REGION Network 51: 设备上砖流程 取砖X轴提前下降判断
   RUNG wire#powerrail
      { S7_Templates := "SrcType := DInt" } GE_Contact(in1 := #Z轴高速转低速编码值, in2 := #取砖X轴提前下降设定值)
      Coil( #上砖提前下降判断标志位 )
   END_RUNG
   // the same network as SCL:
   #上砖提前下降判断标志位 := #Z轴高速转低速编码值 >= #取砖X轴提前下降设定值;
END_REGION

REGION Network 52: 设备上砖流程 Z轴提前下降
   RUNG wire#powerrail
      Contact( #"上砖x轴正转转低速-待命位到2库" )
      wire#w1
      { S7_Templates := "SrcType := Byte" } EQ_Contact(in1 := #机械手取放砖选择, in2 := 2)
      wire#w2
      Contact( #上砖提前下降判断标志位 )
      Contact( #上砖z轴提前下降中间变量 )
      wire#w3
      I_Contact( #设备报警标志位 )
      Contact( #设备启动标志位 )
      S_Coil( #上砖z轴AB库位下降 )
   END_RUNG
   RUNG wire#powerrail
      Contact( #"上砖x轴反转转低速-待命位到1库" )
   END_RUNG wire#w1
   RUNG wire#w2
      I_Contact( #上砖提前下降判断标志位 )
      Contact( #上砖x轴到达A库下方中间变量 )
   END_RUNG wire#w3
   // the same network as SCL:
   IF (#"上砖x轴正转转低速-待命位到2库" OR #"上砖x轴反转转低速-待命位到1库") AND (#机械手取放砖选择 = 2) AND ((#上砖提前下降判断标志位 AND #上砖z轴提前下降中间变量) OR (NOT #上砖提前下降判断标志位 AND #上砖x轴到达A库下方中间变量)) AND NOT #设备报警标志位 AND #设备启动标志位 THEN
       #上砖z轴AB库位下降 := TRUE;
   END_IF;
END_REGION

REGION Network 53: 设备上砖流程 z轴下降取砖
   RUNG wire#powerrail
      Contact( #"上砖x轴正转转低速-待命位到2库" )
      wire#w1
      { S7_Templates := "SrcType := Byte" } EQ_Contact(in1 := #机械手取放砖选择, in2 := 2)
      Contact( #上砖x轴到达A库下方中间变量 )
      I_Contact( #设备报警标志位 )
      wire#w2
      R_Coil( #上砖X轴快速移动2库 )
   END_RUNG
   RUNG wire#powerrail
      Contact( #"上砖x轴反转转低速-待命位到1库" )
   END_RUNG wire#w1
   RUNG wire#w2
      R_Coil( #上砖X轴快速移动1库 )
   END_RUNG
   RUNG wire#w2
      R_Coil( #"上砖x轴正转转低速-待命位到2库" )
   END_RUNG
   RUNG wire#w2
      R_Coil( #"上砖x轴反转转低速-待命位到1库" )
   END_RUNG
   RUNG wire#w2
      Move(in := 0, out1 => #X轴减速光电通断次数, out2 => #减速光电计数传送)
   END_RUNG
   // the same network as SCL:
   IF (#"上砖x轴正转转低速-待命位到2库" OR #"上砖x轴反转转低速-待命位到1库") AND (#机械手取放砖选择 = 2) AND #上砖x轴到达A库下方中间变量 AND NOT #设备报警标志位 THEN
       #上砖X轴快速移动2库 := FALSE;
       #上砖X轴快速移动1库 := FALSE;
   END_IF;
   #_w1 := (#"上砖x轴正转转低速-待命位到2库" OR #"上砖x轴反转转低速-待命位到1库") AND (#机械手取放砖选择 = 2) AND #上砖x轴到达A库下方中间变量 AND NOT #设备报警标志位;
   IF #_w1 THEN
       #"上砖x轴正转转低速-待命位到2库" := FALSE;
       #"上砖x轴反转转低速-待命位到1库" := FALSE;
       #X轴减速光电通断次数 := 0;
       #减速光电计数传送 := 0;
   END_IF;
END_REGION

REGION Network 54: 设备上砖流程 到达检测，Z轴停止
   #上砖z轴AB库置取砖到位中间变量 := #上砖z轴AB库位下降 AND (#W轴吸取接近开关 OR #W轴吸取极限接近开关) AND (((#Z轴编码器实时值 >= #Z轴停止编码值下限) AND (#Z轴编码器实时值 <= #Z轴停止编码值上限)) OR #上砖吸取接近稳定时间定时器.Q);
   IF #上砖z轴AB库位下降 AND (#Z轴编码器实时值 > #Z轴高速转低速编码值) THEN #上砖真空电磁阀打开 := TRUE; END_IF;
   #上砖吸取接近稳定时间定时器.TON(IN := #上砖z轴AB库位下降 AND #W轴吸取接近开关, PT := #吸取到位稳定时间);   // TON coil
END_REGION

REGION Network 55: 设备上砖流程 压力开关检测标志位
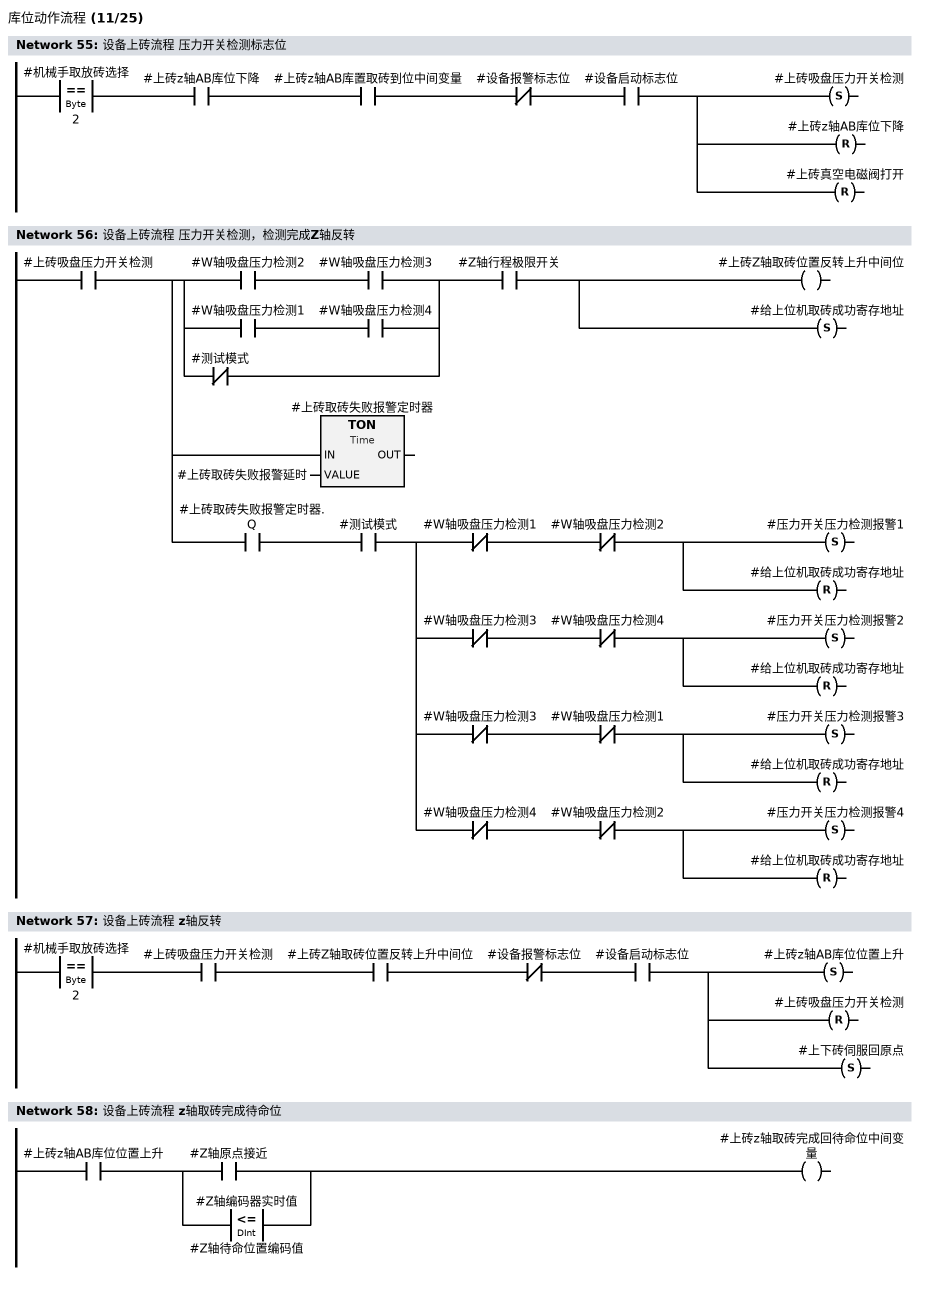
   RUNG wire#powerrail
      { S7_Templates := "SrcType := Byte" } EQ_Contact(in1 := #机械手取放砖选择, in2 := 2)
      Contact( #上砖z轴AB库位下降 )
      Contact( #上砖z轴AB库置取砖到位中间变量 )
      I_Contact( #设备报警标志位 )
      Contact( #设备启动标志位 )
      wire#w1
      S_Coil( #上砖吸盘压力开关检测 )
   END_RUNG
   RUNG wire#w1
      R_Coil( #上砖z轴AB库位下降 )
   END_RUNG
   RUNG wire#w1
      R_Coil( #上砖真空电磁阀打开 )
   END_RUNG
   // the same network as SCL:
   IF (#机械手取放砖选择 = 2) AND #上砖z轴AB库位下降 AND #上砖z轴AB库置取砖到位中间变量 AND NOT #设备报警标志位 AND #设备启动标志位 THEN
       #上砖吸盘压力开关检测 := TRUE;
   END_IF;
   #_w1 := (#机械手取放砖选择 = 2) AND #上砖z轴AB库位下降 AND #上砖z轴AB库置取砖到位中间变量 AND NOT #设备报警标志位 AND #设备启动标志位;
   IF #_w1 THEN
       #上砖z轴AB库位下降 := FALSE;
       #上砖真空电磁阀打开 := FALSE;
   END_IF;
END_REGION

REGION Network 56: 设备上砖流程 压力开关检测，检测完成Z轴反转
   #上砖Z轴取砖位置反转上升中间位 := #上砖吸盘压力开关检测 AND ((#W轴吸盘压力检测2 AND #W轴吸盘压力检测3) OR (#W轴吸盘压力检测1 AND #W轴吸盘压力检测4) OR NOT #测试模式) AND #Z轴行程极限开关;
   IF #上砖Z轴取砖位置反转上升中间位 THEN #给上位机取砖成功寄存地址 := TRUE; END_IF;
   #上砖取砖失败报警定时器.TON(IN := #上砖吸盘压力开关检测, PT := #上砖取砖失败报警延时);   // TON coil
   #_w1 := #上砖吸盘压力开关检测 AND #上砖取砖失败报警定时器.Q AND #测试模式;
   IF #_w1 AND NOT #W轴吸盘压力检测1 AND NOT #W轴吸盘压力检测2 THEN
       #压力开关压力检测报警1 := TRUE;
       #给上位机取砖成功寄存地址 := FALSE;
   END_IF;
   IF #_w1 AND NOT #W轴吸盘压力检测3 AND NOT #W轴吸盘压力检测4 THEN
       #压力开关压力检测报警2 := TRUE;
       #给上位机取砖成功寄存地址 := FALSE;
   END_IF;
   IF #_w1 AND NOT #W轴吸盘压力检测3 AND NOT #W轴吸盘压力检测1 THEN
       #压力开关压力检测报警3 := TRUE;
       #给上位机取砖成功寄存地址 := FALSE;
   END_IF;
   IF #_w1 AND NOT #W轴吸盘压力检测4 AND NOT #W轴吸盘压力检测2 THEN
       #压力开关压力检测报警4 := TRUE;
       #给上位机取砖成功寄存地址 := FALSE;
   END_IF;
END_REGION

REGION Network 57: 设备上砖流程 z轴反转
   RUNG wire#powerrail
      { S7_Templates := "SrcType := Byte" } EQ_Contact(in1 := #机械手取放砖选择, in2 := 2)
      Contact( #上砖吸盘压力开关检测 )
      Contact( #上砖Z轴取砖位置反转上升中间位 )
      I_Contact( #设备报警标志位 )
      Contact( #设备启动标志位 )
      wire#w1
      S_Coil( #上砖z轴AB库位位置上升 )
   END_RUNG
   RUNG wire#w1
      R_Coil( #上砖吸盘压力开关检测 )
   END_RUNG
   RUNG wire#w1
      S_Coil( #上下砖伺服回原点 )
   END_RUNG
   // the same network as SCL:
   IF (#机械手取放砖选择 = 2) AND #上砖吸盘压力开关检测 AND #上砖Z轴取砖位置反转上升中间位 AND NOT #设备报警标志位 AND #设备启动标志位 THEN
       #上砖z轴AB库位位置上升 := TRUE;
   END_IF;
   #_w1 := (#机械手取放砖选择 = 2) AND #上砖吸盘压力开关检测 AND #上砖Z轴取砖位置反转上升中间位 AND NOT #设备报警标志位 AND #设备启动标志位;
   IF #_w1 THEN
       #上砖吸盘压力开关检测 := FALSE;
       #上下砖伺服回原点 := TRUE;
   END_IF;
END_REGION

REGION Network 58: 设备上砖流程 z轴取砖完成待命位
   RUNG wire#powerrail
      Contact( #上砖z轴AB库位位置上升 )
      wire#w1
      Contact( #Z轴原点接近 )
      wire#w2
      Coil( #上砖z轴取砖完成回待命位中间变量 )
   END_RUNG
   RUNG wire#w1
      { S7_Templates := "SrcType := DInt" } LE_Contact(in1 := #Z轴编码器实时值, in2 := #Z轴待命位置编码值)
   END_RUNG wire#w2
   // the same network as SCL:
   #上砖z轴取砖完成回待命位中间变量 := #上砖z轴AB库位位置上升 AND (#Z轴原点接近 OR (#Z轴编码器实时值 <= #Z轴待命位置编码值));
END_REGION

REGION Network 59: 设备上砖流程 X轴正转高速A库--待命位 X轴反转高速B库---待命位
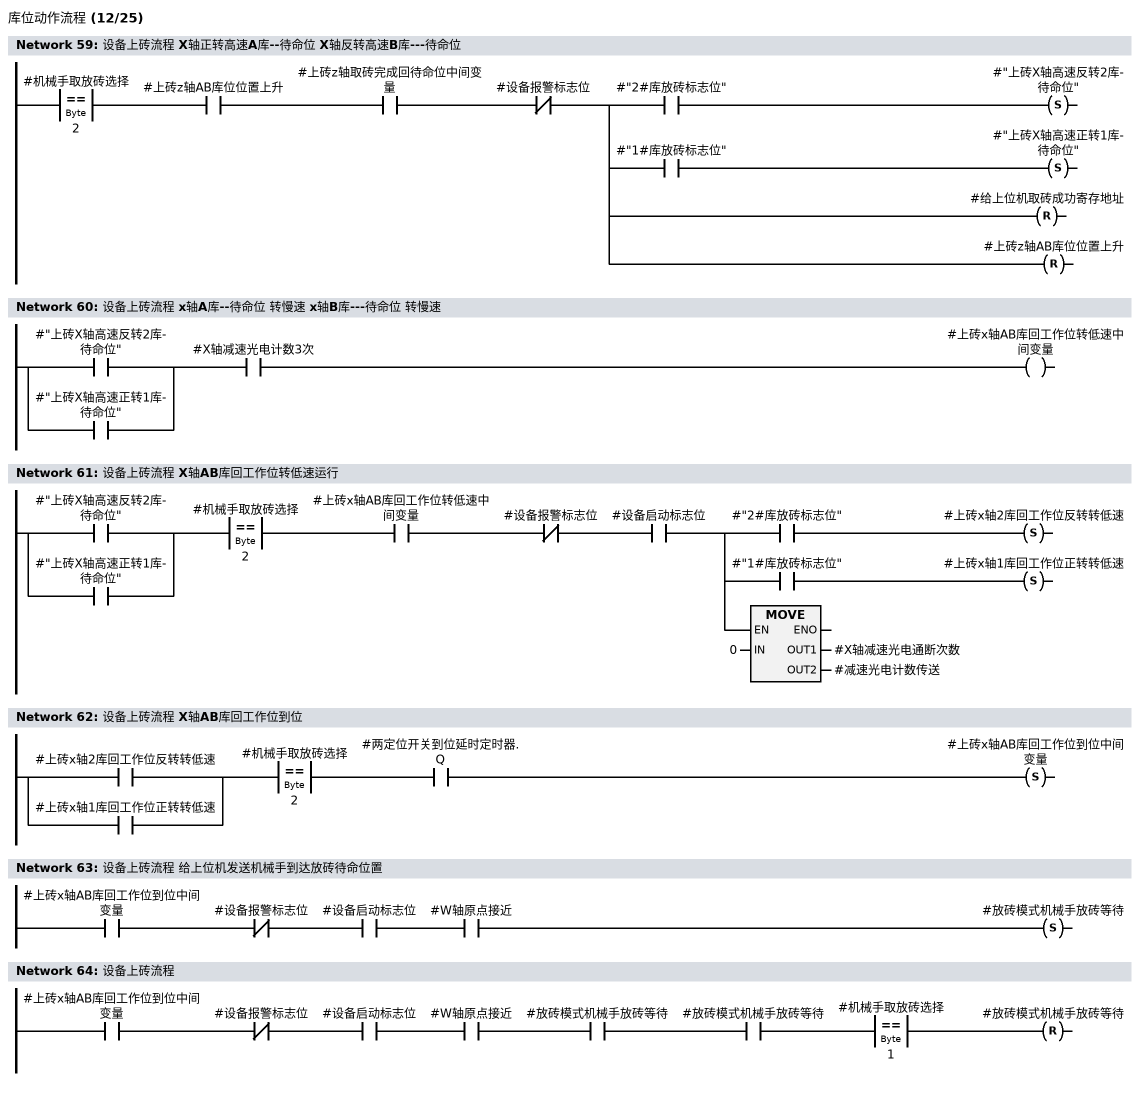
   RUNG wire#powerrail
      { S7_Templates := "SrcType := Byte" } EQ_Contact(in1 := #机械手取放砖选择, in2 := 2)
      Contact( #上砖z轴AB库位位置上升 )
      Contact( #上砖z轴取砖完成回待命位中间变量 )
      I_Contact( #设备报警标志位 )
      wire#w1
      Contact( #"2#库放砖标志位" )
      S_Coil( #"上砖X轴高速反转2库-待命位" )
   END_RUNG
   RUNG wire#w1
      Contact( #"1#库放砖标志位" )
      S_Coil( #"上砖X轴高速正转1库-待命位" )
   END_RUNG
   RUNG wire#w1
      R_Coil( #给上位机取砖成功寄存地址 )
   END_RUNG
   RUNG wire#w1
      R_Coil( #上砖z轴AB库位位置上升 )
   END_RUNG
   // the same network as SCL:
   #_w1 := (#机械手取放砖选择 = 2) AND #上砖z轴AB库位位置上升 AND #上砖z轴取砖完成回待命位中间变量 AND NOT #设备报警标志位;
   IF #_w1 AND #"2#库放砖标志位" THEN #"上砖X轴高速反转2库-待命位" := TRUE; END_IF;
   IF #_w1 AND #"1#库放砖标志位" THEN #"上砖X轴高速正转1库-待命位" := TRUE; END_IF;
   IF #_w1 THEN
       #给上位机取砖成功寄存地址 := FALSE;
       #上砖z轴AB库位位置上升 := FALSE;
   END_IF;
END_REGION

REGION Network 60: 设备上砖流程 x轴A库--待命位 转慢速 x轴B库---待命位 转慢速
   RUNG wire#powerrail
      Contact( #"上砖X轴高速反转2库-待命位" )
      wire#w1
      Contact( #X轴减速光电计数3次 )
      Coil( #上砖x轴AB库回工作位转低速中间变量 )
   END_RUNG
   RUNG wire#powerrail
      Contact( #"上砖X轴高速正转1库-待命位" )
   END_RUNG wire#w1
   // the same network as SCL:
   #上砖x轴AB库回工作位转低速中间变量 := (#"上砖X轴高速反转2库-待命位" OR #"上砖X轴高速正转1库-待命位") AND #X轴减速光电计数3次;
END_REGION

REGION Network 61: 设备上砖流程 X轴AB库回工作位转低速运行
   RUNG wire#powerrail
      Contact( #"上砖X轴高速反转2库-待命位" )
      wire#w1
      { S7_Templates := "SrcType := Byte" } EQ_Contact(in1 := #机械手取放砖选择, in2 := 2)
      Contact( #上砖x轴AB库回工作位转低速中间变量 )
      I_Contact( #设备报警标志位 )
      Contact( #设备启动标志位 )
      wire#w2
      Contact( #"2#库放砖标志位" )
      S_Coil( #上砖x轴2库回工作位反转转低速 )
   END_RUNG
   RUNG wire#powerrail
      Contact( #"上砖X轴高速正转1库-待命位" )
   END_RUNG wire#w1
   RUNG wire#w2
      Contact( #"1#库放砖标志位" )
      S_Coil( #上砖x轴1库回工作位正转转低速 )
   END_RUNG
   RUNG wire#w2
      Move(in := 0, out1 => #X轴减速光电通断次数, out2 => #减速光电计数传送)
   END_RUNG
   // the same network as SCL:
   #_w1 := (#"上砖X轴高速反转2库-待命位" OR #"上砖X轴高速正转1库-待命位") AND (#机械手取放砖选择 = 2) AND #上砖x轴AB库回工作位转低速中间变量 AND NOT #设备报警标志位 AND #设备启动标志位;
   IF #_w1 AND #"2#库放砖标志位" THEN #上砖x轴2库回工作位反转转低速 := TRUE; END_IF;
   IF #_w1 AND #"1#库放砖标志位" THEN #上砖x轴1库回工作位正转转低速 := TRUE; END_IF;
   IF #_w1 THEN
       #X轴减速光电通断次数 := 0;
       #减速光电计数传送 := 0;
   END_IF;
END_REGION

REGION Network 62: 设备上砖流程 X轴AB库回工作位到位
   RUNG wire#powerrail
      Contact( #上砖x轴2库回工作位反转转低速 )
      wire#w1
      { S7_Templates := "SrcType := Byte" } EQ_Contact(in1 := #机械手取放砖选择, in2 := 2)
      Contact( #两定位开关到位延时定时器.Q )
      S_Coil( #上砖x轴AB库回工作位到位中间变量 )
   END_RUNG
   RUNG wire#powerrail
      Contact( #上砖x轴1库回工作位正转转低速 )
   END_RUNG wire#w1
   // the same network as SCL:
   IF (#上砖x轴2库回工作位反转转低速 OR #上砖x轴1库回工作位正转转低速) AND (#机械手取放砖选择 = 2) AND #两定位开关到位延时定时器.Q THEN
       #上砖x轴AB库回工作位到位中间变量 := TRUE;
   END_IF;
END_REGION

REGION Network 63: 设备上砖流程 给上位机发送机械手到达放砖待命位置
   RUNG wire#powerrail
      Contact( #上砖x轴AB库回工作位到位中间变量 )
      I_Contact( #设备报警标志位 )
      Contact( #设备启动标志位 )
      Contact( #W轴原点接近 )
      S_Coil( #放砖模式机械手放砖等待 )
   END_RUNG
   // the same network as SCL:
   IF #上砖x轴AB库回工作位到位中间变量 AND NOT #设备报警标志位 AND #设备启动标志位 AND #W轴原点接近 THEN #放砖模式机械手放砖等待 := TRUE; END_IF;
END_REGION

REGION Network 64: 设备上砖流程
   RUNG wire#powerrail
      Contact( #上砖x轴AB库回工作位到位中间变量 )
      I_Contact( #设备报警标志位 )
      Contact( #设备启动标志位 )
      Contact( #W轴原点接近 )
      Contact( #放砖模式机械手放砖等待 )
      Contact( #放砖模式机械手放砖等待 )
      { S7_Templates := "SrcType := Byte" } EQ_Contact(in1 := #机械手取放砖选择, in2 := 1)
      R_Coil( #放砖模式机械手放砖等待 )
   END_RUNG
   // the same network as SCL:
   IF #上砖x轴AB库回工作位到位中间变量 AND NOT #设备报警标志位 AND #设备启动标志位 AND #W轴原点接近 AND #放砖模式机械手放砖等待 AND #放砖模式机械手放砖等待 AND (#机械手取放砖选择 = 1) THEN
       #放砖模式机械手放砖等待 := FALSE;
   END_IF;
END_REGION

REGION Network 65: 设备上砖流程 z轴下降放砖
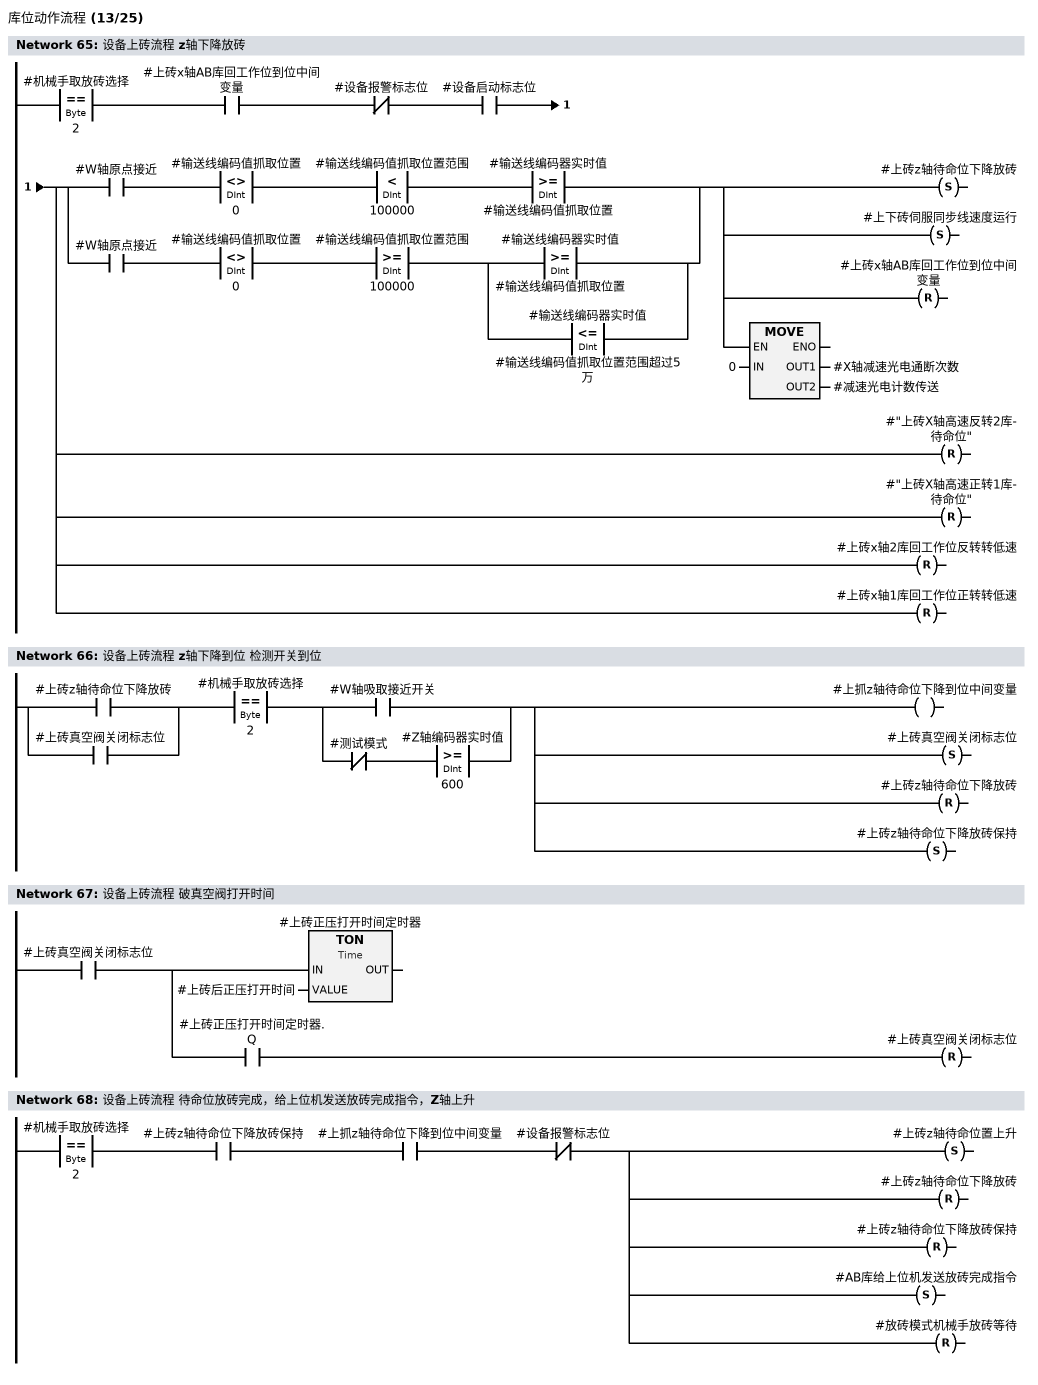
   RUNG wire#powerrail
      { S7_Templates := "SrcType := Byte" } EQ_Contact(in1 := #机械手取放砖选择, in2 := 2)
      Contact( #上砖x轴AB库回工作位到位中间变量 )
      I_Contact( #设备报警标志位 )
      Contact( #设备启动标志位 )
      wire#w1
      Contact( #W轴原点接近 )
      { S7_Templates := "SrcType := DInt" } NE_Contact(in1 := #输送线编码值抓取位置, in2 := 0)
      { S7_Templates := "SrcType := DInt" } LT_Contact(in1 := #输送线编码值抓取位置范围, in2 := 100000)
      { S7_Templates := "SrcType := DInt" } GE_Contact(in1 := #输送线编码器实时值, in2 := #输送线编码值抓取位置)
      wire#w2
      S_Coil( #上砖z轴待命位下降放砖 )
   END_RUNG
   RUNG wire#w1
      Contact( #W轴原点接近 )
      { S7_Templates := "SrcType := DInt" } NE_Contact(in1 := #输送线编码值抓取位置, in2 := 0)
      { S7_Templates := "SrcType := DInt" } GE_Contact(in1 := #输送线编码值抓取位置范围, in2 := 100000)
      wire#w3
      { S7_Templates := "SrcType := DInt" } GE_Contact(in1 := #输送线编码器实时值, in2 := #输送线编码值抓取位置)
   END_RUNG wire#w2
   RUNG wire#w3
      { S7_Templates := "SrcType := DInt" } LE_Contact(in1 := #输送线编码器实时值, in2 := #输送线编码值抓取位置范围超过5万)
   END_RUNG wire#w2
   RUNG wire#w2
      S_Coil( #上下砖伺服同步线速度运行 )
   END_RUNG
   RUNG wire#w2
      R_Coil( #上砖x轴AB库回工作位到位中间变量 )
   END_RUNG
   RUNG wire#w2
      Move(in := 0, out1 => #X轴减速光电通断次数, out2 => #减速光电计数传送)
   END_RUNG
   RUNG wire#w1
      R_Coil( #"上砖X轴高速反转2库-待命位" )
   END_RUNG
   RUNG wire#w1
      R_Coil( #"上砖X轴高速正转1库-待命位" )
   END_RUNG
   RUNG wire#w1
      R_Coil( #上砖x轴2库回工作位反转转低速 )
   END_RUNG
   RUNG wire#w1
      R_Coil( #上砖x轴1库回工作位正转转低速 )
   END_RUNG
   // the same network as SCL:
   #_w1 := (#机械手取放砖选择 = 2) AND #上砖x轴AB库回工作位到位中间变量 AND NOT #设备报警标志位 AND #设备启动标志位;
   IF #_w1 AND ((#W轴原点接近 AND (#输送线编码值抓取位置 <> 0) AND (#输送线编码值抓取位置范围 < 100000) AND (#输送线编码器实时值 >= #输送线编码值抓取位置)) OR (#W轴原点接近 AND (#输送线编码值抓取位置 <> 0) AND (#输送线编码值抓取位置范围 >= 100000) AND ((#输送线编码器实时值 >= #输送线编码值抓取位置) OR (#输送线编码器实时值 <= #输送线编码值抓取位置范围超过5万)))) THEN
       #上砖z轴待命位下降放砖 := TRUE;
       #上下砖伺服同步线速度运行 := TRUE;
       #上砖x轴AB库回工作位到位中间变量 := FALSE;
       #X轴减速光电通断次数 := 0;
       #减速光电计数传送 := 0;
   END_IF;
   IF #_w1 THEN
       #"上砖X轴高速反转2库-待命位" := FALSE;
       #"上砖X轴高速正转1库-待命位" := FALSE;
       #上砖x轴2库回工作位反转转低速 := FALSE;
       #上砖x轴1库回工作位正转转低速 := FALSE;
   END_IF;
END_REGION

REGION Network 66: 设备上砖流程 z轴下降到位 检测开关到位
   RUNG wire#powerrail
      Contact( #上砖z轴待命位下降放砖 )
      wire#w1
      { S7_Templates := "SrcType := Byte" } EQ_Contact(in1 := #机械手取放砖选择, in2 := 2)
      wire#w2
      Contact( #W轴吸取接近开关 )
      wire#w3
      Coil( #上抓z轴待命位下降到位中间变量 )
   END_RUNG
   RUNG wire#powerrail
      Contact( #上砖真空阀关闭标志位 )
   END_RUNG wire#w1
   RUNG wire#w2
      I_Contact( #测试模式 )
      { S7_Templates := "SrcType := DInt" } GE_Contact(in1 := #Z轴编码器实时值, in2 := 600)
   END_RUNG wire#w3
   RUNG wire#w3
      S_Coil( #上砖真空阀关闭标志位 )
   END_RUNG
   RUNG wire#w3
      R_Coil( #上砖z轴待命位下降放砖 )
   END_RUNG
   RUNG wire#w3
      S_Coil( #上砖z轴待命位下降放砖保持 )
   END_RUNG
   // the same network as SCL:
   #上抓z轴待命位下降到位中间变量 := (#上砖z轴待命位下降放砖 OR #上砖真空阀关闭标志位) AND (#机械手取放砖选择 = 2) AND (#W轴吸取接近开关 OR (NOT #测试模式 AND (#Z轴编码器实时值 >= 600)));
   IF #上抓z轴待命位下降到位中间变量 THEN
       #上砖真空阀关闭标志位 := TRUE;
       #上砖z轴待命位下降放砖 := FALSE;
       #上砖z轴待命位下降放砖保持 := TRUE;
   END_IF;
END_REGION

REGION Network 67: 设备上砖流程 破真空阀打开时间
   #上砖正压打开时间定时器.TON(IN := #上砖真空阀关闭标志位, PT := #上砖后正压打开时间);   // TON coil
   IF #上砖真空阀关闭标志位 AND #上砖正压打开时间定时器.Q THEN #上砖真空阀关闭标志位 := FALSE; END_IF;
END_REGION

REGION Network 68: 设备上砖流程 待命位放砖完成，给上位机发送放砖完成指令，Z轴上升
   RUNG wire#powerrail
      { S7_Templates := "SrcType := Byte" } EQ_Contact(in1 := #机械手取放砖选择, in2 := 2)
      Contact( #上砖z轴待命位下降放砖保持 )
      Contact( #上抓z轴待命位下降到位中间变量 )
      I_Contact( #设备报警标志位 )
      wire#w1
      S_Coil( #上砖z轴待命位置上升 )
   END_RUNG
   RUNG wire#w1
      R_Coil( #上砖z轴待命位下降放砖 )
   END_RUNG
   RUNG wire#w1
      R_Coil( #上砖z轴待命位下降放砖保持 )
   END_RUNG
   RUNG wire#w1
      S_Coil( #AB库给上位机发送放砖完成指令 )
   END_RUNG
   RUNG wire#w1
      R_Coil( #放砖模式机械手放砖等待 )
   END_RUNG
   // the same network as SCL:
   IF (#机械手取放砖选择 = 2) AND #上砖z轴待命位下降放砖保持 AND #上抓z轴待命位下降到位中间变量 AND NOT #设备报警标志位 THEN
       #上砖z轴待命位置上升 := TRUE;
       #上砖z轴待命位下降放砖 := FALSE;
   END_IF;
   #_w1 := (#机械手取放砖选择 = 2) AND #上砖z轴待命位下降放砖保持 AND #上抓z轴待命位下降到位中间变量 AND NOT #设备报警标志位;
   IF #_w1 THEN
       #上砖z轴待命位下降放砖保持 := FALSE;
       #AB库给上位机发送放砖完成指令 := TRUE;
       #放砖模式机械手放砖等待 := FALSE;
   END_IF;
END_REGION

REGION Network 69: 设备上砖流程 Z轴待命位上升到目标位
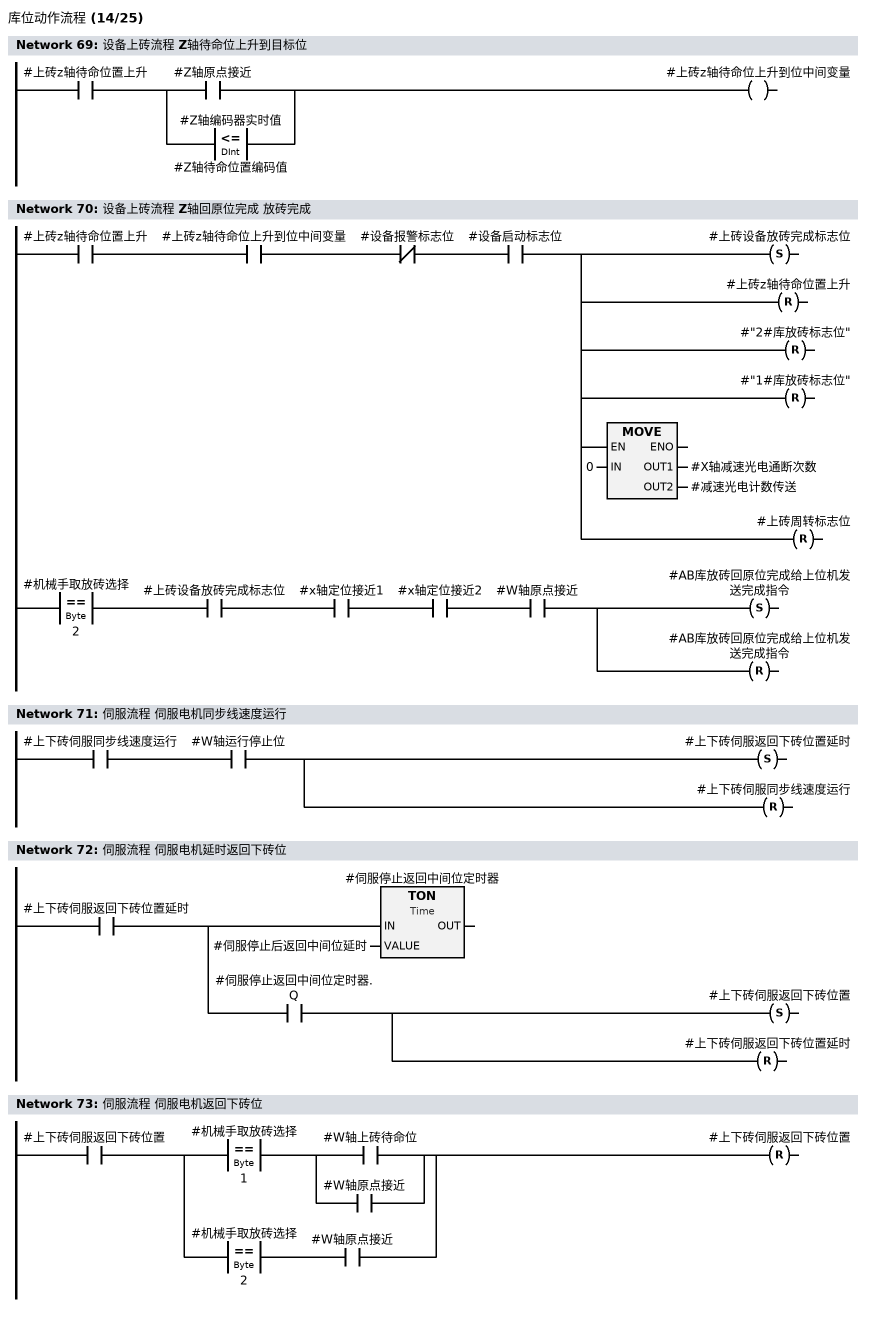
   RUNG wire#powerrail
      Contact( #上砖z轴待命位置上升 )
      wire#w1
      Contact( #Z轴原点接近 )
      wire#w2
      Coil( #上砖z轴待命位上升到位中间变量 )
   END_RUNG
   RUNG wire#w1
      { S7_Templates := "SrcType := DInt" } LE_Contact(in1 := #Z轴编码器实时值, in2 := #Z轴待命位置编码值)
   END_RUNG wire#w2
   // the same network as SCL:
   #上砖z轴待命位上升到位中间变量 := #上砖z轴待命位置上升 AND (#Z轴原点接近 OR (#Z轴编码器实时值 <= #Z轴待命位置编码值));
END_REGION

REGION Network 70: 设备上砖流程 Z轴回原位完成 放砖完成
   RUNG wire#powerrail
      Contact( #上砖z轴待命位置上升 )
      Contact( #上砖z轴待命位上升到位中间变量 )
      I_Contact( #设备报警标志位 )
      Contact( #设备启动标志位 )
      wire#w1
      S_Coil( #上砖设备放砖完成标志位 )
   END_RUNG
   RUNG wire#w1
      R_Coil( #上砖z轴待命位置上升 )
   END_RUNG
   RUNG wire#w1
      R_Coil( #"2#库放砖标志位" )
   END_RUNG
   RUNG wire#w1
      R_Coil( #"1#库放砖标志位" )
   END_RUNG
   RUNG wire#w1
      Move(in := 0, out1 => #X轴减速光电通断次数, out2 => #减速光电计数传送)
   END_RUNG
   RUNG wire#w1
      R_Coil( #上砖周转标志位 )
   END_RUNG
   RUNG wire#powerrail
      { S7_Templates := "SrcType := Byte" } EQ_Contact(in1 := #机械手取放砖选择, in2 := 2)
      Contact( #上砖设备放砖完成标志位 )
      Contact( #x轴定位接近1 )
      Contact( #x轴定位接近2 )
      Contact( #W轴原点接近 )
      wire#w2
      S_Coil( #AB库放砖回原位完成给上位机发送完成指令 )
   END_RUNG
   RUNG wire#w2
      R_Coil( #AB库放砖回原位完成给上位机发送完成指令 )
   END_RUNG
   // the same network as SCL:
   IF #上砖z轴待命位置上升 AND #上砖z轴待命位上升到位中间变量 AND NOT #设备报警标志位 AND #设备启动标志位 THEN #上砖设备放砖完成标志位 := TRUE; END_IF;
   #_w1 := #上砖z轴待命位置上升 AND #上砖z轴待命位上升到位中间变量 AND NOT #设备报警标志位 AND #设备启动标志位;
   IF #_w1 THEN
       #上砖z轴待命位置上升 := FALSE;
       #"2#库放砖标志位" := FALSE;
       #"1#库放砖标志位" := FALSE;
       #X轴减速光电通断次数 := 0;
       #减速光电计数传送 := 0;
       #上砖周转标志位 := FALSE;
   END_IF;
   IF (#机械手取放砖选择 = 2) AND #上砖设备放砖完成标志位 AND #x轴定位接近1 AND #x轴定位接近2 AND #W轴原点接近 THEN
       #AB库放砖回原位完成给上位机发送完成指令 := TRUE;
       #AB库放砖回原位完成给上位机发送完成指令 := FALSE;
   END_IF;
END_REGION

REGION Network 71: 伺服流程 伺服电机同步线速度运行
   RUNG wire#powerrail
      Contact( #上下砖伺服同步线速度运行 )
      Contact( #W轴运行停止位 )
      wire#w1
      S_Coil( #上下砖伺服返回下砖位置延时 )
   END_RUNG
   RUNG wire#w1
      R_Coil( #上下砖伺服同步线速度运行 )
   END_RUNG
   // the same network as SCL:
   IF #上下砖伺服同步线速度运行 AND #W轴运行停止位 THEN
       #上下砖伺服返回下砖位置延时 := TRUE;
       #上下砖伺服同步线速度运行 := FALSE;
   END_IF;
END_REGION

REGION Network 72: 伺服流程 伺服电机延时返回下砖位
   #伺服停止返回中间位定时器.TON(IN := #上下砖伺服返回下砖位置延时, PT := #伺服停止后返回中间位延时);   // TON coil
   IF #上下砖伺服返回下砖位置延时 AND #伺服停止返回中间位定时器.Q THEN
       #上下砖伺服返回下砖位置 := TRUE;
       #上下砖伺服返回下砖位置延时 := FALSE;
   END_IF;
END_REGION

REGION Network 73: 伺服流程 伺服电机返回下砖位
   RUNG wire#powerrail
      Contact( #上下砖伺服返回下砖位置 )
      wire#w1
      { S7_Templates := "SrcType := Byte" } EQ_Contact(in1 := #机械手取放砖选择, in2 := 1)
      wire#w2
      Contact( #W轴上砖待命位 )
      wire#w3
      R_Coil( #上下砖伺服返回下砖位置 )
   END_RUNG
   RUNG wire#w2
      Contact( #W轴原点接近 )
   END_RUNG wire#w3
   RUNG wire#w1
      { S7_Templates := "SrcType := Byte" } EQ_Contact(in1 := #机械手取放砖选择, in2 := 2)
      Contact( #W轴原点接近 )
   END_RUNG wire#w3
   // the same network as SCL:
   IF #上下砖伺服返回下砖位置 AND (((#机械手取放砖选择 = 1) AND (#W轴上砖待命位 OR #W轴原点接近)) OR ((#机械手取放砖选择 = 2) AND #W轴原点接近)) THEN
       #上下砖伺服返回下砖位置 := FALSE;
   END_IF;
END_REGION

REGION Network 74: 伺服流程 伺服回原点
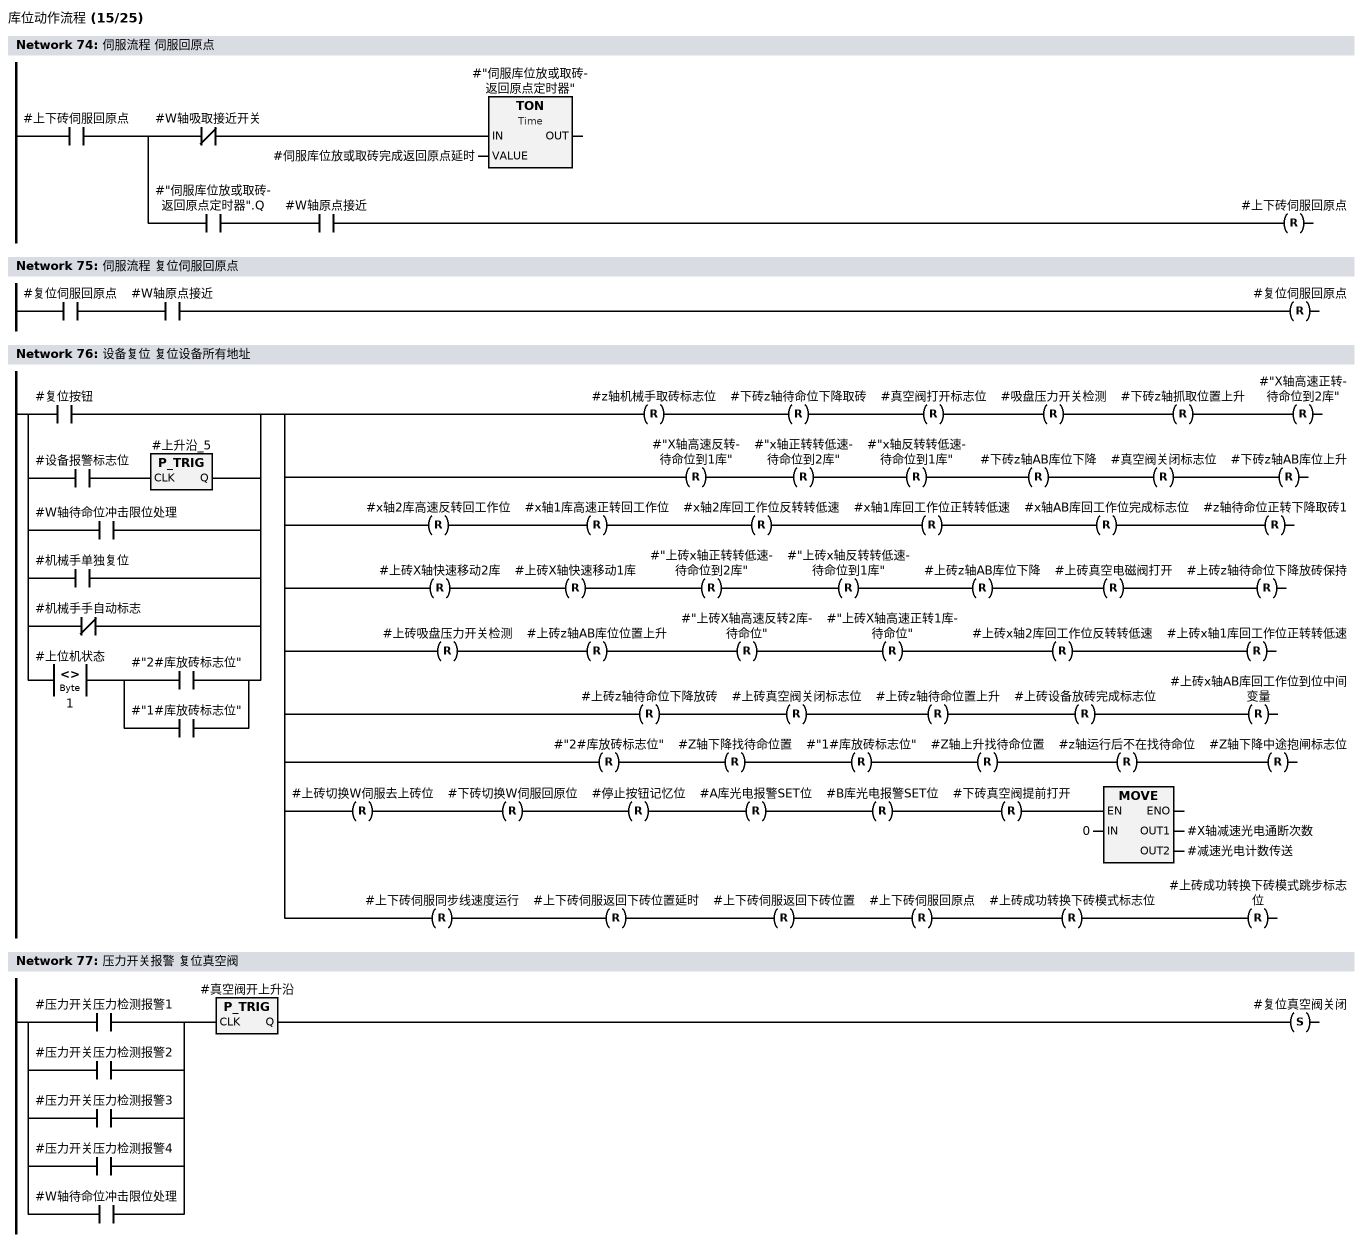
   #"伺服库位放或取砖-返回原点定时器".TON(IN := #上下砖伺服回原点 AND NOT #W轴吸取接近开关, PT := #伺服库位放或取砖完成返回原点延时);   // TON coil
   IF #上下砖伺服回原点 AND #"伺服库位放或取砖-返回原点定时器".Q AND #W轴原点接近 THEN #上下砖伺服回原点 := FALSE; END_IF;
END_REGION

REGION Network 75: 伺服流程 复位伺服回原点
   RUNG wire#powerrail
      Contact( #复位伺服回原点 )
      Contact( #W轴原点接近 )
      R_Coil( #复位伺服回原点 )
   END_RUNG
   // the same network as SCL:
   IF #复位伺服回原点 AND #W轴原点接近 THEN #复位伺服回原点 := FALSE; END_IF;
END_REGION

REGION Network 76: 设备复位 复位设备所有地址
   RUNG wire#powerrail
      Contact( #复位按钮 )
      wire#w1
      R_Coil( #z轴机械手取砖标志位 )
      R_Coil( #下砖z轴待命位下降取砖 )
      R_Coil( #真空阀打开标志位 )
      R_Coil( #吸盘压力开关检测 )
      R_Coil( #下砖z轴抓取位置上升 )
      R_Coil( #"X轴高速正转-待命位到2库" )
   END_RUNG
   RUNG wire#powerrail
      Contact( #设备报警标志位 )
      P_Trig( #上升沿_5 )
   END_RUNG wire#w1
   RUNG wire#powerrail
      Contact( #W轴待命位冲击限位处理 )
   END_RUNG wire#w1
   RUNG wire#powerrail
      Contact( #机械手单独复位 )
   END_RUNG wire#w1
   RUNG wire#powerrail
      I_Contact( #机械手手自动标志 )
   END_RUNG wire#w1
   RUNG wire#powerrail
      { S7_Templates := "SrcType := Byte" } NE_Contact(in1 := #上位机状态, in2 := 1)
      wire#w2
      Contact( #"2#库放砖标志位" )
   END_RUNG wire#w1
   RUNG wire#w2
      Contact( #"1#库放砖标志位" )
   END_RUNG wire#w1
   RUNG wire#w1
      R_Coil( #"X轴高速反转-待命位到1库" )
      R_Coil( #"x轴正转转低速-待命位到2库" )
      R_Coil( #"x轴反转转低速-待命位到1库" )
      R_Coil( #下砖z轴AB库位下降 )
      R_Coil( #真空阀关闭标志位 )
      R_Coil( #下砖z轴AB库位上升 )
   END_RUNG
   RUNG wire#w1
      R_Coil( #x轴2库高速反转回工作位 )
      R_Coil( #x轴1库高速正转回工作位 )
      R_Coil( #x轴2库回工作位反转转低速 )
      R_Coil( #x轴1库回工作位正转转低速 )
      R_Coil( #x轴AB库回工作位完成标志位 )
      R_Coil( #z轴待命位正转下降取砖1 )
   END_RUNG
   RUNG wire#w1
      R_Coil( #上砖X轴快速移动2库 )
      R_Coil( #上砖X轴快速移动1库 )
      R_Coil( #"上砖x轴正转转低速-待命位到2库" )
      R_Coil( #"上砖x轴反转转低速-待命位到1库" )
      R_Coil( #上砖z轴AB库位下降 )
      R_Coil( #上砖真空电磁阀打开 )
      R_Coil( #上砖z轴待命位下降放砖保持 )
   END_RUNG
   RUNG wire#w1
      R_Coil( #上砖吸盘压力开关检测 )
      R_Coil( #上砖z轴AB库位位置上升 )
      R_Coil( #"上砖X轴高速反转2库-待命位" )
      R_Coil( #"上砖X轴高速正转1库-待命位" )
      R_Coil( #上砖x轴2库回工作位反转转低速 )
      R_Coil( #上砖x轴1库回工作位正转转低速 )
   END_RUNG
   RUNG wire#w1
      R_Coil( #上砖z轴待命位下降放砖 )
      R_Coil( #上砖真空阀关闭标志位 )
      R_Coil( #上砖z轴待命位置上升 )
      R_Coil( #上砖设备放砖完成标志位 )
      R_Coil( #上砖x轴AB库回工作位到位中间变量 )
   END_RUNG
   RUNG wire#w1
      R_Coil( #"2#库放砖标志位" )
      R_Coil( #Z轴下降找待命位置 )
      R_Coil( #"1#库放砖标志位" )
      R_Coil( #Z轴上升找待命位置 )
      R_Coil( #z轴运行后不在找待命位 )
      R_Coil( #Z轴下降中途抱闸标志位 )
   END_RUNG
   RUNG wire#w1
      R_Coil( #上砖切换W伺服去上砖位 )
      R_Coil( #下砖切换W伺服回原位 )
      R_Coil( #停止按钮记忆位 )
      R_Coil( #A库光电报警SET位 )
      R_Coil( #B库光电报警SET位 )
      R_Coil( #下砖真空阀提前打开 )
      Move(in := 0, out1 => #X轴减速光电通断次数, out2 => #减速光电计数传送)
   END_RUNG
   RUNG wire#w1
      R_Coil( #上下砖伺服同步线速度运行 )
      R_Coil( #上下砖伺服返回下砖位置延时 )
      R_Coil( #上下砖伺服返回下砖位置 )
      R_Coil( #上下砖伺服回原点 )
      R_Coil( #上砖成功转换下砖模式标志位 )
      R_Coil( #上砖成功转换下砖模式跳步标志位 )
   END_RUNG
   // the same network as SCL:
   #_w1 := #设备报警标志位 AND NOT #上升沿_5;   // rising edge
   #上升沿_5 := #设备报警标志位;
   IF #复位按钮 OR #_w1 OR #W轴待命位冲击限位处理 OR #机械手单独复位 OR NOT #机械手手自动标志 OR ((#上位机状态 <> 1) AND (#"2#库放砖标志位" OR #"1#库放砖标志位")) THEN
       #z轴机械手取砖标志位 := FALSE;
       #下砖z轴待命位下降取砖 := FALSE;
       #真空阀打开标志位 := FALSE;
       #吸盘压力开关检测 := FALSE;
       #下砖z轴抓取位置上升 := FALSE;
       #"X轴高速正转-待命位到2库" := FALSE;
       #"X轴高速反转-待命位到1库" := FALSE;
       #"x轴正转转低速-待命位到2库" := FALSE;
       #"x轴反转转低速-待命位到1库" := FALSE;
       #下砖z轴AB库位下降 := FALSE;
       #真空阀关闭标志位 := FALSE;
       #下砖z轴AB库位上升 := FALSE;
       #x轴2库高速反转回工作位 := FALSE;
       #x轴1库高速正转回工作位 := FALSE;
       #x轴2库回工作位反转转低速 := FALSE;
       #x轴1库回工作位正转转低速 := FALSE;
       #x轴AB库回工作位完成标志位 := FALSE;
       #z轴待命位正转下降取砖1 := FALSE;
       #上砖X轴快速移动2库 := FALSE;
       #上砖X轴快速移动1库 := FALSE;
       #"上砖x轴正转转低速-待命位到2库" := FALSE;
       #"上砖x轴反转转低速-待命位到1库" := FALSE;
       #上砖z轴AB库位下降 := FALSE;
       #上砖真空电磁阀打开 := FALSE;
       #上砖z轴待命位下降放砖保持 := FALSE;
       #上砖吸盘压力开关检测 := FALSE;
       #上砖z轴AB库位位置上升 := FALSE;
       #"上砖X轴高速反转2库-待命位" := FALSE;
       #"上砖X轴高速正转1库-待命位" := FALSE;
       #上砖x轴2库回工作位反转转低速 := FALSE;
       #上砖x轴1库回工作位正转转低速 := FALSE;
       #上砖z轴待命位下降放砖 := FALSE;
       #上砖真空阀关闭标志位 := FALSE;
       #上砖z轴待命位置上升 := FALSE;
       #上砖设备放砖完成标志位 := FALSE;
       #上砖x轴AB库回工作位到位中间变量 := FALSE;
   END_IF;
   #_w2 := #复位按钮 OR #_w1 OR #W轴待命位冲击限位处理 OR #机械手单独复位 OR NOT #机械手手自动标志 OR ((#上位机状态 <> 1) AND (#"2#库放砖标志位" OR #"1#库放砖标志位"));
   IF #_w2 THEN
       #"2#库放砖标志位" := FALSE;
       #Z轴下降找待命位置 := FALSE;
       #"1#库放砖标志位" := FALSE;
       #Z轴上升找待命位置 := FALSE;
       #z轴运行后不在找待命位 := FALSE;
       #Z轴下降中途抱闸标志位 := FALSE;
       #上砖切换W伺服去上砖位 := FALSE;
       #下砖切换W伺服回原位 := FALSE;
       #停止按钮记忆位 := FALSE;
       #A库光电报警SET位 := FALSE;
       #B库光电报警SET位 := FALSE;
       #下砖真空阀提前打开 := FALSE;
       #X轴减速光电通断次数 := 0;
       #减速光电计数传送 := 0;
       #上下砖伺服同步线速度运行 := FALSE;
       #上下砖伺服返回下砖位置延时 := FALSE;
       #上下砖伺服返回下砖位置 := FALSE;
       #上下砖伺服回原点 := FALSE;
       #上砖成功转换下砖模式标志位 := FALSE;
       #上砖成功转换下砖模式跳步标志位 := FALSE;
   END_IF;
END_REGION

REGION Network 77: 压力开关报警 复位真空阀
   RUNG wire#powerrail
      Contact( #压力开关压力检测报警1 )
      wire#w1
      P_Trig( #真空阀开上升沿 )
      S_Coil( #复位真空阀关闭 )
   END_RUNG
   RUNG wire#powerrail
      Contact( #压力开关压力检测报警2 )
   END_RUNG wire#w1
   RUNG wire#powerrail
      Contact( #压力开关压力检测报警3 )
   END_RUNG wire#w1
   RUNG wire#powerrail
      Contact( #压力开关压力检测报警4 )
   END_RUNG wire#w1
   RUNG wire#powerrail
      Contact( #W轴待命位冲击限位处理 )
   END_RUNG wire#w1
   // the same network as SCL:
   #_w1 := #压力开关压力检测报警1 OR #压力开关压力检测报警2 OR #压力开关压力检测报警3 OR #压力开关压力检测报警4 OR #W轴待命位冲击限位处理;
   #_w2 := #_w1 AND NOT #真空阀开上升沿;   // rising edge
   #真空阀开上升沿 := #_w1;
   IF #_w2 THEN #复位真空阀关闭 := TRUE; END_IF;
END_REGION

REGION Network 78: 设备复位开始
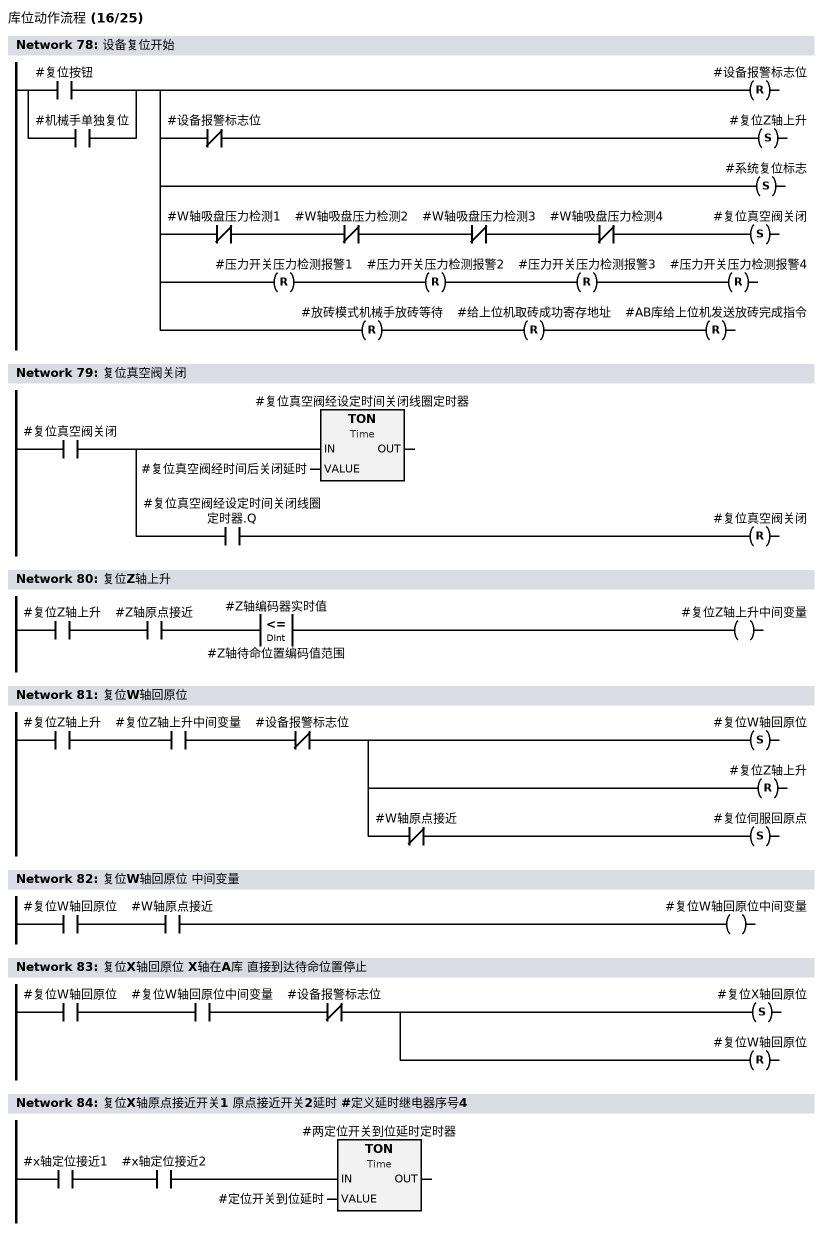
   RUNG wire#powerrail
      Contact( #复位按钮 )
      wire#w1
      R_Coil( #设备报警标志位 )
   END_RUNG
   RUNG wire#powerrail
      Contact( #机械手单独复位 )
   END_RUNG wire#w1
   RUNG wire#w1
      I_Contact( #设备报警标志位 )
      S_Coil( #复位Z轴上升 )
   END_RUNG
   RUNG wire#w1
      S_Coil( #系统复位标志 )
   END_RUNG
   RUNG wire#w1
      I_Contact( #W轴吸盘压力检测1 )
      I_Contact( #W轴吸盘压力检测2 )
      I_Contact( #W轴吸盘压力检测3 )
      I_Contact( #W轴吸盘压力检测4 )
      S_Coil( #复位真空阀关闭 )
   END_RUNG
   RUNG wire#w1
      R_Coil( #压力开关压力检测报警1 )
      R_Coil( #压力开关压力检测报警2 )
      R_Coil( #压力开关压力检测报警3 )
      R_Coil( #压力开关压力检测报警4 )
   END_RUNG
   RUNG wire#w1
      R_Coil( #放砖模式机械手放砖等待 )
      R_Coil( #给上位机取砖成功寄存地址 )
      R_Coil( #AB库给上位机发送放砖完成指令 )
   END_RUNG
   // the same network as SCL:
   #_w1 := #复位按钮 OR #机械手单独复位;
   IF #_w1 THEN #设备报警标志位 := FALSE; END_IF;
   IF #_w1 AND NOT #设备报警标志位 THEN #复位Z轴上升 := TRUE; END_IF;
   IF #_w1 THEN #系统复位标志 := TRUE; END_IF;
   IF #_w1 AND NOT #W轴吸盘压力检测1 AND NOT #W轴吸盘压力检测2 AND NOT #W轴吸盘压力检测3 AND NOT #W轴吸盘压力检测4 THEN
       #复位真空阀关闭 := TRUE;
   END_IF;
   IF #_w1 THEN
       #压力开关压力检测报警1 := FALSE;
       #压力开关压力检测报警2 := FALSE;
       #压力开关压力检测报警3 := FALSE;
       #压力开关压力检测报警4 := FALSE;
       #放砖模式机械手放砖等待 := FALSE;
       #给上位机取砖成功寄存地址 := FALSE;
       #AB库给上位机发送放砖完成指令 := FALSE;
   END_IF;
END_REGION

REGION Network 79: 复位真空阀关闭
   #复位真空阀经设定时间关闭线圈定时器.TON(IN := #复位真空阀关闭, PT := #复位真空阀经时间后关闭延时);   // TON coil
   IF #复位真空阀关闭 AND #复位真空阀经设定时间关闭线圈定时器.Q THEN #复位真空阀关闭 := FALSE; END_IF;
END_REGION

REGION Network 80: 复位Z轴上升
   RUNG wire#powerrail
      Contact( #复位Z轴上升 )
      Contact( #Z轴原点接近 )
      { S7_Templates := "SrcType := DInt" } LE_Contact(in1 := #Z轴编码器实时值, in2 := #Z轴待命位置编码值范围)
      Coil( #复位Z轴上升中间变量 )
   END_RUNG
   // the same network as SCL:
   #复位Z轴上升中间变量 := #复位Z轴上升 AND #Z轴原点接近 AND (#Z轴编码器实时值 <= #Z轴待命位置编码值范围);
END_REGION

REGION Network 81: 复位W轴回原位
   RUNG wire#powerrail
      Contact( #复位Z轴上升 )
      Contact( #复位Z轴上升中间变量 )
      I_Contact( #设备报警标志位 )
      wire#w1
      S_Coil( #复位W轴回原位 )
   END_RUNG
   RUNG wire#w1
      R_Coil( #复位Z轴上升 )
   END_RUNG
   RUNG wire#w1
      I_Contact( #W轴原点接近 )
      S_Coil( #复位伺服回原点 )
   END_RUNG
   // the same network as SCL:
   #_w1 := #复位Z轴上升 AND #复位Z轴上升中间变量 AND NOT #设备报警标志位;
   IF #_w1 THEN
       #复位W轴回原位 := TRUE;
       #复位Z轴上升 := FALSE;
   END_IF;
   IF #_w1 AND NOT #W轴原点接近 THEN #复位伺服回原点 := TRUE; END_IF;
END_REGION

REGION Network 82: 复位W轴回原位 中间变量
   RUNG wire#powerrail
      Contact( #复位W轴回原位 )
      Contact( #W轴原点接近 )
      Coil( #复位W轴回原位中间变量 )
   END_RUNG
   // the same network as SCL:
   #复位W轴回原位中间变量 := #复位W轴回原位 AND #W轴原点接近;
END_REGION

REGION Network 83: 复位X轴回原位 X轴在A库 直接到达待命位置停止
   RUNG wire#powerrail
      Contact( #复位W轴回原位 )
      Contact( #复位W轴回原位中间变量 )
      I_Contact( #设备报警标志位 )
      wire#w1
      S_Coil( #复位X轴回原位 )
   END_RUNG
   RUNG wire#w1
      R_Coil( #复位W轴回原位 )
   END_RUNG
   // the same network as SCL:
   IF #复位W轴回原位 AND #复位W轴回原位中间变量 AND NOT #设备报警标志位 THEN
       #复位X轴回原位 := TRUE;
       #复位W轴回原位 := FALSE;
   END_IF;
END_REGION

REGION Network 84: 复位X轴原点接近开关1 原点接近开关2延时 #定义延时继电器序号4
   #两定位开关到位延时定时器.TON(IN := #x轴定位接近1 AND #x轴定位接近2, PT := #定位开关到位延时);   // TON coil
END_REGION

REGION Network 85: 复位X轴回原位 X轴在A库 直接到达待命位置 经过设定延时停止 X轴在B库 经过定位接近2后反转
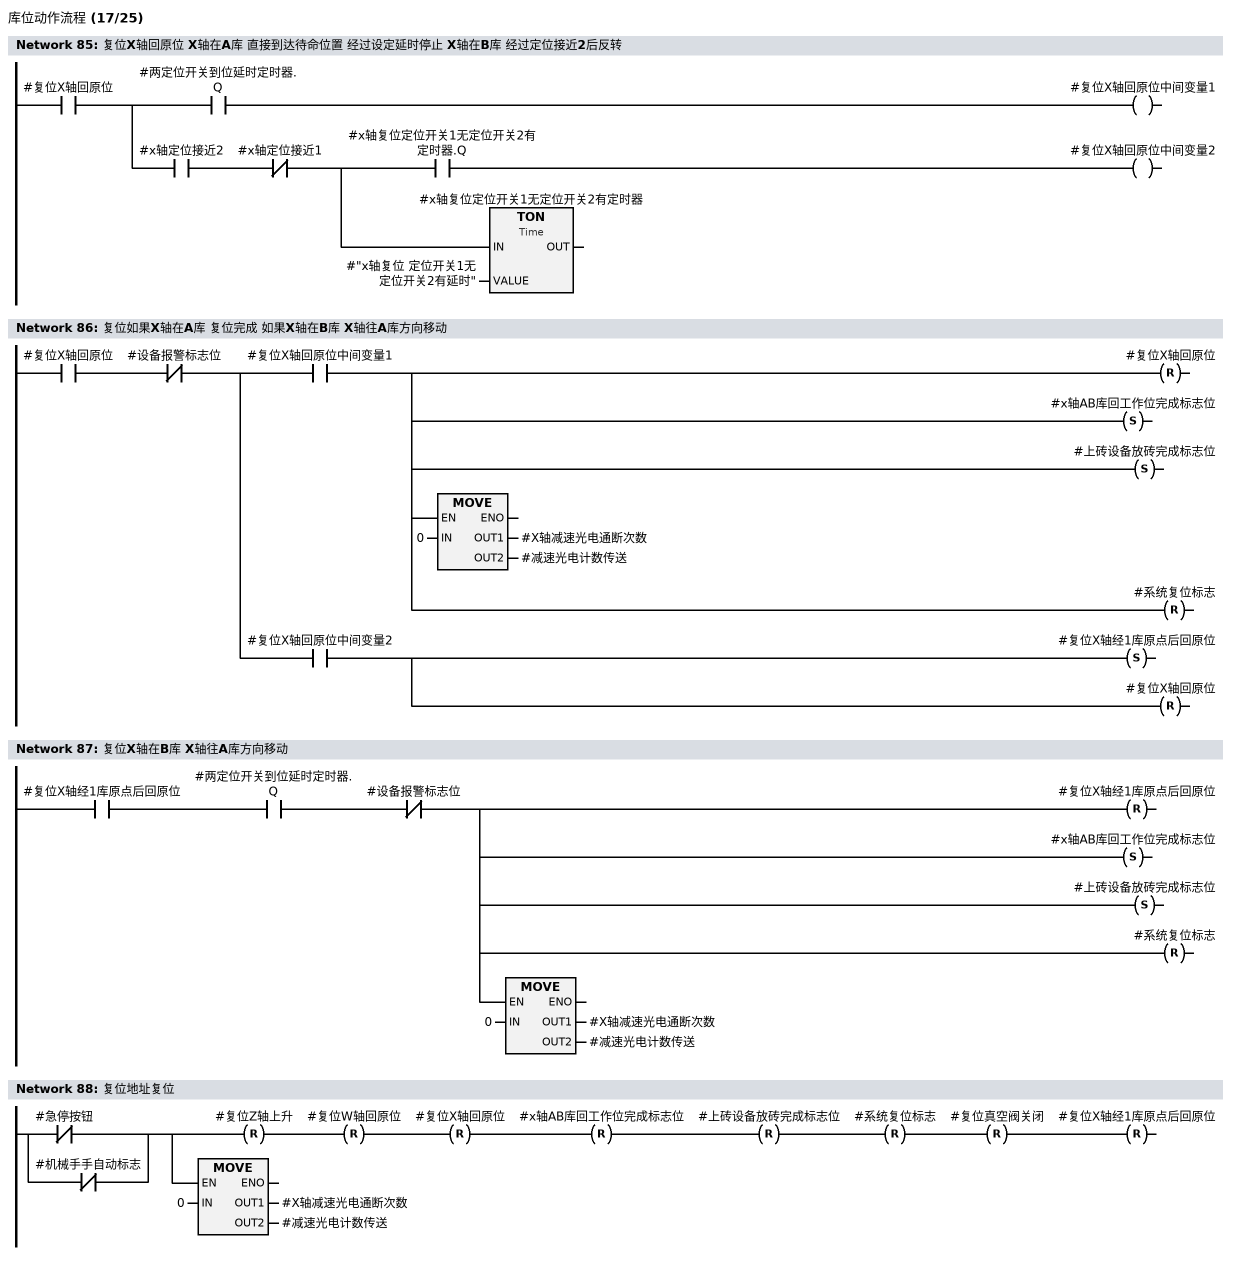
   #复位X轴回原位中间变量1 := #复位X轴回原位 AND #两定位开关到位延时定时器.Q;
   #_w1 := #复位X轴回原位 AND #x轴定位接近2 AND NOT #x轴定位接近1;
   #复位X轴回原位中间变量2 := #_w1 AND #x轴复位定位开关1无定位开关2有定时器.Q;
   #x轴复位定位开关1无定位开关2有定时器.TON(IN := #_w1, PT := #"x轴复位 定位开关1无 定位开关2有延时");   // TON coil
END_REGION

REGION Network 86: 复位如果X轴在A库 复位完成 如果X轴在B库 X轴往A库方向移动
   RUNG wire#powerrail
      Contact( #复位X轴回原位 )
      I_Contact( #设备报警标志位 )
      wire#w1
      Contact( #复位X轴回原位中间变量1 )
      wire#w2
      R_Coil( #复位X轴回原位 )
   END_RUNG
   RUNG wire#w2
      S_Coil( #x轴AB库回工作位完成标志位 )
   END_RUNG
   RUNG wire#w2
      S_Coil( #上砖设备放砖完成标志位 )
   END_RUNG
   RUNG wire#w2
      Move(in := 0, out1 => #X轴减速光电通断次数, out2 => #减速光电计数传送)
   END_RUNG
   RUNG wire#w2
      R_Coil( #系统复位标志 )
   END_RUNG
   RUNG wire#w1
      Contact( #复位X轴回原位中间变量2 )
      wire#w3
      S_Coil( #复位X轴经1库原点后回原位 )
   END_RUNG
   RUNG wire#w3
      R_Coil( #复位X轴回原位 )
   END_RUNG
   // the same network as SCL:
   #_w1 := #复位X轴回原位 AND NOT #设备报警标志位;
   IF #_w1 AND #复位X轴回原位中间变量1 THEN
       #复位X轴回原位 := FALSE;
       #x轴AB库回工作位完成标志位 := TRUE;
       #上砖设备放砖完成标志位 := TRUE;
       #X轴减速光电通断次数 := 0;
       #减速光电计数传送 := 0;
       #系统复位标志 := FALSE;
   END_IF;
   IF #_w1 AND #复位X轴回原位中间变量2 THEN
       #复位X轴经1库原点后回原位 := TRUE;
       #复位X轴回原位 := FALSE;
   END_IF;
END_REGION

REGION Network 87: 复位X轴在B库 X轴往A库方向移动
   RUNG wire#powerrail
      Contact( #复位X轴经1库原点后回原位 )
      Contact( #两定位开关到位延时定时器.Q )
      I_Contact( #设备报警标志位 )
      wire#w1
      R_Coil( #复位X轴经1库原点后回原位 )
   END_RUNG
   RUNG wire#w1
      S_Coil( #x轴AB库回工作位完成标志位 )
   END_RUNG
   RUNG wire#w1
      S_Coil( #上砖设备放砖完成标志位 )
   END_RUNG
   RUNG wire#w1
      R_Coil( #系统复位标志 )
   END_RUNG
   RUNG wire#w1
      Move(in := 0, out1 => #X轴减速光电通断次数, out2 => #减速光电计数传送)
   END_RUNG
   // the same network as SCL:
   #_w1 := #复位X轴经1库原点后回原位 AND #两定位开关到位延时定时器.Q AND NOT #设备报警标志位;
   IF #_w1 THEN
       #复位X轴经1库原点后回原位 := FALSE;
       #x轴AB库回工作位完成标志位 := TRUE;
       #上砖设备放砖完成标志位 := TRUE;
       #系统复位标志 := FALSE;
       #X轴减速光电通断次数 := 0;
       #减速光电计数传送 := 0;
   END_IF;
END_REGION

REGION Network 88: 复位地址复位
   RUNG wire#powerrail
      I_Contact( #急停按钮 )
      wire#w1
      R_Coil( #复位Z轴上升 )
      R_Coil( #复位W轴回原位 )
      R_Coil( #复位X轴回原位 )
      R_Coil( #x轴AB库回工作位完成标志位 )
      R_Coil( #上砖设备放砖完成标志位 )
      R_Coil( #系统复位标志 )
      R_Coil( #复位真空阀关闭 )
      R_Coil( #复位X轴经1库原点后回原位 )
   END_RUNG
   RUNG wire#powerrail
      I_Contact( #机械手手自动标志 )
   END_RUNG wire#w1
   RUNG wire#w1
      Move(in := 0, out1 => #X轴减速光电通断次数, out2 => #减速光电计数传送)
   END_RUNG
   // the same network as SCL:
   IF NOT #急停按钮 OR NOT #机械手手自动标志 THEN
       #复位Z轴上升 := FALSE;
       #复位W轴回原位 := FALSE;
       #复位X轴回原位 := FALSE;
       #x轴AB库回工作位完成标志位 := FALSE;
       #上砖设备放砖完成标志位 := FALSE;
       #系统复位标志 := FALSE;
       #复位真空阀关闭 := FALSE;
       #复位X轴经1库原点后回原位 := FALSE;
       #X轴减速光电通断次数 := 0;
       #减速光电计数传送 := 0;
   END_IF;
END_REGION

REGION Network 89: W轴在待命位置冲击限位处理
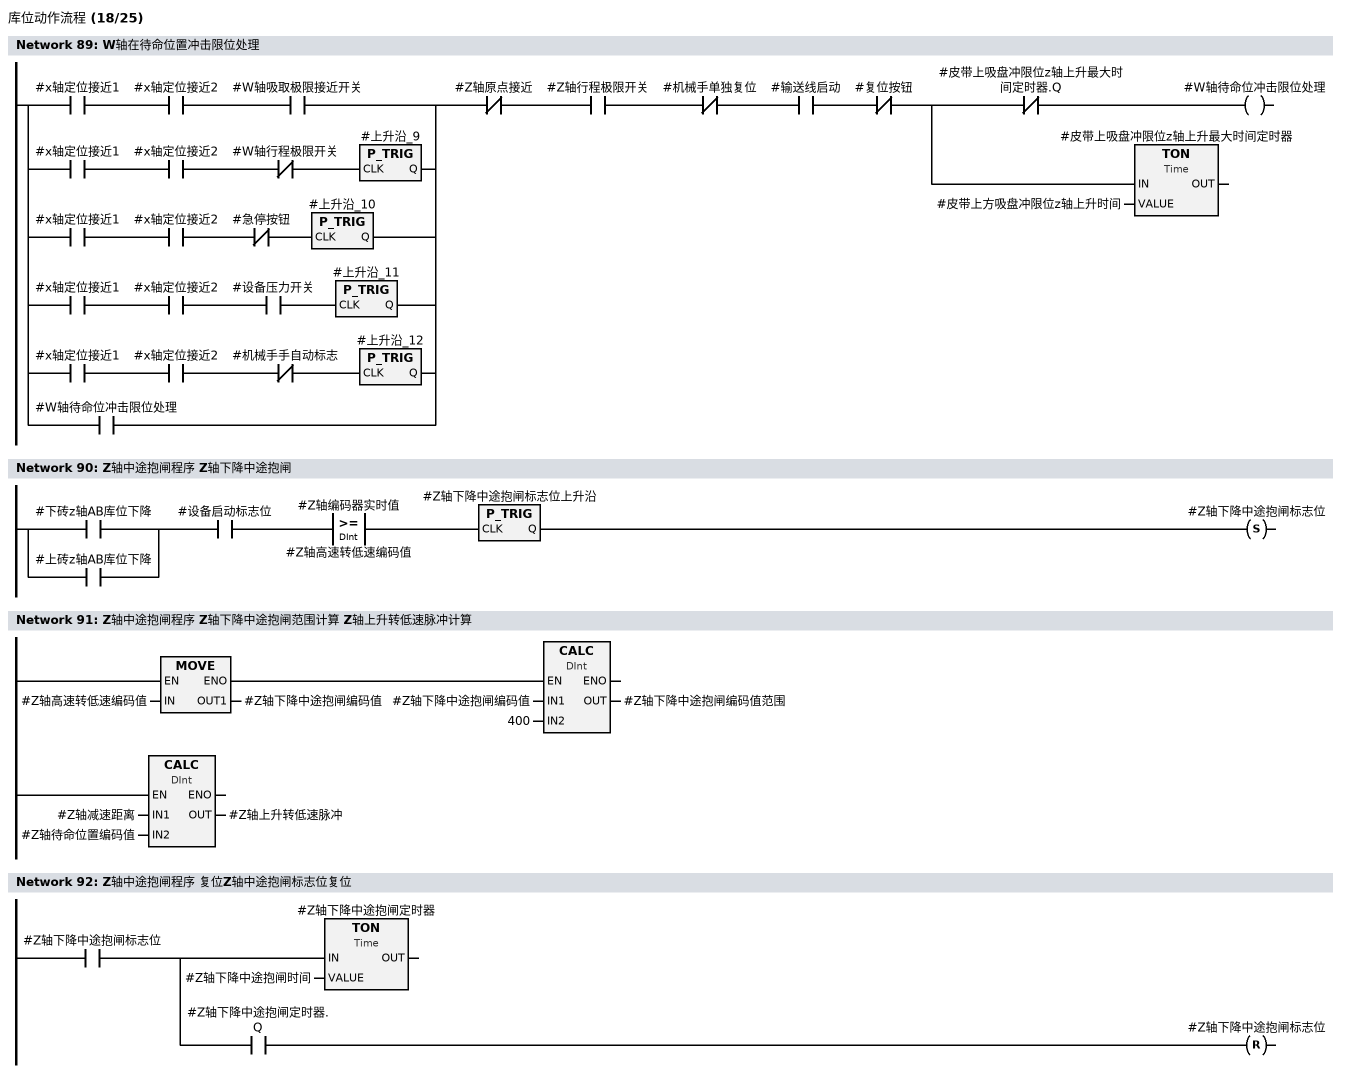
   #_w1 := #x轴定位接近1 AND #x轴定位接近2 AND NOT #W轴行程极限开关;
   #_w2 := #_w1 AND NOT #上升沿_9;   // rising edge
   #上升沿_9 := #_w1;
   #_w3 := #x轴定位接近1 AND #x轴定位接近2 AND NOT #急停按钮;
   #_w4 := #_w3 AND NOT #上升沿_10;   // rising edge
   #上升沿_10 := #_w3;
   #_w5 := #x轴定位接近1 AND #x轴定位接近2 AND #设备压力开关;
   #_w6 := #_w5 AND NOT #上升沿_11;   // rising edge
   #上升沿_11 := #_w5;
   #_w7 := #x轴定位接近1 AND #x轴定位接近2 AND NOT #机械手手自动标志;
   #_w8 := #_w7 AND NOT #上升沿_12;   // rising edge
   #上升沿_12 := #_w7;
   #_w9 := ((#x轴定位接近1 AND #x轴定位接近2 AND #W轴吸取极限接近开关) OR #_w2 OR #_w4 OR #_w6 OR #_w8 OR #W轴待命位冲击限位处理) AND NOT #Z轴原点接近 AND #Z轴行程极限开关 AND NOT #机械手单独复位 AND #输送线启动 AND NOT #复位按钮;
   #W轴待命位冲击限位处理 := #_w9 AND NOT #皮带上吸盘冲限位z轴上升最大时间定时器.Q;
   #皮带上吸盘冲限位z轴上升最大时间定时器.TON(IN := #_w9, PT := #皮带上方吸盘冲限位z轴上升时间);   // TON coil
END_REGION

REGION Network 90: Z轴中途抱闸程序 Z轴下降中途抱闸
   RUNG wire#powerrail
      Contact( #下砖z轴AB库位下降 )
      wire#w1
      Contact( #设备启动标志位 )
      { S7_Templates := "SrcType := DInt" } GE_Contact(in1 := #Z轴编码器实时值, in2 := #Z轴高速转低速编码值)
      P_Trig( #Z轴下降中途抱闸标志位上升沿 )
      S_Coil( #Z轴下降中途抱闸标志位 )
   END_RUNG
   RUNG wire#powerrail
      Contact( #上砖z轴AB库位下降 )
   END_RUNG wire#w1
   // the same network as SCL:
   #_w1 := (#下砖z轴AB库位下降 OR #上砖z轴AB库位下降) AND #设备启动标志位 AND (#Z轴编码器实时值 >= #Z轴高速转低速编码值);
   #_w2 := #_w1 AND NOT #Z轴下降中途抱闸标志位上升沿;   // rising edge
   #Z轴下降中途抱闸标志位上升沿 := #_w1;
   IF #_w2 THEN #Z轴下降中途抱闸标志位 := TRUE; END_IF;
END_REGION

REGION Network 91: Z轴中途抱闸程序 Z轴下降中途抱闸范围计算 Z轴上升转低速脉冲计算
   #Z轴下降中途抱闸编码值 := #Z轴高速转低速编码值;
   CALC(in1 := #Z轴下降中途抱闸编码值, in2 := 400, out => #Z轴下降中途抱闸编码值范围);
   CALC(in1 := #Z轴减速距离, in2 := #Z轴待命位置编码值, out => #Z轴上升转低速脉冲);
END_REGION

REGION Network 92: Z轴中途抱闸程序 复位Z轴中途抱闸标志位复位
   #Z轴下降中途抱闸定时器.TON(IN := #Z轴下降中途抱闸标志位, PT := #Z轴下降中途抱闸时间);   // TON coil
   IF #Z轴下降中途抱闸标志位 AND #Z轴下降中途抱闸定时器.Q THEN #Z轴下降中途抱闸标志位 := FALSE; END_IF;
END_REGION

REGION Network 93: 输出 Z轴下降输出
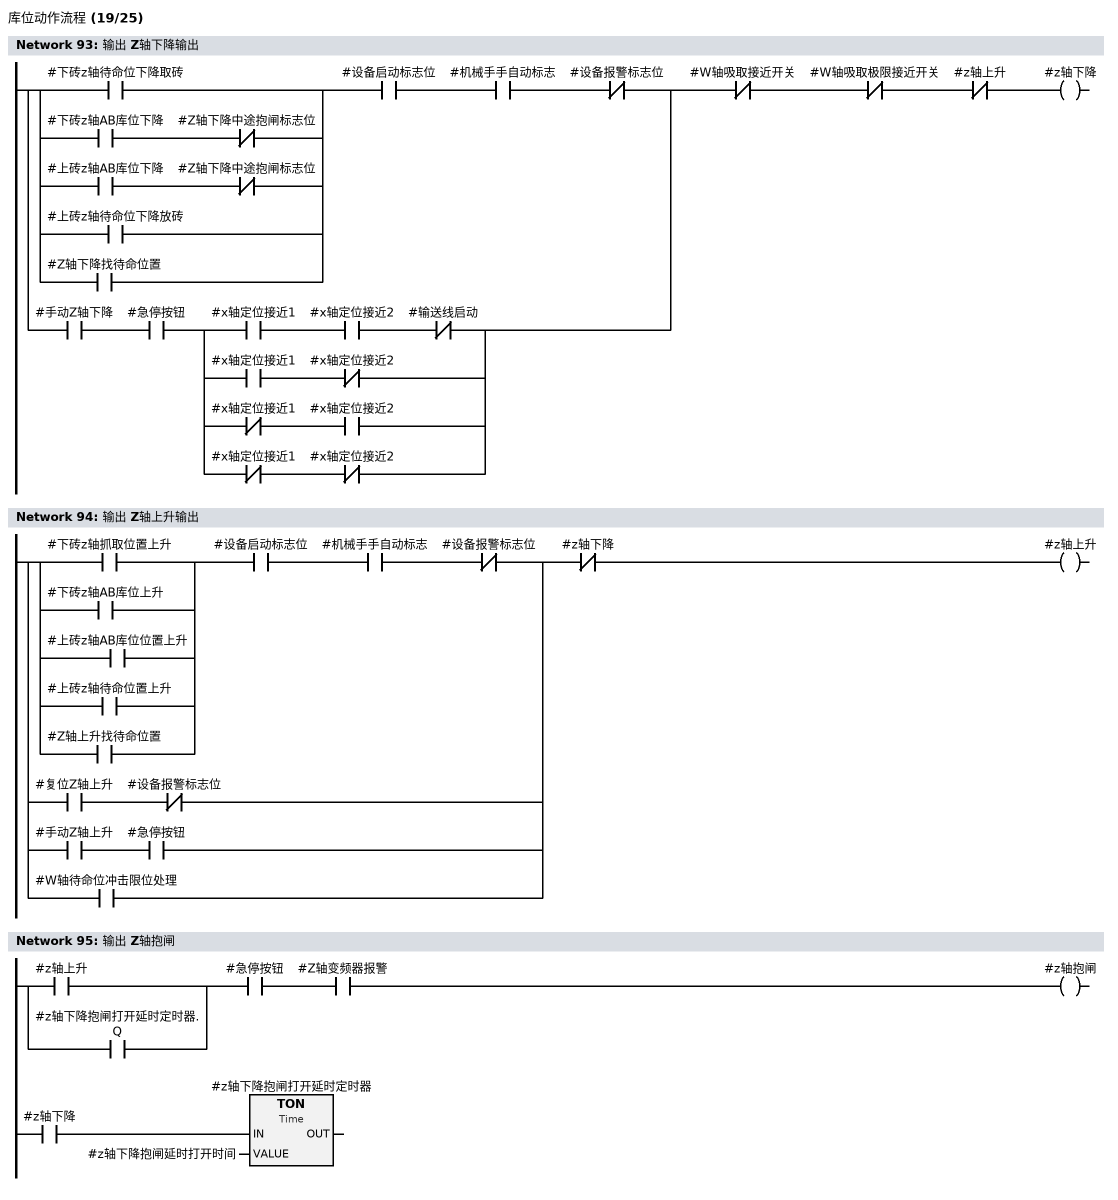
   RUNG wire#powerrail
      Contact( #下砖z轴待命位下降取砖 )
      wire#w1
      Contact( #设备启动标志位 )
      Contact( #机械手手自动标志 )
      I_Contact( #设备报警标志位 )
      wire#w2
      I_Contact( #W轴吸取接近开关 )
      I_Contact( #W轴吸取极限接近开关 )
      I_Contact( #z轴上升 )
      Coil( #z轴下降 )
   END_RUNG
   RUNG wire#powerrail
      Contact( #下砖z轴AB库位下降 )
      I_Contact( #Z轴下降中途抱闸标志位 )
   END_RUNG wire#w1
   RUNG wire#powerrail
      Contact( #上砖z轴AB库位下降 )
      I_Contact( #Z轴下降中途抱闸标志位 )
   END_RUNG wire#w1
   RUNG wire#powerrail
      Contact( #上砖z轴待命位下降放砖 )
   END_RUNG wire#w1
   RUNG wire#powerrail
      Contact( #Z轴下降找待命位置 )
   END_RUNG wire#w1
   RUNG wire#powerrail
      Contact( #手动Z轴下降 )
      Contact( #急停按钮 )
      wire#w3
      Contact( #x轴定位接近1 )
      Contact( #x轴定位接近2 )
      I_Contact( #输送线启动 )
   END_RUNG wire#w2
   RUNG wire#w3
      Contact( #x轴定位接近1 )
      I_Contact( #x轴定位接近2 )
   END_RUNG wire#w2
   RUNG wire#w3
      I_Contact( #x轴定位接近1 )
      Contact( #x轴定位接近2 )
   END_RUNG wire#w2
   RUNG wire#w3
      I_Contact( #x轴定位接近1 )
      I_Contact( #x轴定位接近2 )
   END_RUNG wire#w2
   // the same network as SCL:
   #z轴下降 := (((#下砖z轴待命位下降取砖 OR (#下砖z轴AB库位下降 AND NOT #Z轴下降中途抱闸标志位) OR (#上砖z轴AB库位下降 AND NOT #Z轴下降中途抱闸标志位) OR #上砖z轴待命位下降放砖 OR #Z轴下降找待命位置) AND #设备启动标志位 AND #机械手手自动标志 AND NOT #设备报警标志位) OR (#手动Z轴下降 AND #急停按钮 AND ((#x轴定位接近1 AND #x轴定位接近2 AND NOT #输送线启动) OR (#x轴定位接近1 AND NOT #x轴定位接近2) OR (NOT #x轴定位接近1 AND #x轴定位接近2) OR (NOT #x轴定位接近1 AND NOT #x轴定位接近2)))) AND NOT #W轴吸取接近开关 AND NOT #W轴吸取极限接近开关 AND NOT #z轴上升;
END_REGION

REGION Network 94: 输出 Z轴上升输出
   RUNG wire#powerrail
      Contact( #下砖z轴抓取位置上升 )
      wire#w1
      Contact( #设备启动标志位 )
      Contact( #机械手手自动标志 )
      I_Contact( #设备报警标志位 )
      wire#w2
      I_Contact( #z轴下降 )
      Coil( #z轴上升 )
   END_RUNG
   RUNG wire#powerrail
      Contact( #下砖z轴AB库位上升 )
   END_RUNG wire#w1
   RUNG wire#powerrail
      Contact( #上砖z轴AB库位位置上升 )
   END_RUNG wire#w1
   RUNG wire#powerrail
      Contact( #上砖z轴待命位置上升 )
   END_RUNG wire#w1
   RUNG wire#powerrail
      Contact( #Z轴上升找待命位置 )
   END_RUNG wire#w1
   RUNG wire#powerrail
      Contact( #复位Z轴上升 )
      I_Contact( #设备报警标志位 )
   END_RUNG wire#w2
   RUNG wire#powerrail
      Contact( #手动Z轴上升 )
      Contact( #急停按钮 )
   END_RUNG wire#w2
   RUNG wire#powerrail
      Contact( #W轴待命位冲击限位处理 )
   END_RUNG wire#w2
   // the same network as SCL:
   #z轴上升 := (((#下砖z轴抓取位置上升 OR #下砖z轴AB库位上升 OR #上砖z轴AB库位位置上升 OR #上砖z轴待命位置上升 OR #Z轴上升找待命位置) AND #设备启动标志位 AND #机械手手自动标志 AND NOT #设备报警标志位) OR (#复位Z轴上升 AND NOT #设备报警标志位) OR (#手动Z轴上升 AND #急停按钮) OR #W轴待命位冲击限位处理) AND NOT #z轴下降;
END_REGION

REGION Network 95: 输出 Z轴抱闸
   #z轴抱闸 := (#z轴上升 OR #z轴下降抱闸打开延时定时器.Q) AND #急停按钮 AND #Z轴变频器报警;
   #z轴下降抱闸打开延时定时器.TON(IN := #z轴下降, PT := #z轴下降抱闸延时打开时间);   // TON coil
END_REGION

REGION Network 96: 输出 Z轴端子1-速度
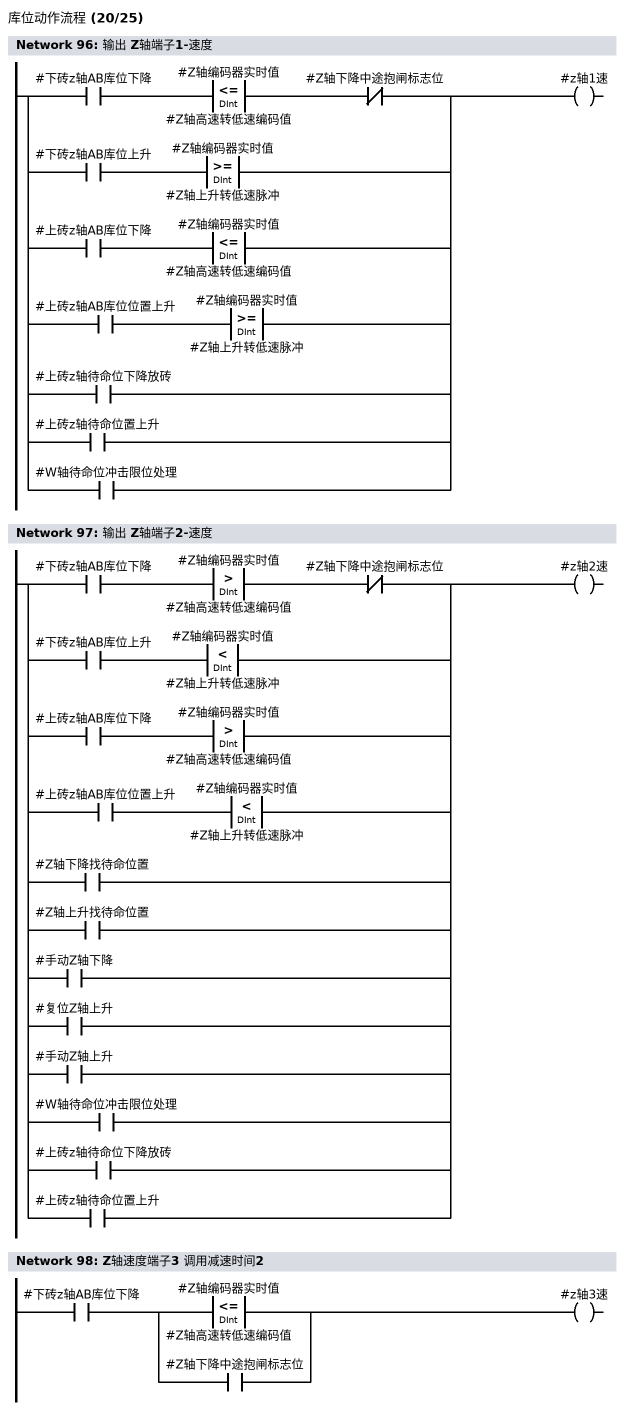
   RUNG wire#powerrail
      Contact( #下砖z轴AB库位下降 )
      { S7_Templates := "SrcType := DInt" } LE_Contact(in1 := #Z轴编码器实时值, in2 := #Z轴高速转低速编码值)
      I_Contact( #Z轴下降中途抱闸标志位 )
      wire#w1
      Coil( #z轴1速 )
   END_RUNG
   RUNG wire#powerrail
      Contact( #下砖z轴AB库位上升 )
      { S7_Templates := "SrcType := DInt" } GE_Contact(in1 := #Z轴编码器实时值, in2 := #Z轴上升转低速脉冲)
   END_RUNG wire#w1
   RUNG wire#powerrail
      Contact( #上砖z轴AB库位下降 )
      { S7_Templates := "SrcType := DInt" } LE_Contact(in1 := #Z轴编码器实时值, in2 := #Z轴高速转低速编码值)
   END_RUNG wire#w1
   RUNG wire#powerrail
      Contact( #上砖z轴AB库位位置上升 )
      { S7_Templates := "SrcType := DInt" } GE_Contact(in1 := #Z轴编码器实时值, in2 := #Z轴上升转低速脉冲)
   END_RUNG wire#w1
   RUNG wire#powerrail
      Contact( #上砖z轴待命位下降放砖 )
   END_RUNG wire#w1
   RUNG wire#powerrail
      Contact( #上砖z轴待命位置上升 )
   END_RUNG wire#w1
   RUNG wire#powerrail
      Contact( #W轴待命位冲击限位处理 )
   END_RUNG wire#w1
   // the same network as SCL:
   #z轴1速 := (#下砖z轴AB库位下降 AND (#Z轴编码器实时值 <= #Z轴高速转低速编码值) AND NOT #Z轴下降中途抱闸标志位) OR (#下砖z轴AB库位上升 AND (#Z轴编码器实时值 >= #Z轴上升转低速脉冲)) OR (#上砖z轴AB库位下降 AND (#Z轴编码器实时值 <= #Z轴高速转低速编码值)) OR (#上砖z轴AB库位位置上升 AND (#Z轴编码器实时值 >= #Z轴上升转低速脉冲)) OR #上砖z轴待命位下降放砖 OR #上砖z轴待命位置上升 OR #W轴待命位冲击限位处理;
END_REGION

REGION Network 97: 输出 Z轴端子2-速度
   RUNG wire#powerrail
      Contact( #下砖z轴AB库位下降 )
      { S7_Templates := "SrcType := DInt" } GT_Contact(in1 := #Z轴编码器实时值, in2 := #Z轴高速转低速编码值)
      I_Contact( #Z轴下降中途抱闸标志位 )
      wire#w1
      Coil( #z轴2速 )
   END_RUNG
   RUNG wire#powerrail
      Contact( #下砖z轴AB库位上升 )
      { S7_Templates := "SrcType := DInt" } LT_Contact(in1 := #Z轴编码器实时值, in2 := #Z轴上升转低速脉冲)
   END_RUNG wire#w1
   RUNG wire#powerrail
      Contact( #上砖z轴AB库位下降 )
      { S7_Templates := "SrcType := DInt" } GT_Contact(in1 := #Z轴编码器实时值, in2 := #Z轴高速转低速编码值)
   END_RUNG wire#w1
   RUNG wire#powerrail
      Contact( #上砖z轴AB库位位置上升 )
      { S7_Templates := "SrcType := DInt" } LT_Contact(in1 := #Z轴编码器实时值, in2 := #Z轴上升转低速脉冲)
   END_RUNG wire#w1
   RUNG wire#powerrail
      Contact( #Z轴下降找待命位置 )
   END_RUNG wire#w1
   RUNG wire#powerrail
      Contact( #Z轴上升找待命位置 )
   END_RUNG wire#w1
   RUNG wire#powerrail
      Contact( #手动Z轴下降 )
   END_RUNG wire#w1
   RUNG wire#powerrail
      Contact( #复位Z轴上升 )
   END_RUNG wire#w1
   RUNG wire#powerrail
      Contact( #手动Z轴上升 )
   END_RUNG wire#w1
   RUNG wire#powerrail
      Contact( #W轴待命位冲击限位处理 )
   END_RUNG wire#w1
   RUNG wire#powerrail
      Contact( #上砖z轴待命位下降放砖 )
   END_RUNG wire#w1
   RUNG wire#powerrail
      Contact( #上砖z轴待命位置上升 )
   END_RUNG wire#w1
   // the same network as SCL:
   #z轴2速 := (#下砖z轴AB库位下降 AND (#Z轴编码器实时值 > #Z轴高速转低速编码值) AND NOT #Z轴下降中途抱闸标志位) OR (#下砖z轴AB库位上升 AND (#Z轴编码器实时值 < #Z轴上升转低速脉冲)) OR (#上砖z轴AB库位下降 AND (#Z轴编码器实时值 > #Z轴高速转低速编码值)) OR (#上砖z轴AB库位位置上升 AND (#Z轴编码器实时值 < #Z轴上升转低速脉冲)) OR #Z轴下降找待命位置 OR #Z轴上升找待命位置 OR #手动Z轴下降 OR #复位Z轴上升 OR #手动Z轴上升 OR #W轴待命位冲击限位处理 OR #上砖z轴待命位下降放砖 OR #上砖z轴待命位置上升;
END_REGION

REGION Network 98: Z轴速度端子3 调用减速时间2
   RUNG wire#powerrail
      Contact( #下砖z轴AB库位下降 )
      wire#w1
      { S7_Templates := "SrcType := DInt" } LE_Contact(in1 := #Z轴编码器实时值, in2 := #Z轴高速转低速编码值)
      wire#w2
      Coil( #z轴3速 )
   END_RUNG
   RUNG wire#w1
      Contact( #Z轴下降中途抱闸标志位 )
   END_RUNG wire#w2
   // the same network as SCL:
   #z轴3速 := #下砖z轴AB库位下降 AND ((#Z轴编码器实时值 <= #Z轴高速转低速编码值) OR #Z轴下降中途抱闸标志位);
END_REGION

REGION Network 99: 输出 真空阀吸真空打开
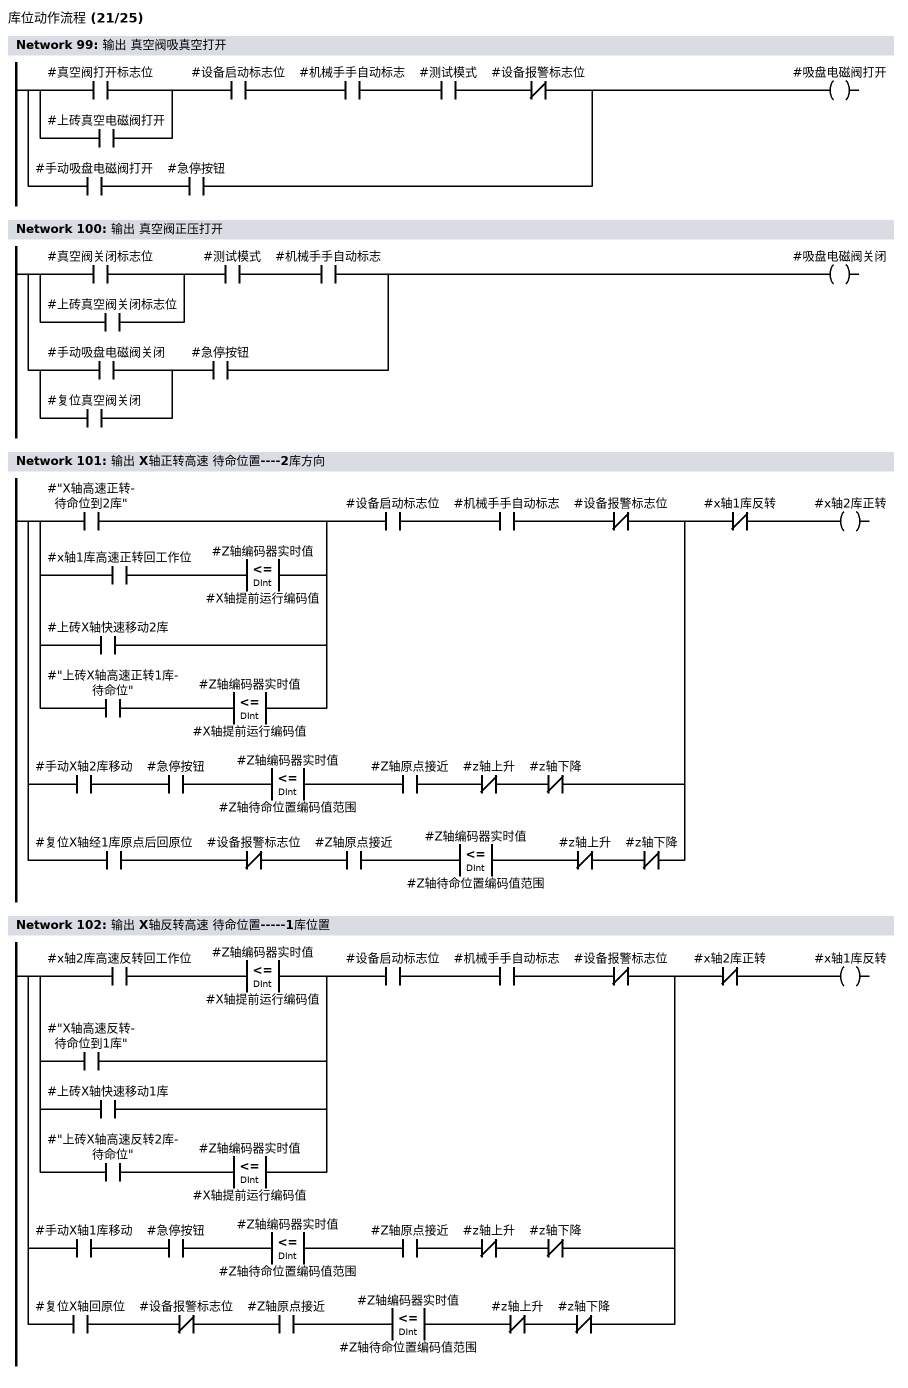
   RUNG wire#powerrail
      Contact( #真空阀打开标志位 )
      wire#w1
      Contact( #设备启动标志位 )
      Contact( #机械手手自动标志 )
      Contact( #测试模式 )
      I_Contact( #设备报警标志位 )
      wire#w2
      Coil( #吸盘电磁阀打开 )
   END_RUNG
   RUNG wire#powerrail
      Contact( #上砖真空电磁阀打开 )
   END_RUNG wire#w1
   RUNG wire#powerrail
      Contact( #手动吸盘电磁阀打开 )
      Contact( #急停按钮 )
   END_RUNG wire#w2
   // the same network as SCL:
   #吸盘电磁阀打开 := ((#真空阀打开标志位 OR #上砖真空电磁阀打开) AND #设备启动标志位 AND #机械手手自动标志 AND #测试模式 AND NOT #设备报警标志位) OR (#手动吸盘电磁阀打开 AND #急停按钮);
END_REGION

REGION Network 100: 输出 真空阀正压打开
   RUNG wire#powerrail
      Contact( #真空阀关闭标志位 )
      wire#w1
      Contact( #测试模式 )
      Contact( #机械手手自动标志 )
      wire#w2
      Coil( #吸盘电磁阀关闭 )
   END_RUNG
   RUNG wire#powerrail
      Contact( #上砖真空阀关闭标志位 )
   END_RUNG wire#w1
   RUNG wire#powerrail
      Contact( #手动吸盘电磁阀关闭 )
      wire#w3
      Contact( #急停按钮 )
   END_RUNG wire#w2
   RUNG wire#powerrail
      Contact( #复位真空阀关闭 )
   END_RUNG wire#w3
   // the same network as SCL:
   #吸盘电磁阀关闭 := ((#真空阀关闭标志位 OR #上砖真空阀关闭标志位) AND #测试模式 AND #机械手手自动标志) OR ((#手动吸盘电磁阀关闭 OR #复位真空阀关闭) AND #急停按钮);
END_REGION

REGION Network 101: 输出 X轴正转高速 待命位置----2库方向
   RUNG wire#powerrail
      Contact( #"X轴高速正转-待命位到2库" )
      wire#w1
      Contact( #设备启动标志位 )
      Contact( #机械手手自动标志 )
      I_Contact( #设备报警标志位 )
      wire#w2
      I_Contact( #x轴1库反转 )
      Coil( #x轴2库正转 )
   END_RUNG
   RUNG wire#powerrail
      Contact( #x轴1库高速正转回工作位 )
      { S7_Templates := "SrcType := DInt" } LE_Contact(in1 := #Z轴编码器实时值, in2 := #X轴提前运行编码值)
   END_RUNG wire#w1
   RUNG wire#powerrail
      Contact( #上砖X轴快速移动2库 )
   END_RUNG wire#w1
   RUNG wire#powerrail
      Contact( #"上砖X轴高速正转1库-待命位" )
      { S7_Templates := "SrcType := DInt" } LE_Contact(in1 := #Z轴编码器实时值, in2 := #X轴提前运行编码值)
   END_RUNG wire#w1
   RUNG wire#powerrail
      Contact( #手动X轴2库移动 )
      Contact( #急停按钮 )
      { S7_Templates := "SrcType := DInt" } LE_Contact(in1 := #Z轴编码器实时值, in2 := #Z轴待命位置编码值范围)
      Contact( #Z轴原点接近 )
      I_Contact( #z轴上升 )
      I_Contact( #z轴下降 )
   END_RUNG wire#w2
   RUNG wire#powerrail
      Contact( #复位X轴经1库原点后回原位 )
      I_Contact( #设备报警标志位 )
      Contact( #Z轴原点接近 )
      { S7_Templates := "SrcType := DInt" } LE_Contact(in1 := #Z轴编码器实时值, in2 := #Z轴待命位置编码值范围)
      I_Contact( #z轴上升 )
      I_Contact( #z轴下降 )
   END_RUNG wire#w2
   // the same network as SCL:
   #x轴2库正转 := (((#"X轴高速正转-待命位到2库" OR (#x轴1库高速正转回工作位 AND (#Z轴编码器实时值 <= #X轴提前运行编码值)) OR #上砖X轴快速移动2库 OR (#"上砖X轴高速正转1库-待命位" AND (#Z轴编码器实时值 <= #X轴提前运行编码值))) AND #设备启动标志位 AND #机械手手自动标志 AND NOT #设备报警标志位) OR (#手动X轴2库移动 AND #急停按钮 AND (#Z轴编码器实时值 <= #Z轴待命位置编码值范围) AND #Z轴原点接近 AND NOT #z轴上升 AND NOT #z轴下降) OR (#复位X轴经1库原点后回原位 AND NOT #设备报警标志位 AND #Z轴原点接近 AND (#Z轴编码器实时值 <= #Z轴待命位置编码值范围) AND NOT #z轴上升 AND NOT #z轴下降)) AND NOT #x轴1库反转;
END_REGION

REGION Network 102: 输出 X轴反转高速 待命位置-----1库位置
   RUNG wire#powerrail
      Contact( #x轴2库高速反转回工作位 )
      { S7_Templates := "SrcType := DInt" } LE_Contact(in1 := #Z轴编码器实时值, in2 := #X轴提前运行编码值)
      wire#w1
      Contact( #设备启动标志位 )
      Contact( #机械手手自动标志 )
      I_Contact( #设备报警标志位 )
      wire#w2
      I_Contact( #x轴2库正转 )
      Coil( #x轴1库反转 )
   END_RUNG
   RUNG wire#powerrail
      Contact( #"X轴高速反转-待命位到1库" )
   END_RUNG wire#w1
   RUNG wire#powerrail
      Contact( #上砖X轴快速移动1库 )
   END_RUNG wire#w1
   RUNG wire#powerrail
      Contact( #"上砖X轴高速反转2库-待命位" )
      { S7_Templates := "SrcType := DInt" } LE_Contact(in1 := #Z轴编码器实时值, in2 := #X轴提前运行编码值)
   END_RUNG wire#w1
   RUNG wire#powerrail
      Contact( #手动X轴1库移动 )
      Contact( #急停按钮 )
      { S7_Templates := "SrcType := DInt" } LE_Contact(in1 := #Z轴编码器实时值, in2 := #Z轴待命位置编码值范围)
      Contact( #Z轴原点接近 )
      I_Contact( #z轴上升 )
      I_Contact( #z轴下降 )
   END_RUNG wire#w2
   RUNG wire#powerrail
      Contact( #复位X轴回原位 )
      I_Contact( #设备报警标志位 )
      Contact( #Z轴原点接近 )
      { S7_Templates := "SrcType := DInt" } LE_Contact(in1 := #Z轴编码器实时值, in2 := #Z轴待命位置编码值范围)
      I_Contact( #z轴上升 )
      I_Contact( #z轴下降 )
   END_RUNG wire#w2
   // the same network as SCL:
   #x轴1库反转 := ((((#x轴2库高速反转回工作位 AND (#Z轴编码器实时值 <= #X轴提前运行编码值)) OR #"X轴高速反转-待命位到1库" OR #上砖X轴快速移动1库 OR (#"上砖X轴高速反转2库-待命位" AND (#Z轴编码器实时值 <= #X轴提前运行编码值))) AND #设备启动标志位 AND #机械手手自动标志 AND NOT #设备报警标志位) OR (#手动X轴1库移动 AND #急停按钮 AND (#Z轴编码器实时值 <= #Z轴待命位置编码值范围) AND #Z轴原点接近 AND NOT #z轴上升 AND NOT #z轴下降) OR (#复位X轴回原位 AND NOT #设备报警标志位 AND #Z轴原点接近 AND (#Z轴编码器实时值 <= #Z轴待命位置编码值范围) AND NOT #z轴上升 AND NOT #z轴下降)) AND NOT #x轴2库正转;
END_REGION

REGION Network 103: 输出 x轴低速输出
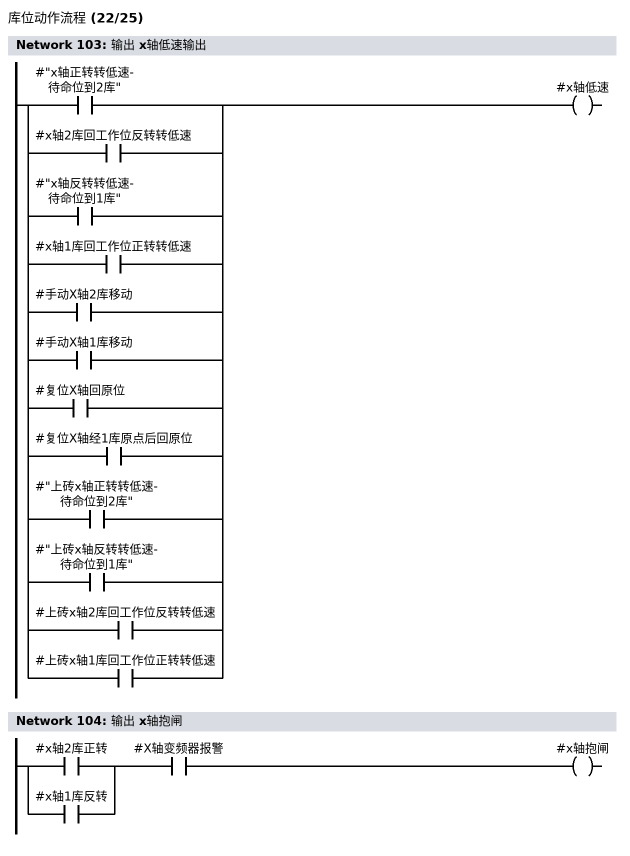
   RUNG wire#powerrail
      Contact( #"x轴正转转低速-待命位到2库" )
      wire#w1
      Coil( #x轴低速 )
   END_RUNG
   RUNG wire#powerrail
      Contact( #x轴2库回工作位反转转低速 )
   END_RUNG wire#w1
   RUNG wire#powerrail
      Contact( #"x轴反转转低速-待命位到1库" )
   END_RUNG wire#w1
   RUNG wire#powerrail
      Contact( #x轴1库回工作位正转转低速 )
   END_RUNG wire#w1
   RUNG wire#powerrail
      Contact( #手动X轴2库移动 )
   END_RUNG wire#w1
   RUNG wire#powerrail
      Contact( #手动X轴1库移动 )
   END_RUNG wire#w1
   RUNG wire#powerrail
      Contact( #复位X轴回原位 )
   END_RUNG wire#w1
   RUNG wire#powerrail
      Contact( #复位X轴经1库原点后回原位 )
   END_RUNG wire#w1
   RUNG wire#powerrail
      Contact( #"上砖x轴正转转低速-待命位到2库" )
   END_RUNG wire#w1
   RUNG wire#powerrail
      Contact( #"上砖x轴反转转低速-待命位到1库" )
   END_RUNG wire#w1
   RUNG wire#powerrail
      Contact( #上砖x轴2库回工作位反转转低速 )
   END_RUNG wire#w1
   RUNG wire#powerrail
      Contact( #上砖x轴1库回工作位正转转低速 )
   END_RUNG wire#w1
   // the same network as SCL:
   #x轴低速 := #"x轴正转转低速-待命位到2库" OR #x轴2库回工作位反转转低速 OR #"x轴反转转低速-待命位到1库" OR #x轴1库回工作位正转转低速 OR #手动X轴2库移动 OR #手动X轴1库移动 OR #复位X轴回原位 OR #复位X轴经1库原点后回原位 OR #"上砖x轴正转转低速-待命位到2库" OR #"上砖x轴反转转低速-待命位到1库" OR #上砖x轴2库回工作位反转转低速 OR #上砖x轴1库回工作位正转转低速;
END_REGION

REGION Network 104: 输出 x轴抱闸
   RUNG wire#powerrail
      Contact( #x轴2库正转 )
      wire#w1
      Contact( #X轴变频器报警 )
      Coil( #x轴抱闸 )
   END_RUNG
   RUNG wire#powerrail
      Contact( #x轴1库反转 )
   END_RUNG wire#w1
   // the same network as SCL:
   #x轴抱闸 := (#x轴2库正转 OR #x轴1库反转) AND #X轴变频器报警;
END_REGION

REGION Network 105: 输出 W伺服启动
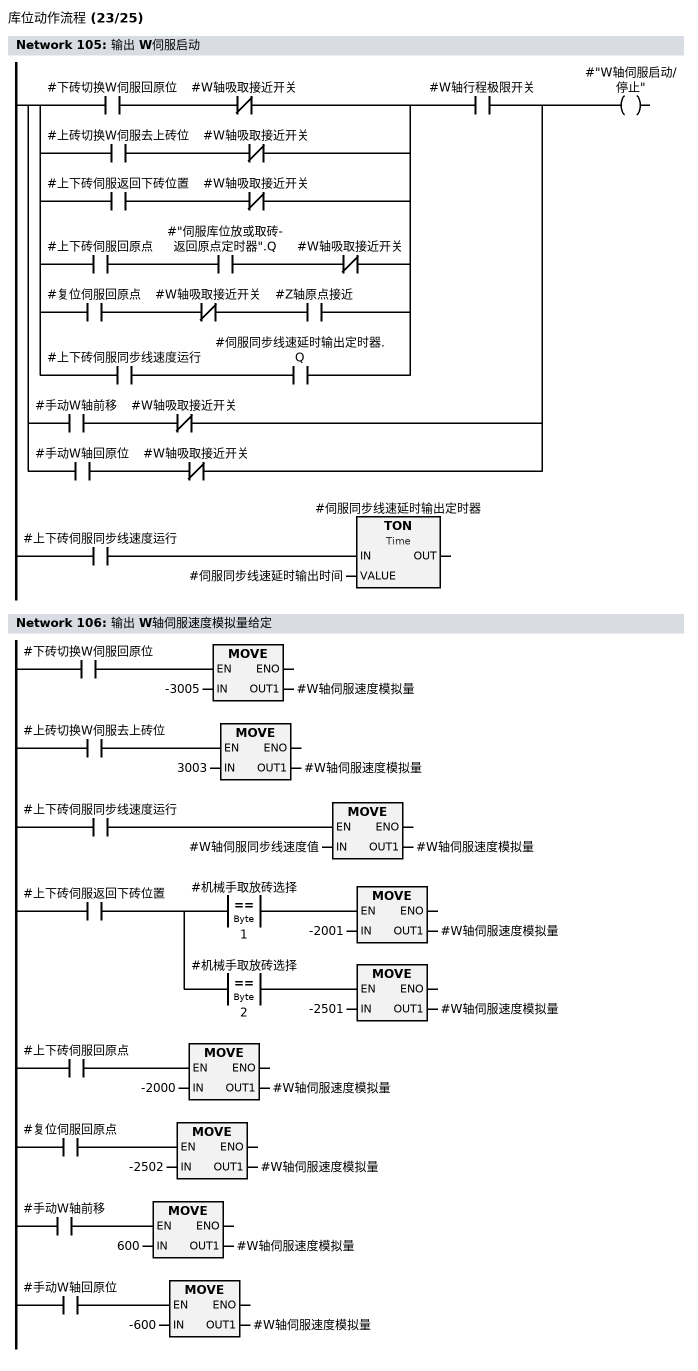
   #"W轴伺服启动/停止" := (((#下砖切换W伺服回原位 AND NOT #W轴吸取接近开关) OR (#上砖切换W伺服去上砖位 AND NOT #W轴吸取接近开关) OR (#上下砖伺服返回下砖位置 AND NOT #W轴吸取接近开关) OR (#上下砖伺服回原点 AND #"伺服库位放或取砖-返回原点定时器".Q AND NOT #W轴吸取接近开关) OR (#复位伺服回原点 AND NOT #W轴吸取接近开关 AND #Z轴原点接近) OR (#上下砖伺服同步线速度运行 AND #伺服同步线速延时输出定时器.Q)) AND #W轴行程极限开关) OR (#手动W轴前移 AND NOT #W轴吸取接近开关) OR (#手动W轴回原位 AND NOT #W轴吸取接近开关);
   #伺服同步线速延时输出定时器.TON(IN := #上下砖伺服同步线速度运行, PT := #伺服同步线速延时输出时间);   // TON coil
END_REGION

REGION Network 106: 输出 W轴伺服速度模拟量给定
   RUNG wire#powerrail
      Contact( #下砖切换W伺服回原位 )
      Move(in := -3005, out1 => #W轴伺服速度模拟量)
   END_RUNG
   RUNG wire#powerrail
      Contact( #上砖切换W伺服去上砖位 )
      Move(in := 3003, out1 => #W轴伺服速度模拟量)
   END_RUNG
   RUNG wire#powerrail
      Contact( #上下砖伺服同步线速度运行 )
      Move(in := #W轴伺服同步线速度值, out1 => #W轴伺服速度模拟量)
   END_RUNG
   RUNG wire#powerrail
      Contact( #上下砖伺服返回下砖位置 )
      wire#w1
      { S7_Templates := "SrcType := Byte" } EQ_Contact(in1 := #机械手取放砖选择, in2 := 1)
      Move(in := -2001, out1 => #W轴伺服速度模拟量)
   END_RUNG
   RUNG wire#w1
      { S7_Templates := "SrcType := Byte" } EQ_Contact(in1 := #机械手取放砖选择, in2 := 2)
      Move(in := -2501, out1 => #W轴伺服速度模拟量)
   END_RUNG
   RUNG wire#powerrail
      Contact( #上下砖伺服回原点 )
      Move(in := -2000, out1 => #W轴伺服速度模拟量)
   END_RUNG
   RUNG wire#powerrail
      Contact( #复位伺服回原点 )
      Move(in := -2502, out1 => #W轴伺服速度模拟量)
   END_RUNG
   RUNG wire#powerrail
      Contact( #手动W轴前移 )
      Move(in := 600, out1 => #W轴伺服速度模拟量)
   END_RUNG
   RUNG wire#powerrail
      Contact( #手动W轴回原位 )
      Move(in := -600, out1 => #W轴伺服速度模拟量)
   END_RUNG
   // the same network as SCL:
   IF #下砖切换W伺服回原位 THEN #W轴伺服速度模拟量 := -3005; END_IF;
   IF #上砖切换W伺服去上砖位 THEN #W轴伺服速度模拟量 := 3003; END_IF;
   IF #上下砖伺服同步线速度运行 THEN #W轴伺服速度模拟量 := #W轴伺服同步线速度值; END_IF;
   IF #上下砖伺服返回下砖位置 AND (#机械手取放砖选择 = 1) THEN #W轴伺服速度模拟量 := -2001; END_IF;
   IF #上下砖伺服返回下砖位置 AND (#机械手取放砖选择 = 2) THEN #W轴伺服速度模拟量 := -2501; END_IF;
   IF #上下砖伺服回原点 THEN #W轴伺服速度模拟量 := -2000; END_IF;
   IF #复位伺服回原点 THEN #W轴伺服速度模拟量 := -2502; END_IF;
   IF #手动W轴前移 THEN #W轴伺服速度模拟量 := 600; END_IF;
   IF #手动W轴回原位 THEN #W轴伺服速度模拟量 := -600; END_IF;
END_REGION

REGION Network 107: 输出 库位按钮指示灯
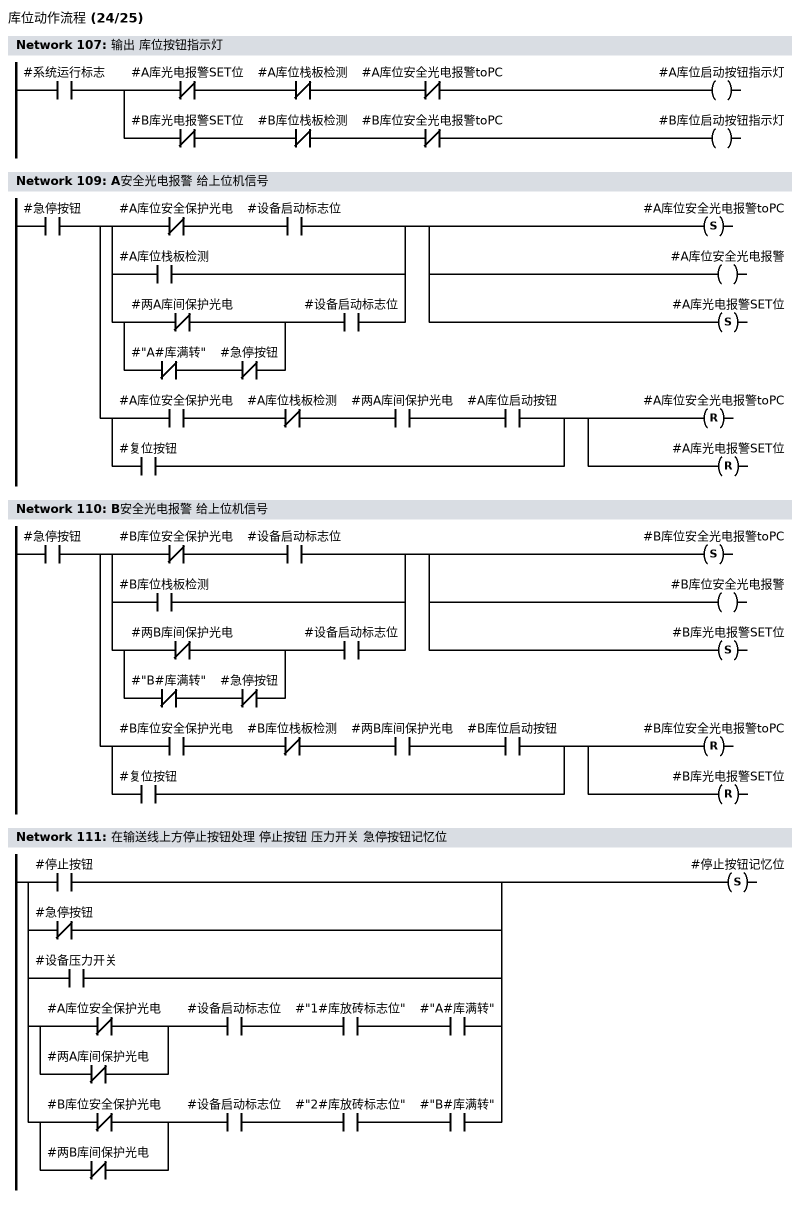
   RUNG wire#powerrail
      Contact( #系统运行标志 )
      wire#w1
      I_Contact( #A库光电报警SET位 )
      I_Contact( #A库位栈板检测 )
      I_Contact( #A库位安全光电报警toPC )
      Coil( #A库位启动按钮指示灯 )
   END_RUNG
   RUNG wire#w1
      I_Contact( #B库光电报警SET位 )
      I_Contact( #B库位栈板检测 )
      I_Contact( #B库位安全光电报警toPC )
      Coil( #B库位启动按钮指示灯 )
   END_RUNG
   // the same network as SCL:
   #A库位启动按钮指示灯 := #系统运行标志 AND NOT #A库光电报警SET位 AND NOT #A库位栈板检测 AND NOT #A库位安全光电报警toPC;
   #B库位启动按钮指示灯 := #系统运行标志 AND NOT #B库光电报警SET位 AND NOT #B库位栈板检测 AND NOT #B库位安全光电报警toPC;
END_REGION

REGION Network 108: 特殊故障处理
END_REGION

REGION Network 109: A安全光电报警 给上位机信号
   RUNG wire#powerrail
      Contact( #急停按钮 )
      wire#w1
      I_Contact( #A库位安全保护光电 )
      Contact( #设备启动标志位 )
      wire#w2
      S_Coil( #A库位安全光电报警toPC )
   END_RUNG
   RUNG wire#w1
      Contact( #A库位栈板检测 )
   END_RUNG wire#w2
   RUNG wire#w1
      I_Contact( #两A库间保护光电 )
      wire#w3
      Contact( #设备启动标志位 )
   END_RUNG wire#w2
   RUNG wire#w1
      I_Contact( #"A#库满转" )
      I_Contact( #急停按钮 )
   END_RUNG wire#w3
   RUNG wire#w2
      Coil( #A库位安全光电报警 )
   END_RUNG
   RUNG wire#w2
      S_Coil( #A库光电报警SET位 )
   END_RUNG
   RUNG wire#w1
      Contact( #A库位安全保护光电 )
      I_Contact( #A库位栈板检测 )
      Contact( #两A库间保护光电 )
      Contact( #A库位启动按钮 )
      wire#w4
      R_Coil( #A库位安全光电报警toPC )
   END_RUNG
   RUNG wire#w1
      Contact( #复位按钮 )
   END_RUNG wire#w4
   RUNG wire#w4
      R_Coil( #A库光电报警SET位 )
   END_RUNG
   // the same network as SCL:
   #_w1 := #急停按钮 AND ((NOT #A库位安全保护光电 AND #设备启动标志位) OR #A库位栈板检测 OR ((NOT #两A库间保护光电 OR (NOT #"A#库满转" AND NOT #急停按钮)) AND #设备启动标志位));
   IF #_w1 THEN #A库位安全光电报警toPC := TRUE; END_IF;
   #A库位安全光电报警 := #_w1;
   IF #_w1 THEN #A库光电报警SET位 := TRUE; END_IF;
   IF #急停按钮 AND ((#A库位安全保护光电 AND NOT #A库位栈板检测 AND #两A库间保护光电 AND #A库位启动按钮) OR #复位按钮) THEN
       #A库位安全光电报警toPC := FALSE;
       #A库光电报警SET位 := FALSE;
   END_IF;
END_REGION

REGION Network 110: B安全光电报警 给上位机信号
   RUNG wire#powerrail
      Contact( #急停按钮 )
      wire#w1
      I_Contact( #B库位安全保护光电 )
      Contact( #设备启动标志位 )
      wire#w2
      S_Coil( #B库位安全光电报警toPC )
   END_RUNG
   RUNG wire#w1
      Contact( #B库位栈板检测 )
   END_RUNG wire#w2
   RUNG wire#w1
      I_Contact( #两B库间保护光电 )
      wire#w3
      Contact( #设备启动标志位 )
   END_RUNG wire#w2
   RUNG wire#w1
      I_Contact( #"B#库满转" )
      I_Contact( #急停按钮 )
   END_RUNG wire#w3
   RUNG wire#w2
      Coil( #B库位安全光电报警 )
   END_RUNG
   RUNG wire#w2
      S_Coil( #B库光电报警SET位 )
   END_RUNG
   RUNG wire#w1
      Contact( #B库位安全保护光电 )
      I_Contact( #B库位栈板检测 )
      Contact( #两B库间保护光电 )
      Contact( #B库位启动按钮 )
      wire#w4
      R_Coil( #B库位安全光电报警toPC )
   END_RUNG
   RUNG wire#w1
      Contact( #复位按钮 )
   END_RUNG wire#w4
   RUNG wire#w4
      R_Coil( #B库光电报警SET位 )
   END_RUNG
   // the same network as SCL:
   #_w1 := #急停按钮 AND ((NOT #B库位安全保护光电 AND #设备启动标志位) OR #B库位栈板检测 OR ((NOT #两B库间保护光电 OR (NOT #"B#库满转" AND NOT #急停按钮)) AND #设备启动标志位));
   IF #_w1 THEN #B库位安全光电报警toPC := TRUE; END_IF;
   #B库位安全光电报警 := #_w1;
   IF #_w1 THEN #B库光电报警SET位 := TRUE; END_IF;
   IF #急停按钮 AND ((#B库位安全保护光电 AND NOT #B库位栈板检测 AND #两B库间保护光电 AND #B库位启动按钮) OR #复位按钮) THEN
       #B库位安全光电报警toPC := FALSE;
       #B库光电报警SET位 := FALSE;
   END_IF;
END_REGION

REGION Network 111: 在输送线上方停止按钮处理 停止按钮 压力开关 急停按钮记忆位
   RUNG wire#powerrail
      Contact( #停止按钮 )
      wire#w1
      S_Coil( #停止按钮记忆位 )
   END_RUNG
   RUNG wire#powerrail
      I_Contact( #急停按钮 )
   END_RUNG wire#w1
   RUNG wire#powerrail
      Contact( #设备压力开关 )
   END_RUNG wire#w1
   RUNG wire#powerrail
      I_Contact( #A库位安全保护光电 )
      wire#w2
      Contact( #设备启动标志位 )
      Contact( #"1#库放砖标志位" )
      Contact( #"A#库满转" )
   END_RUNG wire#w1
   RUNG wire#powerrail
      I_Contact( #两A库间保护光电 )
   END_RUNG wire#w2
   RUNG wire#powerrail
      I_Contact( #B库位安全保护光电 )
      wire#w3
      Contact( #设备启动标志位 )
      Contact( #"2#库放砖标志位" )
      Contact( #"B#库满转" )
   END_RUNG wire#w1
   RUNG wire#powerrail
      I_Contact( #两B库间保护光电 )
   END_RUNG wire#w3
   // the same network as SCL:
   IF #停止按钮 OR NOT #急停按钮 OR #设备压力开关 OR ((NOT #A库位安全保护光电 OR NOT #两A库间保护光电) AND #设备启动标志位 AND #"1#库放砖标志位" AND #"A#库满转") OR ((NOT #B库位安全保护光电 OR NOT #两B库间保护光电) AND #设备启动标志位 AND #"2#库放砖标志位" AND #"B#库满转") THEN
       #停止按钮记忆位 := TRUE;
   END_IF;
END_REGION

REGION Network 112: 在输送线上方停止按钮处理 停止按钮标志位
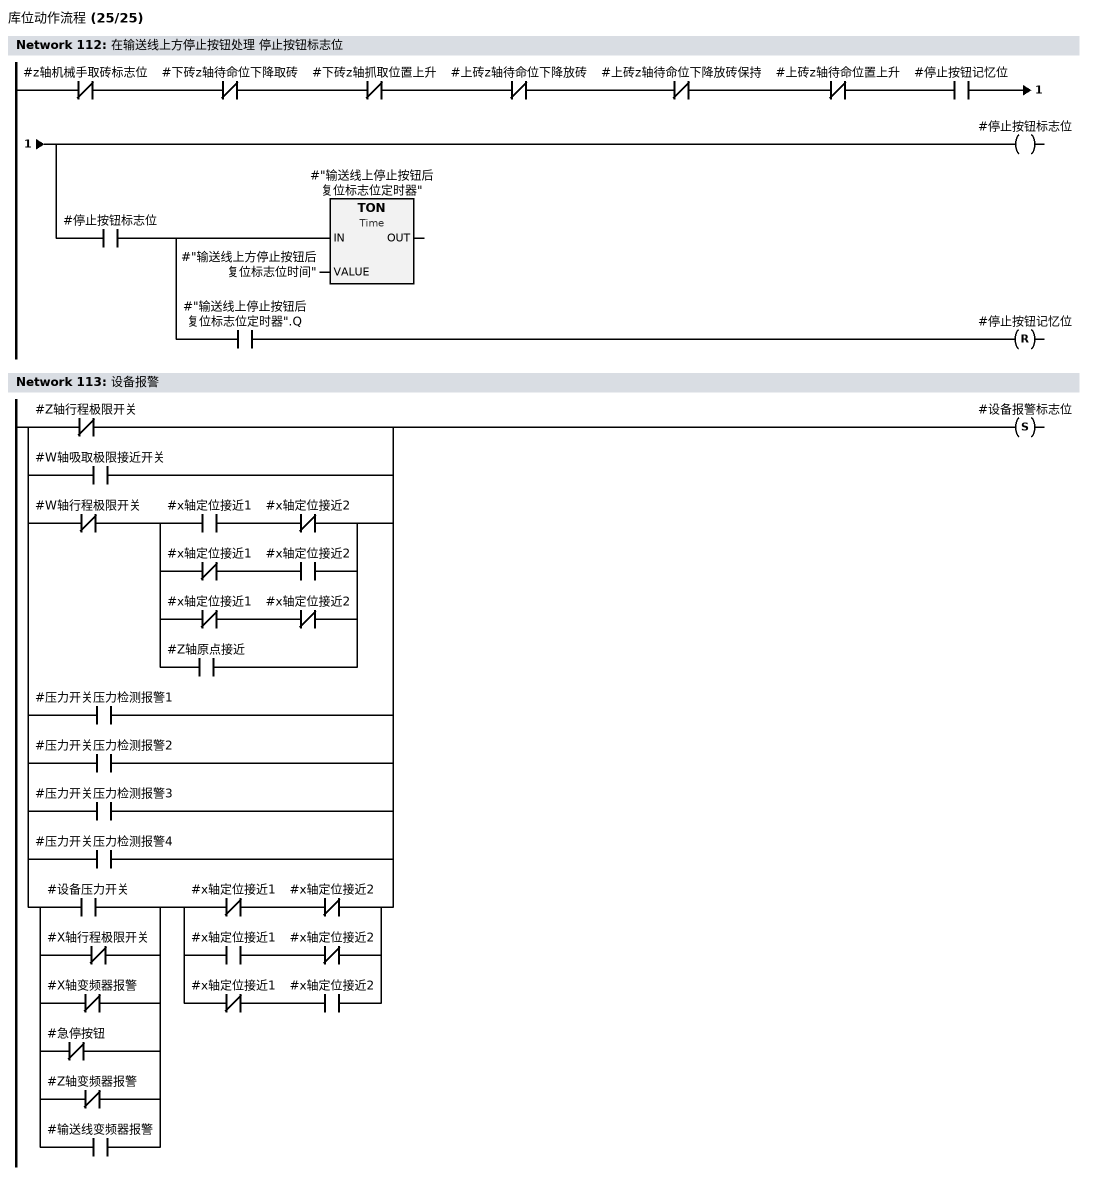
   #停止按钮标志位 := NOT #z轴机械手取砖标志位 AND NOT #下砖z轴待命位下降取砖 AND NOT #下砖z轴抓取位置上升 AND NOT #上砖z轴待命位下降放砖 AND NOT #上砖z轴待命位下降放砖保持 AND NOT #上砖z轴待命位置上升 AND #停止按钮记忆位;
   #_w1 := #停止按钮标志位 AND #停止按钮标志位;
   #"输送线上停止按钮后 复位标志位定时器".TON(IN := #_w1, PT := #"输送线上方停止按钮后 复位标志位时间");   // TON coil
   IF #_w1 AND #"输送线上停止按钮后 复位标志位定时器".Q THEN #停止按钮记忆位 := FALSE; END_IF;
END_REGION

REGION Network 113: 设备报警
   RUNG wire#powerrail
      I_Contact( #Z轴行程极限开关 )
      wire#w1
      S_Coil( #设备报警标志位 )
   END_RUNG
   RUNG wire#powerrail
      Contact( #W轴吸取极限接近开关 )
   END_RUNG wire#w1
   RUNG wire#powerrail
      I_Contact( #W轴行程极限开关 )
      wire#w2
      Contact( #x轴定位接近1 )
      I_Contact( #x轴定位接近2 )
   END_RUNG wire#w1
   RUNG wire#w2
      I_Contact( #x轴定位接近1 )
      Contact( #x轴定位接近2 )
   END_RUNG wire#w1
   RUNG wire#w2
      I_Contact( #x轴定位接近1 )
      I_Contact( #x轴定位接近2 )
   END_RUNG wire#w1
   RUNG wire#w2
      Contact( #Z轴原点接近 )
   END_RUNG wire#w1
   RUNG wire#powerrail
      Contact( #压力开关压力检测报警1 )
   END_RUNG wire#w1
   RUNG wire#powerrail
      Contact( #压力开关压力检测报警2 )
   END_RUNG wire#w1
   RUNG wire#powerrail
      Contact( #压力开关压力检测报警3 )
   END_RUNG wire#w1
   RUNG wire#powerrail
      Contact( #压力开关压力检测报警4 )
   END_RUNG wire#w1
   RUNG wire#powerrail
      Contact( #设备压力开关 )
      wire#w3
      I_Contact( #x轴定位接近1 )
      I_Contact( #x轴定位接近2 )
   END_RUNG wire#w1
   RUNG wire#powerrail
      I_Contact( #X轴行程极限开关 )
   END_RUNG wire#w3
   RUNG wire#powerrail
      I_Contact( #X轴变频器报警 )
   END_RUNG wire#w3
   RUNG wire#powerrail
      I_Contact( #急停按钮 )
   END_RUNG wire#w3
   RUNG wire#powerrail
      I_Contact( #Z轴变频器报警 )
   END_RUNG wire#w3
   RUNG wire#powerrail
      Contact( #输送线变频器报警 )
   END_RUNG wire#w3
   RUNG wire#w3
      Contact( #x轴定位接近1 )
      I_Contact( #x轴定位接近2 )
   END_RUNG wire#w1
   RUNG wire#w3
      I_Contact( #x轴定位接近1 )
      Contact( #x轴定位接近2 )
   END_RUNG wire#w1
   // the same network as SCL:
   IF NOT #Z轴行程极限开关 OR #W轴吸取极限接近开关 OR (NOT #W轴行程极限开关 AND ((#x轴定位接近1 AND NOT #x轴定位接近2) OR (NOT #x轴定位接近1 AND #x轴定位接近2) OR (NOT #x轴定位接近1 AND NOT #x轴定位接近2) OR #Z轴原点接近)) OR #压力开关压力检测报警1 OR #压力开关压力检测报警2 OR #压力开关压力检测报警3 OR #压力开关压力检测报警4 OR ((#设备压力开关 OR NOT #X轴行程极限开关 OR NOT #X轴变频器报警 OR NOT #急停按钮 OR NOT #Z轴变频器报警 OR #输送线变频器报警) AND ((NOT #x轴定位接近1 AND NOT #x轴定位接近2) OR (#x轴定位接近1 AND NOT #x轴定位接近2) OR (NOT #x轴定位接近1 AND #x轴定位接近2))) THEN
       #设备报警标志位 := TRUE;
   END_IF;
END_REGION
END_FUNCTION_BLOCK

FUNCTION_BLOCK "手动"   // FB2, LAD
{ S7_Optimized_Access := 'TRUE' }
VERSION : 0.1
   VAR_INPUT
      机械手手自动状态 : Bool;   // （1手动2自动）
      手动Z轴上下 : Byte;   // （1上2下）
      消音按钮 : Bool;
      限位开关Z轴 : Bool;
      Z轴正转下降 : Bool;
      Z轴原点光电 : Bool;
      Z轴反转上升 : Bool;
      急停按钮 : Bool;
      手动X轴左右 : Byte;
      限位开关X轴 : Bool;
      X轴2库正转 : Bool;
      X轴1库反转 : Bool;
      手动W轴前后 : Byte;
      限位开关W轴 : Bool;
      W轴速度写入值 : Int;
      W轴原位光电 : Bool;
      W轴停止光电 : Bool;
      手动吸盘打开关闭 : Bool;
      X轴定位开关1 : Bool;
      X轴定位开关2 : Bool;
   END_VAR
   VAR_OUTPUT
      手动Z轴下降 : Bool;
      手动Z轴上升 : Bool;
      手动X轴2库移动 : Bool;
      手动X轴1库移动 : Bool;
      手动W轴前移 : Bool;
      手动W轴后退 : Bool;
      手动真空阀打开 : Bool;
      手动真空阀关闭 : Bool;
   END_VAR
   VAR
      手动Z撞击限位下 : Bool;
      手动Z撞击限位上 : Bool;
      手动X撞击限位2库 : Bool;
      手动X撞击限位1库 : Bool;
      手动W撞击限位前 : Bool;
      手动W撞击限位后 : Bool;
   END_VAR
BEGIN

REGION Network 1: 机械手 Z轴下降
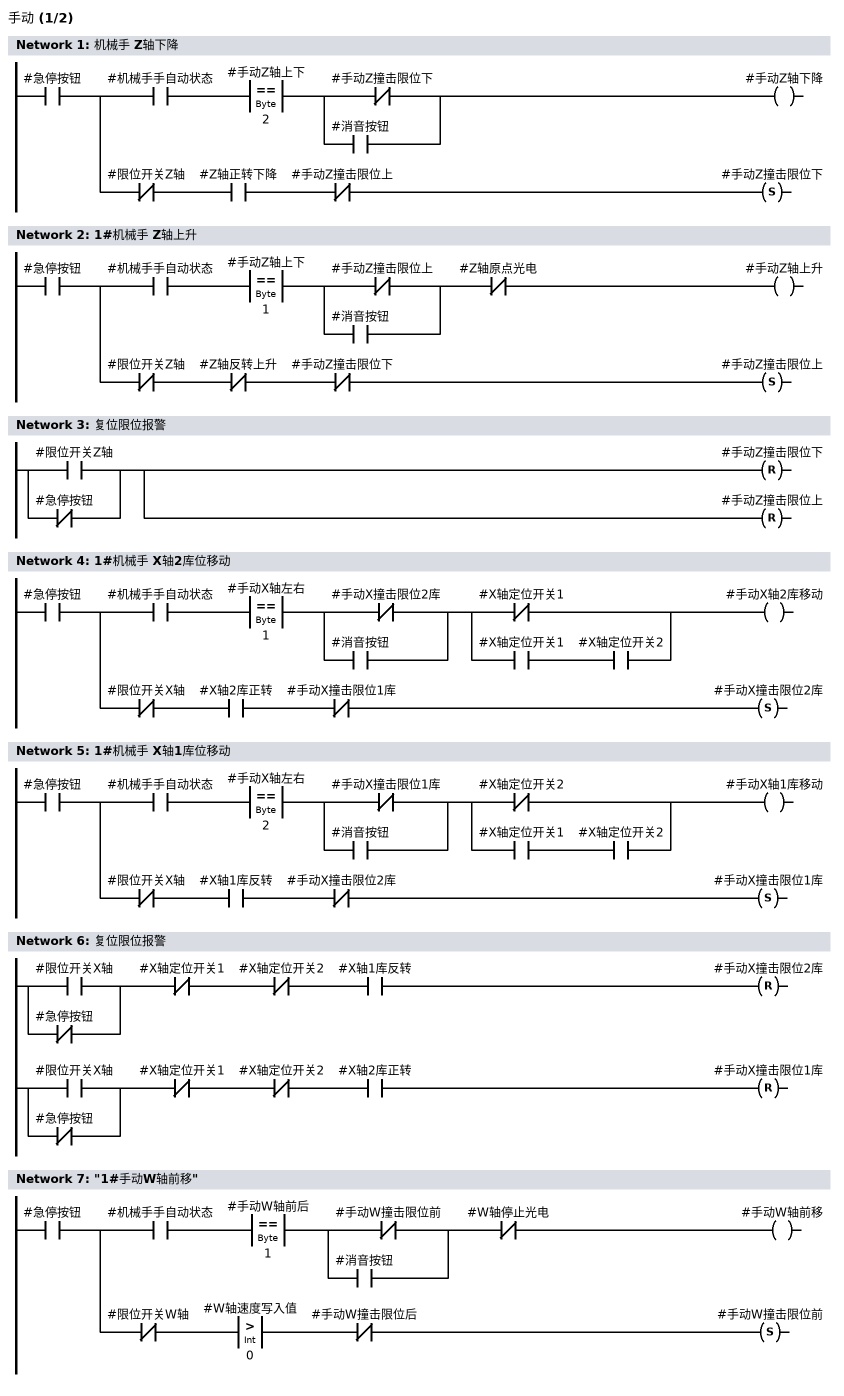
   RUNG wire#powerrail
      Contact( #急停按钮 )
      wire#w1
      Contact( #机械手手自动状态 )
      { S7_Templates := "SrcType := Byte" } EQ_Contact(in1 := #手动Z轴上下, in2 := 2)
      wire#w2
      I_Contact( #手动Z撞击限位下 )
      wire#w3
      Coil( #手动Z轴下降 )
   END_RUNG
   RUNG wire#w2
      Contact( #消音按钮 )
   END_RUNG wire#w3
   RUNG wire#w1
      I_Contact( #限位开关Z轴 )
      Contact( #Z轴正转下降 )
      I_Contact( #手动Z撞击限位上 )
      S_Coil( #手动Z撞击限位下 )
   END_RUNG
   // the same network as SCL:
   #手动Z轴下降 := #急停按钮 AND #机械手手自动状态 AND (#手动Z轴上下 = 2) AND (NOT #手动Z撞击限位下 OR #消音按钮);
   IF #急停按钮 AND NOT #限位开关Z轴 AND #Z轴正转下降 AND NOT #手动Z撞击限位上 THEN #手动Z撞击限位下 := TRUE; END_IF;
END_REGION

REGION Network 2: 1#机械手 Z轴上升
   RUNG wire#powerrail
      Contact( #急停按钮 )
      wire#w1
      Contact( #机械手手自动状态 )
      { S7_Templates := "SrcType := Byte" } EQ_Contact(in1 := #手动Z轴上下, in2 := 1)
      wire#w2
      I_Contact( #手动Z撞击限位上 )
      wire#w3
      I_Contact( #Z轴原点光电 )
      Coil( #手动Z轴上升 )
   END_RUNG
   RUNG wire#w2
      Contact( #消音按钮 )
   END_RUNG wire#w3
   RUNG wire#w1
      I_Contact( #限位开关Z轴 )
      I_Contact( #Z轴反转上升 )
      I_Contact( #手动Z撞击限位下 )
      S_Coil( #手动Z撞击限位上 )
   END_RUNG
   // the same network as SCL:
   #手动Z轴上升 := #急停按钮 AND #机械手手自动状态 AND (#手动Z轴上下 = 1) AND (NOT #手动Z撞击限位上 OR #消音按钮) AND NOT #Z轴原点光电;
   IF #急停按钮 AND NOT #限位开关Z轴 AND NOT #Z轴反转上升 AND NOT #手动Z撞击限位下 THEN #手动Z撞击限位上 := TRUE; END_IF;
END_REGION

REGION Network 3: 复位限位报警
   RUNG wire#powerrail
      Contact( #限位开关Z轴 )
      wire#w1
      R_Coil( #手动Z撞击限位下 )
   END_RUNG
   RUNG wire#powerrail
      I_Contact( #急停按钮 )
   END_RUNG wire#w1
   RUNG wire#w1
      R_Coil( #手动Z撞击限位上 )
   END_RUNG
   // the same network as SCL:
   IF #限位开关Z轴 OR NOT #急停按钮 THEN
       #手动Z撞击限位下 := FALSE;
       #手动Z撞击限位上 := FALSE;
   END_IF;
END_REGION

REGION Network 4: 1#机械手 X轴2库位移动
   RUNG wire#powerrail
      Contact( #急停按钮 )
      wire#w1
      Contact( #机械手手自动状态 )
      { S7_Templates := "SrcType := Byte" } EQ_Contact(in1 := #手动X轴左右, in2 := 1)
      wire#w2
      I_Contact( #手动X撞击限位2库 )
      wire#w3
      I_Contact( #X轴定位开关1 )
      wire#w4
      Coil( #手动X轴2库移动 )
   END_RUNG
   RUNG wire#w2
      Contact( #消音按钮 )
   END_RUNG wire#w3
   RUNG wire#w3
      Contact( #X轴定位开关1 )
      Contact( #X轴定位开关2 )
   END_RUNG wire#w4
   RUNG wire#w1
      I_Contact( #限位开关X轴 )
      Contact( #X轴2库正转 )
      I_Contact( #手动X撞击限位1库 )
      S_Coil( #手动X撞击限位2库 )
   END_RUNG
   // the same network as SCL:
   #手动X轴2库移动 := #急停按钮 AND #机械手手自动状态 AND (#手动X轴左右 = 1) AND (NOT #手动X撞击限位2库 OR #消音按钮) AND (NOT #X轴定位开关1 OR (#X轴定位开关1 AND #X轴定位开关2));
   IF #急停按钮 AND NOT #限位开关X轴 AND #X轴2库正转 AND NOT #手动X撞击限位1库 THEN #手动X撞击限位2库 := TRUE; END_IF;
END_REGION

REGION Network 5: 1#机械手 X轴1库位移动
   RUNG wire#powerrail
      Contact( #急停按钮 )
      wire#w1
      Contact( #机械手手自动状态 )
      { S7_Templates := "SrcType := Byte" } EQ_Contact(in1 := #手动X轴左右, in2 := 2)
      wire#w2
      I_Contact( #手动X撞击限位1库 )
      wire#w3
      I_Contact( #X轴定位开关2 )
      wire#w4
      Coil( #手动X轴1库移动 )
   END_RUNG
   RUNG wire#w2
      Contact( #消音按钮 )
   END_RUNG wire#w3
   RUNG wire#w3
      Contact( #X轴定位开关1 )
      Contact( #X轴定位开关2 )
   END_RUNG wire#w4
   RUNG wire#w1
      I_Contact( #限位开关X轴 )
      Contact( #X轴1库反转 )
      I_Contact( #手动X撞击限位2库 )
      S_Coil( #手动X撞击限位1库 )
   END_RUNG
   // the same network as SCL:
   #手动X轴1库移动 := #急停按钮 AND #机械手手自动状态 AND (#手动X轴左右 = 2) AND (NOT #手动X撞击限位1库 OR #消音按钮) AND (NOT #X轴定位开关2 OR (#X轴定位开关1 AND #X轴定位开关2));
   IF #急停按钮 AND NOT #限位开关X轴 AND #X轴1库反转 AND NOT #手动X撞击限位2库 THEN #手动X撞击限位1库 := TRUE; END_IF;
END_REGION

REGION Network 6: 复位限位报警
   RUNG wire#powerrail
      Contact( #限位开关X轴 )
      wire#w1
      I_Contact( #X轴定位开关1 )
      I_Contact( #X轴定位开关2 )
      Contact( #X轴1库反转 )
      R_Coil( #手动X撞击限位2库 )
   END_RUNG
   RUNG wire#powerrail
      I_Contact( #急停按钮 )
   END_RUNG wire#w1
   RUNG wire#powerrail
      Contact( #限位开关X轴 )
      wire#w2
      I_Contact( #X轴定位开关1 )
      I_Contact( #X轴定位开关2 )
      Contact( #X轴2库正转 )
      R_Coil( #手动X撞击限位1库 )
   END_RUNG
   RUNG wire#powerrail
      I_Contact( #急停按钮 )
   END_RUNG wire#w2
   // the same network as SCL:
   IF (#限位开关X轴 OR NOT #急停按钮) AND NOT #X轴定位开关1 AND NOT #X轴定位开关2 AND #X轴1库反转 THEN #手动X撞击限位2库 := FALSE; END_IF;
   IF (#限位开关X轴 OR NOT #急停按钮) AND NOT #X轴定位开关1 AND NOT #X轴定位开关2 AND #X轴2库正转 THEN #手动X撞击限位1库 := FALSE; END_IF;
END_REGION

REGION Network 7: "1#手动W轴前移"
   RUNG wire#powerrail
      Contact( #急停按钮 )
      wire#w1
      Contact( #机械手手自动状态 )
      { S7_Templates := "SrcType := Byte" } EQ_Contact(in1 := #手动W轴前后, in2 := 1)
      wire#w2
      I_Contact( #手动W撞击限位前 )
      wire#w3
      I_Contact( #W轴停止光电 )
      Coil( #手动W轴前移 )
   END_RUNG
   RUNG wire#w2
      Contact( #消音按钮 )
   END_RUNG wire#w3
   RUNG wire#w1
      I_Contact( #限位开关W轴 )
      { S7_Templates := "SrcType := Int" } GT_Contact(in1 := #W轴速度写入值, in2 := 0)
      I_Contact( #手动W撞击限位后 )
      S_Coil( #手动W撞击限位前 )
   END_RUNG
   // the same network as SCL:
   #手动W轴前移 := #急停按钮 AND #机械手手自动状态 AND (#手动W轴前后 = 1) AND (NOT #手动W撞击限位前 OR #消音按钮) AND NOT #W轴停止光电;
   IF #急停按钮 AND NOT #限位开关W轴 AND (#W轴速度写入值 > 0) AND NOT #手动W撞击限位后 THEN #手动W撞击限位前 := TRUE; END_IF;
END_REGION

REGION Network 8: "1#手动W轴回原位"
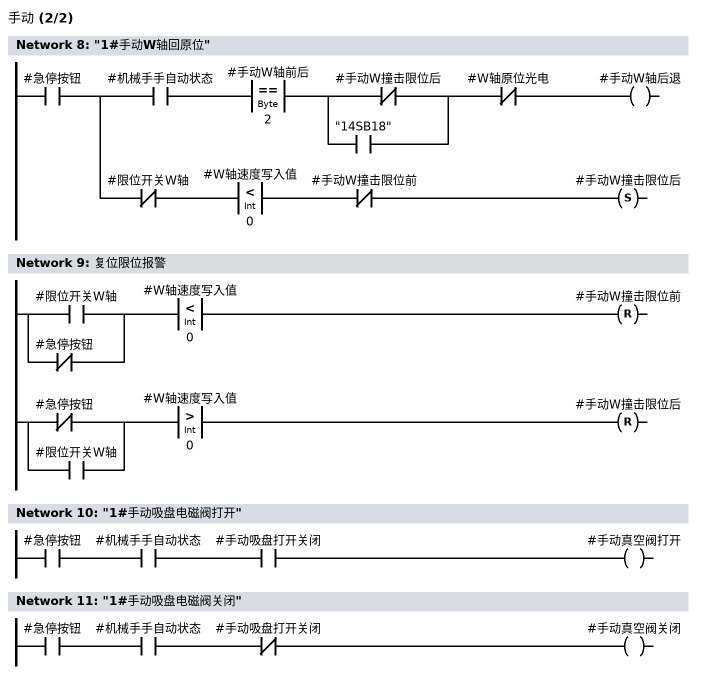
   RUNG wire#powerrail
      Contact( #急停按钮 )
      wire#w1
      Contact( #机械手手自动状态 )
      { S7_Templates := "SrcType := Byte" } EQ_Contact(in1 := #手动W轴前后, in2 := 2)
      wire#w2
      I_Contact( #手动W撞击限位后 )
      wire#w3
      I_Contact( #W轴原位光电 )
      Coil( #手动W轴后退 )
   END_RUNG
   RUNG wire#w2
      Contact( "14SB18" )
   END_RUNG wire#w3
   RUNG wire#w1
      I_Contact( #限位开关W轴 )
      { S7_Templates := "SrcType := Int" } LT_Contact(in1 := #W轴速度写入值, in2 := 0)
      I_Contact( #手动W撞击限位前 )
      S_Coil( #手动W撞击限位后 )
   END_RUNG
   // the same network as SCL:
   #手动W轴后退 := #急停按钮 AND #机械手手自动状态 AND (#手动W轴前后 = 2) AND (NOT #手动W撞击限位后 OR "14SB18") AND NOT #W轴原位光电;
   IF #急停按钮 AND NOT #限位开关W轴 AND (#W轴速度写入值 < 0) AND NOT #手动W撞击限位前 THEN #手动W撞击限位后 := TRUE; END_IF;
END_REGION

REGION Network 9: 复位限位报警
   RUNG wire#powerrail
      Contact( #限位开关W轴 )
      wire#w1
      { S7_Templates := "SrcType := Int" } LT_Contact(in1 := #W轴速度写入值, in2 := 0)
      R_Coil( #手动W撞击限位前 )
   END_RUNG
   RUNG wire#powerrail
      I_Contact( #急停按钮 )
   END_RUNG wire#w1
   RUNG wire#powerrail
      I_Contact( #急停按钮 )
      wire#w2
      { S7_Templates := "SrcType := Int" } GT_Contact(in1 := #W轴速度写入值, in2 := 0)
      R_Coil( #手动W撞击限位后 )
   END_RUNG
   RUNG wire#powerrail
      Contact( #限位开关W轴 )
   END_RUNG wire#w2
   // the same network as SCL:
   IF (#限位开关W轴 OR NOT #急停按钮) AND (#W轴速度写入值 < 0) THEN #手动W撞击限位前 := FALSE; END_IF;
   IF (NOT #急停按钮 OR #限位开关W轴) AND (#W轴速度写入值 > 0) THEN #手动W撞击限位后 := FALSE; END_IF;
END_REGION

REGION Network 10: "1#手动吸盘电磁阀打开"
   RUNG wire#powerrail
      Contact( #急停按钮 )
      Contact( #机械手手自动状态 )
      Contact( #手动吸盘打开关闭 )
      Coil( #手动真空阀打开 )
   END_RUNG
   // the same network as SCL:
   #手动真空阀打开 := #急停按钮 AND #机械手手自动状态 AND #手动吸盘打开关闭;
END_REGION

REGION Network 11: "1#手动吸盘电磁阀关闭"
   RUNG wire#powerrail
      Contact( #急停按钮 )
      Contact( #机械手手自动状态 )
      I_Contact( #手动吸盘打开关闭 )
      Coil( #手动真空阀关闭 )
   END_RUNG
   // the same network as SCL:
   #手动真空阀关闭 := #急停按钮 AND #机械手手自动状态 AND NOT #手动吸盘打开关闭;
END_REGION
END_FUNCTION_BLOCK

FUNCTION_BLOCK "PLC交换PC"   // FB3, LAD
{ S7_Optimized_Access := 'TRUE' }
VERSION : 0.1
   VAR_INPUT
      取上砖选择 : Byte;   // 1取砖2上砖
      "1#库位栈板光电" : Bool;
      "2#库位栈板光电" : Bool;
      定位光电1 : Bool;
      定位光电2 : Bool;
      W原点光电 : Bool;
      x轴限位开关 : Bool;
      z轴限位开关 : Bool;
      w轴限位开关 : Bool;
      吸盘极限光电 : Bool;
      "1#压力开关报警" : Bool;
      "2#压力开关报警" : Bool;
      "3#压力开关报警" : Bool;
      "4#压力开关报警" : Bool;
      "1#库位安全光电报警" : Bool;
      "2#库位安全光电报警" : Bool;
      X轴变频器报警 : Bool;
      Z轴变频器报警 : Bool;
      "1#库位启动按钮" : Bool;
      主控柜复位按钮 : Bool;
      机械手单独复位 : Bool;   // 1复位2完成
      "2#库位启动按钮" : Bool;
      机械手系统复位标志 : Bool;
      "1#启动绿灯" : Bool;
      "2#启动绿灯" : Bool;
      待命位置 : Bool;
      上下模式 : Byte;
      抓取方向 : Bool;
   END_VAR
   VAR_OUTPUT
      x轴限位报警输出 : Bool;
      z轴限位报警输出 : Bool;
      w轴限位报警输出 : Bool;
      吸盘极限光电报警输出 : Bool;
      "1#压力开关报警输出" : Bool;
      "2#压力开关报警输出" : Bool;
      "3#压力开关报警输出" : Bool;
      "4#压力开关报警输出" : Bool;
      "1#库位安全光电报警输出" : Bool;
      "2#库位安全光电报警输出" : Bool;
      X轴变频器报警输出 : Bool;
      Z轴变频器报警输出 : Bool;
      单独复位标志位输出 : Bool;
      机械手复位状态 : Byte;
      "1#库位状态" : Byte;
      "2#库位状态" : Byte;
   END_VAR
   VAR
      取砖转换后定时器 : IEC_TIMER;
      上砖转换后定时器 : IEC_TIMER;
      "1#启动按钮定时器" : IEC_TIMER;
      "1#启动按钮清除计数定时器" : IEC_TIMER;
      "1#报警后启动" : IEC_TIMER;
      "2#启动按钮定时器" : IEC_TIMER;
      "2#启动按钮清除计数定时器" : IEC_TIMER;
      "2#报警后启动" : IEC_TIMER;
      上下砖模式计时器 : IEC_TIMER;
      给复位指令计时器 : IEC_TIMER;
      P1 : Bool;
      P2 : Bool;
      P3 : Bool;
      P4 : Bool;
      P5 : Bool;
      P6 : Bool;
      "1#启动按钮保持" : Bool;
      "1#启动按钮清除计数保持" : Bool;
      "2#启动按钮保持" : Bool;
      "2#启动按钮清除计数保持" : Bool;
      "1#启动按钮计数中间" : Byte;
      "2#启动按钮计数中间" : Byte;
      机械手不动作记忆 : Bool;
   END_VAR
   VAR_TEMP   // added for the SCL form of the ladder/FBD networks
      _w1 : Bool;
      _w2 : Bool;
      _w3 : Bool;
      _w4 : Bool;
      _w5 : Bool;
      _w6 : Bool;
      _w7 : Bool;
      _w8 : Bool;
   END_VAR
BEGIN

REGION Network 1: 1#库位状态
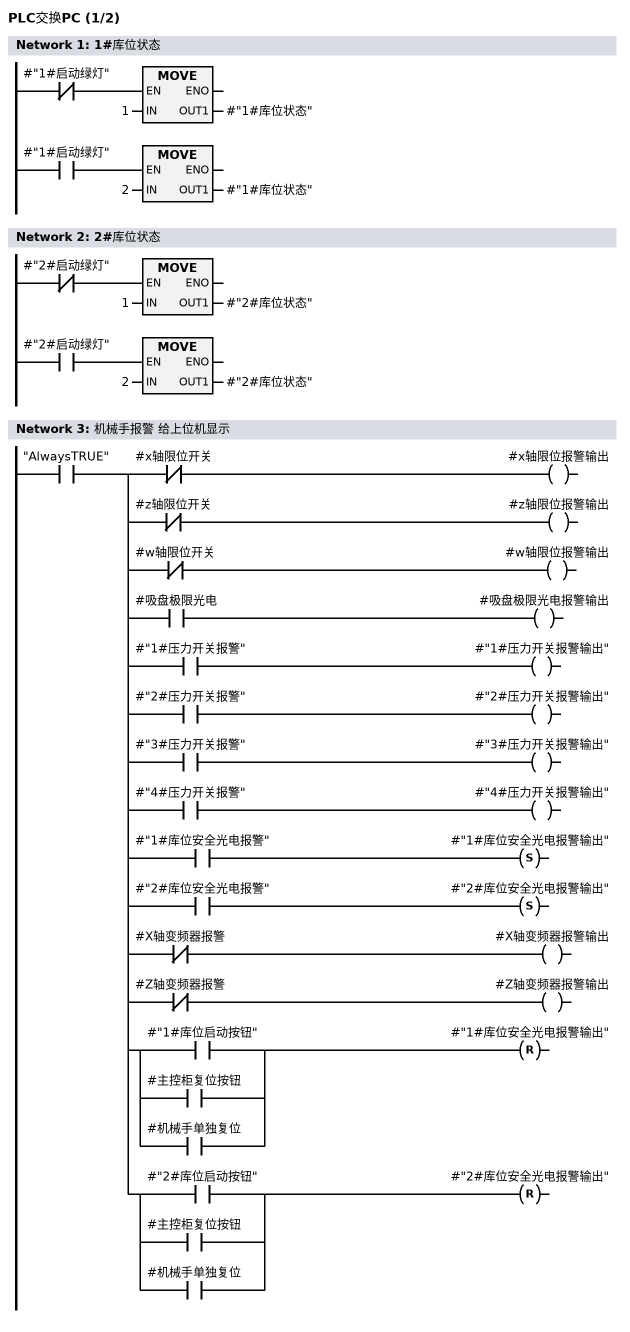
   RUNG wire#powerrail
      I_Contact( #"1#启动绿灯" )
      Move(in := 1, out1 => #"1#库位状态")
   END_RUNG
   RUNG wire#powerrail
      Contact( #"1#启动绿灯" )
      Move(in := 2, out1 => #"1#库位状态")
   END_RUNG
   // the same network as SCL:
   IF NOT #"1#启动绿灯" THEN #"1#库位状态" := 1; END_IF;
   IF #"1#启动绿灯" THEN #"1#库位状态" := 2; END_IF;
END_REGION

REGION Network 2: 2#库位状态
   RUNG wire#powerrail
      I_Contact( #"2#启动绿灯" )
      Move(in := 1, out1 => #"2#库位状态")
   END_RUNG
   RUNG wire#powerrail
      Contact( #"2#启动绿灯" )
      Move(in := 2, out1 => #"2#库位状态")
   END_RUNG
   // the same network as SCL:
   IF NOT #"2#启动绿灯" THEN #"2#库位状态" := 1; END_IF;
   IF #"2#启动绿灯" THEN #"2#库位状态" := 2; END_IF;
END_REGION

REGION Network 3: 机械手报警 给上位机显示
   RUNG wire#powerrail
      Contact( "AlwaysTRUE" )
      wire#w1
      I_Contact( #x轴限位开关 )
      Coil( #x轴限位报警输出 )
   END_RUNG
   RUNG wire#w1
      I_Contact( #z轴限位开关 )
      Coil( #z轴限位报警输出 )
   END_RUNG
   RUNG wire#w1
      I_Contact( #w轴限位开关 )
      Coil( #w轴限位报警输出 )
   END_RUNG
   RUNG wire#w1
      Contact( #吸盘极限光电 )
      Coil( #吸盘极限光电报警输出 )
   END_RUNG
   RUNG wire#w1
      Contact( #"1#压力开关报警" )
      Coil( #"1#压力开关报警输出" )
   END_RUNG
   RUNG wire#w1
      Contact( #"2#压力开关报警" )
      Coil( #"2#压力开关报警输出" )
   END_RUNG
   RUNG wire#w1
      Contact( #"3#压力开关报警" )
      Coil( #"3#压力开关报警输出" )
   END_RUNG
   RUNG wire#w1
      Contact( #"4#压力开关报警" )
      Coil( #"4#压力开关报警输出" )
   END_RUNG
   RUNG wire#w1
      Contact( #"1#库位安全光电报警" )
      S_Coil( #"1#库位安全光电报警输出" )
   END_RUNG
   RUNG wire#w1
      Contact( #"2#库位安全光电报警" )
      S_Coil( #"2#库位安全光电报警输出" )
   END_RUNG
   RUNG wire#w1
      I_Contact( #X轴变频器报警 )
      Coil( #X轴变频器报警输出 )
   END_RUNG
   RUNG wire#w1
      I_Contact( #Z轴变频器报警 )
      Coil( #Z轴变频器报警输出 )
   END_RUNG
   RUNG wire#w1
      Contact( #"1#库位启动按钮" )
      wire#w2
      R_Coil( #"1#库位安全光电报警输出" )
   END_RUNG
   RUNG wire#w1
      Contact( #主控柜复位按钮 )
   END_RUNG wire#w2
   RUNG wire#w1
      Contact( #机械手单独复位 )
   END_RUNG wire#w2
   RUNG wire#w1
      Contact( #"2#库位启动按钮" )
      wire#w3
      R_Coil( #"2#库位安全光电报警输出" )
   END_RUNG
   RUNG wire#w1
      Contact( #主控柜复位按钮 )
   END_RUNG wire#w3
   RUNG wire#w1
      Contact( #机械手单独复位 )
   END_RUNG wire#w3
   // the same network as SCL:
   #x轴限位报警输出 := "AlwaysTRUE" AND NOT #x轴限位开关;
   #z轴限位报警输出 := "AlwaysTRUE" AND NOT #z轴限位开关;
   #w轴限位报警输出 := "AlwaysTRUE" AND NOT #w轴限位开关;
   #吸盘极限光电报警输出 := "AlwaysTRUE" AND #吸盘极限光电;
   #"1#压力开关报警输出" := "AlwaysTRUE" AND #"1#压力开关报警";
   #"2#压力开关报警输出" := "AlwaysTRUE" AND #"2#压力开关报警";
   #"3#压力开关报警输出" := "AlwaysTRUE" AND #"3#压力开关报警";
   #"4#压力开关报警输出" := "AlwaysTRUE" AND #"4#压力开关报警";
   IF "AlwaysTRUE" AND #"1#库位安全光电报警" THEN #"1#库位安全光电报警输出" := TRUE; END_IF;
   IF "AlwaysTRUE" AND #"2#库位安全光电报警" THEN #"2#库位安全光电报警输出" := TRUE; END_IF;
   #X轴变频器报警输出 := "AlwaysTRUE" AND NOT #X轴变频器报警;
   #Z轴变频器报警输出 := "AlwaysTRUE" AND NOT #Z轴变频器报警;
   IF "AlwaysTRUE" AND (#"1#库位启动按钮" OR #主控柜复位按钮 OR #机械手单独复位) THEN #"1#库位安全光电报警输出" := FALSE; END_IF;
   IF "AlwaysTRUE" AND (#"2#库位启动按钮" OR #主控柜复位按钮 OR #机械手单独复位) THEN #"2#库位安全光电报警输出" := FALSE; END_IF;
END_REGION

REGION Network 4: 上下砖模式 设备不动作 PLC处理判断
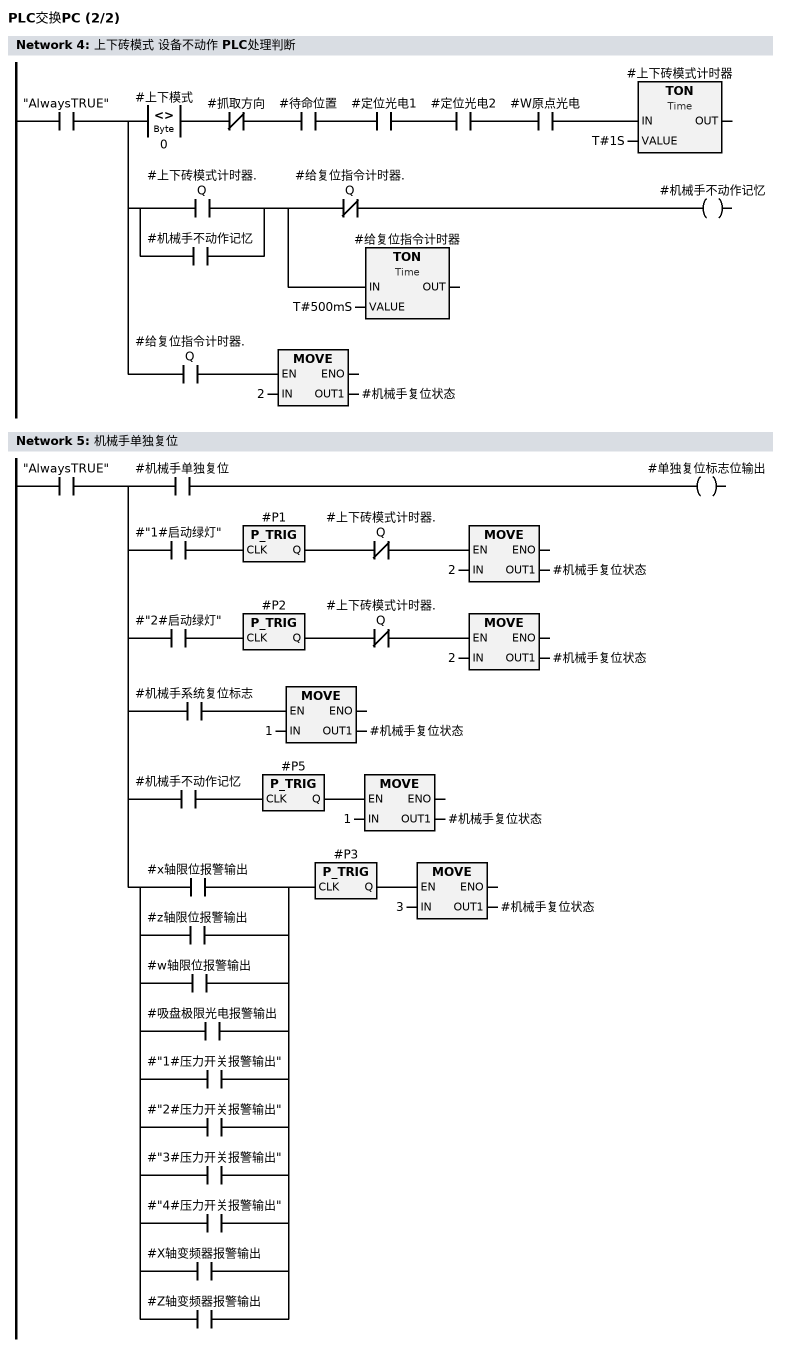
   #上下砖模式计时器.TON(IN := "AlwaysTRUE" AND (#上下模式 <> 0) AND NOT #抓取方向 AND #待命位置 AND #定位光电1 AND #定位光电2 AND #W原点光电, PT := T#1S);   // TON coil
   #_w1 := "AlwaysTRUE" AND (#上下砖模式计时器.Q OR #机械手不动作记忆);
   #机械手不动作记忆 := #_w1 AND NOT #给复位指令计时器.Q;
   #给复位指令计时器.TON(IN := #_w1, PT := T#500mS);   // TON coil
   IF "AlwaysTRUE" AND #给复位指令计时器.Q THEN #机械手复位状态 := 2; END_IF;
END_REGION

REGION Network 5: 机械手单独复位
   RUNG wire#powerrail
      Contact( "AlwaysTRUE" )
      wire#w1
      Contact( #机械手单独复位 )
      Coil( #单独复位标志位输出 )
   END_RUNG
   RUNG wire#w1
      Contact( #"1#启动绿灯" )
      P_Trig( #P1 )
      I_Contact( #上下砖模式计时器.Q )
      Move(in := 2, out1 => #机械手复位状态)
   END_RUNG
   RUNG wire#w1
      Contact( #"2#启动绿灯" )
      P_Trig( #P2 )
      I_Contact( #上下砖模式计时器.Q )
      Move(in := 2, out1 => #机械手复位状态)
   END_RUNG
   RUNG wire#w1
      Contact( #机械手系统复位标志 )
      Move(in := 1, out1 => #机械手复位状态)
   END_RUNG
   RUNG wire#w1
      Contact( #机械手不动作记忆 )
      P_Trig( #P5 )
      Move(in := 1, out1 => #机械手复位状态)
   END_RUNG
   RUNG wire#w1
      Contact( #x轴限位报警输出 )
      wire#w2
      P_Trig( #P3 )
      Move(in := 3, out1 => #机械手复位状态)
   END_RUNG
   RUNG wire#w1
      Contact( #z轴限位报警输出 )
   END_RUNG wire#w2
   RUNG wire#w1
      Contact( #w轴限位报警输出 )
   END_RUNG wire#w2
   RUNG wire#w1
      Contact( #吸盘极限光电报警输出 )
   END_RUNG wire#w2
   RUNG wire#w1
      Contact( #"1#压力开关报警输出" )
   END_RUNG wire#w2
   RUNG wire#w1
      Contact( #"2#压力开关报警输出" )
   END_RUNG wire#w2
   RUNG wire#w1
      Contact( #"3#压力开关报警输出" )
   END_RUNG wire#w2
   RUNG wire#w1
      Contact( #"4#压力开关报警输出" )
   END_RUNG wire#w2
   RUNG wire#w1
      Contact( #X轴变频器报警输出 )
   END_RUNG wire#w2
   RUNG wire#w1
      Contact( #Z轴变频器报警输出 )
   END_RUNG wire#w2
   // the same network as SCL:
   #单独复位标志位输出 := "AlwaysTRUE" AND #机械手单独复位;
   #_w1 := "AlwaysTRUE" AND #"1#启动绿灯";
   #_w2 := #_w1 AND NOT #P1;   // rising edge
   #P1 := #_w1;
   IF #_w2 AND NOT #上下砖模式计时器.Q THEN #机械手复位状态 := 2; END_IF;
   #_w3 := "AlwaysTRUE" AND #"2#启动绿灯";
   #_w4 := #_w3 AND NOT #P2;   // rising edge
   #P2 := #_w3;
   IF #_w4 AND NOT #上下砖模式计时器.Q THEN #机械手复位状态 := 2; END_IF;
   IF "AlwaysTRUE" AND #机械手系统复位标志 THEN #机械手复位状态 := 1; END_IF;
   #_w5 := "AlwaysTRUE" AND #机械手不动作记忆;
   #_w6 := #_w5 AND NOT #P5;   // rising edge
   #P5 := #_w5;
   IF #_w6 THEN #机械手复位状态 := 1; END_IF;
   #_w7 := "AlwaysTRUE" AND (#x轴限位报警输出 OR #z轴限位报警输出 OR #w轴限位报警输出 OR #吸盘极限光电报警输出 OR #"1#压力开关报警输出" OR #"2#压力开关报警输出" OR #"3#压力开关报警输出" OR #"4#压力开关报警输出" OR #X轴变频器报警输出 OR #Z轴变频器报警输出);
   #_w8 := #_w7 AND NOT #P3;   // rising edge
   #P3 := #_w7;
   IF #_w8 THEN #机械手复位状态 := 3; END_IF;
END_REGION
END_FUNCTION_BLOCK

FUNCTION "1#手" : Void   // FC11, LAD
{ S7_Optimized_Access := 'TRUE' }
VERSION : 0.1
   VAR_TEMP   // added for the SCL form of the ladder/FBD networks
      _w1 : Bool;
   END_VAR
BEGIN

REGION Network 1: 14前对中气缸
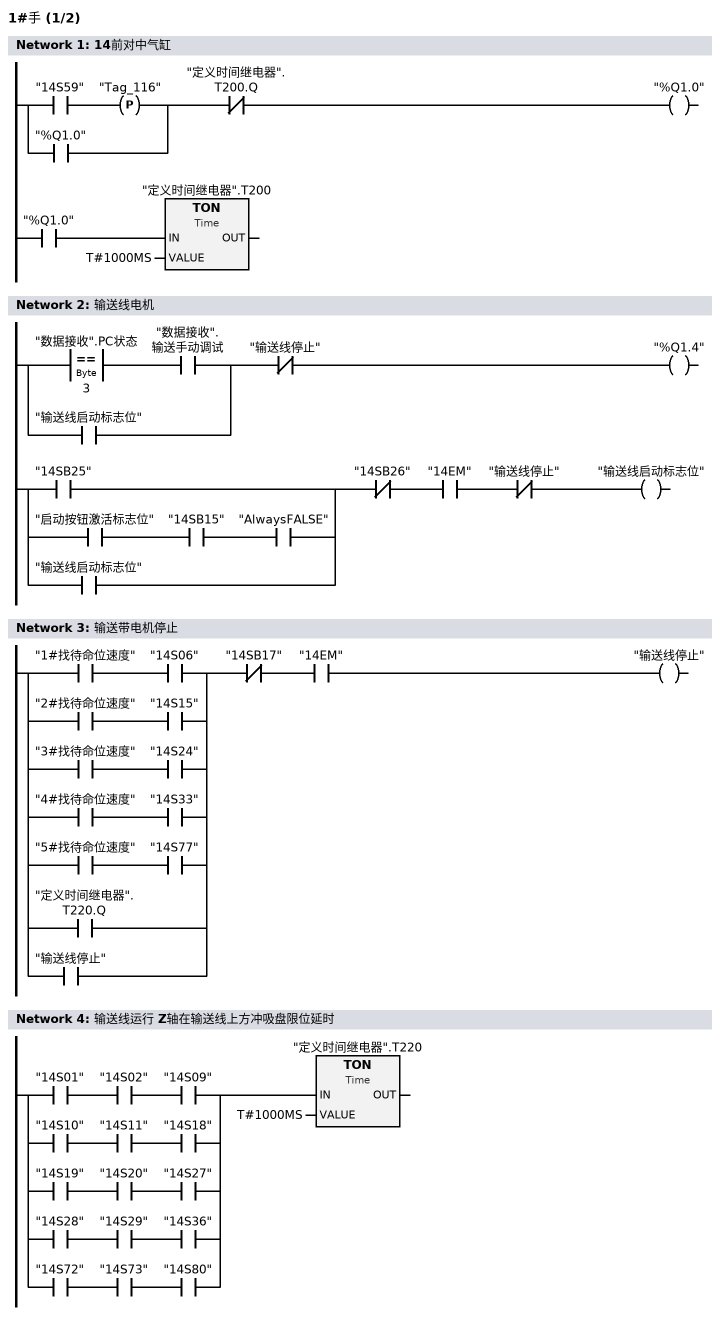
   #_w1 := "14S59" AND NOT "Tag_116";   // rising edge
   "Tag_116" := "14S59";
   "%Q1.0" := (#_w1 OR "%Q1.0") AND NOT "定义时间继电器".T200.Q;
   "定义时间继电器".T200.TON(IN := "%Q1.0", PT := T#1000MS);   // TON coil
END_REGION

REGION Network 2: 输送线电机
   RUNG wire#powerrail
      { S7_Templates := "SrcType := Byte" } EQ_Contact(in1 := "数据接收".PC状态, in2 := 3)
      Contact( "数据接收".输送手动调试 )
      wire#w1
      I_Contact( "输送线停止" )
      Coil( "%Q1.4" )
   END_RUNG
   RUNG wire#powerrail
      Contact( "输送线启动标志位" )
   END_RUNG wire#w1
   RUNG wire#powerrail
      Contact( "14SB25" )
      wire#w2
      I_Contact( "14SB26" )
      Contact( "14EM" )
      I_Contact( "输送线停止" )
      Coil( "输送线启动标志位" )
   END_RUNG
   RUNG wire#powerrail
      Contact( "启动按钮激活标志位" )
      Contact( "14SB15" )
      Contact( "AlwaysFALSE" )
   END_RUNG wire#w2
   RUNG wire#powerrail
      Contact( "输送线启动标志位" )
   END_RUNG wire#w2
   // the same network as SCL:
   "%Q1.4" := ((("数据接收".PC状态 = 3) AND "数据接收".输送手动调试) OR "输送线启动标志位") AND NOT "输送线停止";
   "输送线启动标志位" := ("14SB25" OR ("启动按钮激活标志位" AND "14SB15" AND "AlwaysFALSE") OR "输送线启动标志位") AND NOT "14SB26" AND "14EM" AND NOT "输送线停止";
END_REGION

REGION Network 3: 输送带电机停止
   RUNG wire#powerrail
      Contact( "1#找待命位速度" )
      Contact( "14S06" )
      wire#w1
      I_Contact( "14SB17" )
      Contact( "14EM" )
      Coil( "输送线停止" )
   END_RUNG
   RUNG wire#powerrail
      Contact( "2#找待命位速度" )
      Contact( "14S15" )
   END_RUNG wire#w1
   RUNG wire#powerrail
      Contact( "3#找待命位速度" )
      Contact( "14S24" )
   END_RUNG wire#w1
   RUNG wire#powerrail
      Contact( "4#找待命位速度" )
      Contact( "14S33" )
   END_RUNG wire#w1
   RUNG wire#powerrail
      Contact( "5#找待命位速度" )
      Contact( "14S77" )
   END_RUNG wire#w1
   RUNG wire#powerrail
      Contact( "定义时间继电器".T220.Q )
   END_RUNG wire#w1
   RUNG wire#powerrail
      Contact( "输送线停止" )
   END_RUNG wire#w1
   // the same network as SCL:
   "输送线停止" := (("1#找待命位速度" AND "14S06") OR ("2#找待命位速度" AND "14S15") OR ("3#找待命位速度" AND "14S24") OR ("4#找待命位速度" AND "14S33") OR ("5#找待命位速度" AND "14S77") OR "定义时间继电器".T220.Q OR "输送线停止") AND NOT "14SB17" AND "14EM";
END_REGION

REGION Network 4: 输送线运行 Z轴在输送线上方冲吸盘限位延时
   "定义时间继电器".T220.TON(IN := ("14S01" AND "14S02" AND "14S09") OR ("14S10" AND "14S11" AND "14S18") OR ("14S19" AND "14S20" AND "14S27") OR ("14S28" AND "14S29" AND "14S36") OR ("14S72" AND "14S73" AND "14S80"), PT := T#1000MS);   // TON coil
END_REGION

REGION Network 5: 1#机械手执行流程
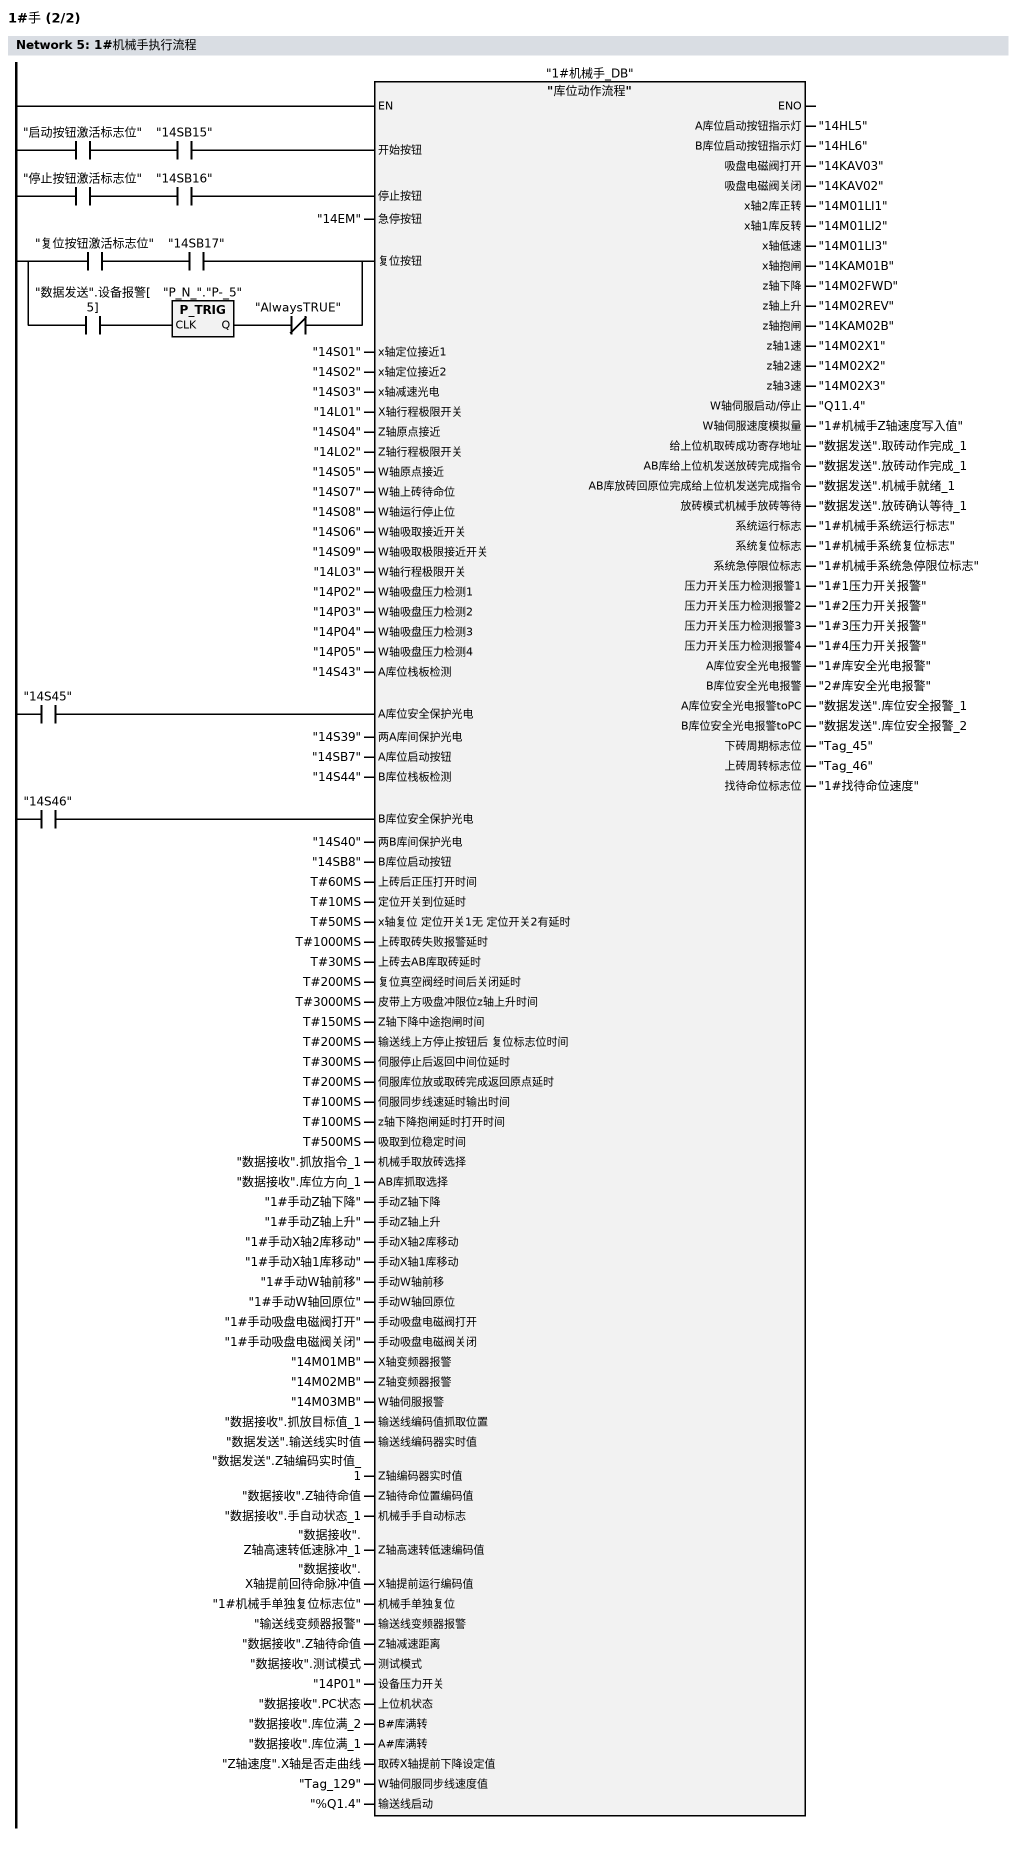
   RUNG wire#powerrail
      "1#机械手_DB"(开始按钮 := wire#w1, 停止按钮 := wire#w2, 复位按钮 := wire#w3, A库位安全保护光电 := wire#w4, B库位安全保护光电 := wire#w5, 急停按钮 := "14EM", x轴定位接近1 := "14S01", x轴定位接近2 := "14S02", x轴减速光电 := "14S03", X轴行程极限开关 := "14L01", Z轴原点接近 := "14S04", Z轴行程极限开关 := "14L02", W轴原点接近 := "14S05", W轴上砖待命位 := "14S07", W轴运行停止位 := "14S08", W轴吸取接近开关 := "14S06", W轴吸取极限接近开关 := "14S09", W轴行程极限开关 := "14L03", W轴吸盘压力检测1 := "14P02", W轴吸盘压力检测2 := "14P03", W轴吸盘压力检测3 := "14P04", W轴吸盘压力检测4 := "14P05", A库位栈板检测 := "14S43", 两A库间保护光电 := "14S39", A库位启动按钮 := "14SB7", B库位栈板检测 := "14S44", 两B库间保护光电 := "14S40", B库位启动按钮 := "14SB8", 上砖后正压打开时间 := T#60MS, 定位开关到位延时 := T#10MS, "x轴复位 定位开关1无 定位开关2有延时" := T#50MS, 上砖取砖失败报警延时 := T#1000MS, 上砖去AB库取砖延时 := T#30MS, 复位真空阀经时间后关闭延时 := T#200MS, 皮带上方吸盘冲限位z轴上升时间 := T#3000MS, Z轴下降中途抱闸时间 := T#150MS, "输送线上方停止按钮后 复位标志位时间" := T#200MS, 伺服停止后返回中间位延时 := T#300MS, 伺服库位放或取砖完成返回原点延时 := T#200MS, 伺服同步线速延时输出时间 := T#100MS, z轴下降抱闸延时打开时间 := T#100MS, 吸取到位稳定时间 := T#500MS, 机械手取放砖选择 := "数据接收".抓放指令_1, AB库抓取选择 := "数据接收".库位方向_1, 手动Z轴下降 := "1#手动Z轴下降", 手动Z轴上升 := "1#手动Z轴上升", 手动X轴2库移动 := "1#手动X轴2库移动", 手动X轴1库移动 := "1#手动X轴1库移动", 手动W轴前移 := "1#手动W轴前移", 手动W轴回原位 := "1#手动W轴回原位", 手动吸盘电磁阀打开 := "1#手动吸盘电磁阀打开", 手动吸盘电磁阀关闭 := "1#手动吸盘电磁阀关闭", X轴变频器报警 := "14M01MB", Z轴变频器报警 := "14M02MB", W轴伺服报警 := "14M03MB", 输送线编码值抓取位置 := "数据接收".抓放目标值_1, 输送线编码器实时值 := "数据发送".输送线实时值, Z轴编码器实时值 := "数据发送".Z轴编码实时值_1, Z轴待命位置编码值 := "数据接收".Z轴待命值, 机械手手自动标志 := "数据接收".手自动状态_1, Z轴高速转低速编码值 := "数据接收".Z轴高速转低速脉冲_1, X轴提前运行编码值 := "数据接收".X轴提前回待命脉冲值, 机械手单独复位 := "1#机械手单独复位标志位", 输送线变频器报警 := "输送线变频器报警", Z轴减速距离 := "数据接收".Z轴待命值, 测试模式 := "数据接收".测试模式, 设备压力开关 := "14P01", 上位机状态 := "数据接收".PC状态, "B#库满转" := "数据接收".库位满_2, "A#库满转" := "数据接收".库位满_1, 取砖X轴提前下降设定值 := "Z轴速度".X轴是否走曲线, W轴伺服同步线速度值 := "Tag_129", 输送线启动 := "%Q1.4", A库位启动按钮指示灯 => "14HL5", B库位启动按钮指示灯 => "14HL6", 吸盘电磁阀打开 => "14KAV03", 吸盘电磁阀关闭 => "14KAV02", x轴2库正转 => "14M01LI1", x轴1库反转 => "14M01LI2", x轴低速 => "14M01LI3", x轴抱闸 => "14KAM01B", z轴下降 => "14M02FWD", z轴上升 => "14M02REV", z轴抱闸 => "14KAM02B", z轴1速 => "14M02X1", z轴2速 => "14M02X2", z轴3速 => "14M02X3", "W轴伺服启动/停止" => "Q11.4", W轴伺服速度模拟量 => "1#机械手Z轴速度写入值", 给上位机取砖成功寄存地址 => "数据发送".取砖动作完成_1, AB库给上位机发送放砖完成指令 => "数据发送".放砖动作完成_1, AB库放砖回原位完成给上位机发送完成指令 => "数据发送".机械手就绪_1, 放砖模式机械手放砖等待 => "数据发送".放砖确认等待_1, 系统运行标志 => "1#机械手系统运行标志", 系统复位标志 => "1#机械手系统复位标志", 系统急停限位标志 => "1#机械手系统急停限位标志", 压力开关压力检测报警1 => "1#1压力开关报警", 压力开关压力检测报警2 => "1#2压力开关报警", 压力开关压力检测报警3 => "1#3压力开关报警", 压力开关压力检测报警4 => "1#4压力开关报警", A库位安全光电报警 => "1#库安全光电报警", B库位安全光电报警 => "2#库安全光电报警", A库位安全光电报警toPC => "数据发送".库位安全报警_1, B库位安全光电报警toPC => "数据发送".库位安全报警_2, 下砖周期标志位 => "Tag_45", 上砖周转标志位 => "Tag_46", 找待命位标志位 => "1#找待命位速度")
   END_RUNG
   RUNG wire#powerrail
      Contact( "启动按钮激活标志位" )
      Contact( "14SB15" )
   END_RUNG wire#w1
   RUNG wire#powerrail
      Contact( "停止按钮激活标志位" )
      Contact( "14SB16" )
   END_RUNG wire#w2
   RUNG wire#powerrail
      Contact( "复位按钮激活标志位" )
      Contact( "14SB17" )
   END_RUNG wire#w3
   RUNG wire#powerrail
      Contact( "数据发送".设备报警[5] )
      P_Trig( "P_N_"."P-_5" )
      I_Contact( "AlwaysTRUE" )
   END_RUNG wire#w3
   RUNG wire#powerrail
      Contact( "14S45" )
   END_RUNG wire#w4
   RUNG wire#powerrail
      Contact( "14S46" )
   END_RUNG wire#w5
   // the same network as SCL:
   #_w1 := "数据发送".设备报警[5] AND NOT "P_N_"."P-_5";   // rising edge
   "P_N_"."P-_5" := "数据发送".设备报警[5];
   "1#机械手_DB"(开始按钮 := "启动按钮激活标志位" AND "14SB15",   // "库位动作流程"
              停止按钮 := "停止按钮激活标志位" AND "14SB16",
              急停按钮 := "14EM",
              复位按钮 := ("复位按钮激活标志位" AND "14SB17") OR (#_w1 AND NOT "AlwaysTRUE"),
              x轴定位接近1 := "14S01",
              x轴定位接近2 := "14S02",
              x轴减速光电 := "14S03",
              X轴行程极限开关 := "14L01",
              Z轴原点接近 := "14S04",
              Z轴行程极限开关 := "14L02",
              W轴原点接近 := "14S05",
              W轴上砖待命位 := "14S07",
              W轴运行停止位 := "14S08",
              W轴吸取接近开关 := "14S06",
              W轴吸取极限接近开关 := "14S09",
              W轴行程极限开关 := "14L03",
              W轴吸盘压力检测1 := "14P02",
              W轴吸盘压力检测2 := "14P03",
              W轴吸盘压力检测3 := "14P04",
              W轴吸盘压力检测4 := "14P05",
              A库位栈板检测 := "14S43",
              A库位安全保护光电 := "14S45",
              两A库间保护光电 := "14S39",
              A库位启动按钮 := "14SB7",
              B库位栈板检测 := "14S44",
              B库位安全保护光电 := "14S46",
              两B库间保护光电 := "14S40",
              B库位启动按钮 := "14SB8",
              上砖后正压打开时间 := T#60MS,
              定位开关到位延时 := T#10MS,
              "x轴复位 定位开关1无 定位开关2有延时" := T#50MS,
              上砖取砖失败报警延时 := T#1000MS,
              上砖去AB库取砖延时 := T#30MS,
              复位真空阀经时间后关闭延时 := T#200MS,
              皮带上方吸盘冲限位z轴上升时间 := T#3000MS,
              Z轴下降中途抱闸时间 := T#150MS,
              "输送线上方停止按钮后 复位标志位时间" := T#200MS,
              伺服停止后返回中间位延时 := T#300MS,
              伺服库位放或取砖完成返回原点延时 := T#200MS,
              伺服同步线速延时输出时间 := T#100MS,
              z轴下降抱闸延时打开时间 := T#100MS,
              吸取到位稳定时间 := T#500MS,
              机械手取放砖选择 := "数据接收".抓放指令_1,
              AB库抓取选择 := "数据接收".库位方向_1,
              手动Z轴下降 := "1#手动Z轴下降",
              手动Z轴上升 := "1#手动Z轴上升",
              手动X轴2库移动 := "1#手动X轴2库移动",
              手动X轴1库移动 := "1#手动X轴1库移动",
              手动W轴前移 := "1#手动W轴前移",
              手动W轴回原位 := "1#手动W轴回原位",
              手动吸盘电磁阀打开 := "1#手动吸盘电磁阀打开",
              手动吸盘电磁阀关闭 := "1#手动吸盘电磁阀关闭",
              X轴变频器报警 := "14M01MB",
              Z轴变频器报警 := "14M02MB",
              W轴伺服报警 := "14M03MB",
              输送线编码值抓取位置 := "数据接收".抓放目标值_1,
              输送线编码器实时值 := "数据发送".输送线实时值,
              Z轴编码器实时值 := "数据发送".Z轴编码实时值_1,
              Z轴待命位置编码值 := "数据接收".Z轴待命值,
              机械手手自动标志 := "数据接收".手自动状态_1,
              Z轴高速转低速编码值 := "数据接收".Z轴高速转低速脉冲_1,
              X轴提前运行编码值 := "数据接收".X轴提前回待命脉冲值,
              机械手单独复位 := "1#机械手单独复位标志位",
              输送线变频器报警 := "输送线变频器报警",
              Z轴减速距离 := "数据接收".Z轴待命值,
              测试模式 := "数据接收".测试模式,
              设备压力开关 := "14P01",
              上位机状态 := "数据接收".PC状态,
              "B#库满转" := "数据接收".库位满_2,
              "A#库满转" := "数据接收".库位满_1,
              取砖X轴提前下降设定值 := "Z轴速度".X轴是否走曲线,
              W轴伺服同步线速度值 := "Tag_129",
              输送线启动 := "%Q1.4",
              A库位启动按钮指示灯 => "14HL5",
              B库位启动按钮指示灯 => "14HL6",
              吸盘电磁阀打开 => "14KAV03",
              吸盘电磁阀关闭 => "14KAV02",
              x轴2库正转 => "14M01LI1",
              x轴1库反转 => "14M01LI2",
              x轴低速 => "14M01LI3",
              x轴抱闸 => "14KAM01B",
              z轴下降 => "14M02FWD",
              z轴上升 => "14M02REV",
              z轴抱闸 => "14KAM02B",
              z轴1速 => "14M02X1",
              z轴2速 => "14M02X2",
              z轴3速 => "14M02X3",
              "W轴伺服启动/停止" => "Q11.4",
              W轴伺服速度模拟量 => "1#机械手Z轴速度写入值",
              给上位机取砖成功寄存地址 => "数据发送".取砖动作完成_1,
              AB库给上位机发送放砖完成指令 => "数据发送".放砖动作完成_1,
              AB库放砖回原位完成给上位机发送完成指令 => "数据发送".机械手就绪_1,
              放砖模式机械手放砖等待 => "数据发送".放砖确认等待_1,
              系统运行标志 => "1#机械手系统运行标志",
              系统复位标志 => "1#机械手系统复位标志",
              系统急停限位标志 => "1#机械手系统急停限位标志",
              压力开关压力检测报警1 => "1#1压力开关报警",
              压力开关压力检测报警2 => "1#2压力开关报警",
              压力开关压力检测报警3 => "1#3压力开关报警",
              压力开关压力检测报警4 => "1#4压力开关报警",
              A库位安全光电报警 => "1#库安全光电报警",
              B库位安全光电报警 => "2#库安全光电报警",
              A库位安全光电报警toPC => "数据发送".库位安全报警_1,
              B库位安全光电报警toPC => "数据发送".库位安全报警_2,
              下砖周期标志位 => "Tag_45",
              上砖周转标志位 => "Tag_46",
              找待命位标志位 => "1#找待命位速度");
END_REGION
END_FUNCTION

FUNCTION "编码器/线速度" : Void   // FC12, LAD
{ S7_Optimized_Access := 'TRUE' }
VERSION : 0.1
   VAR_TEMP   // added for the SCL form of the ladder/FBD networks
      _w1 : Bool;
      _w2 : Bool;
      _w3 : Bool;
      _w4 : Bool;
      _w5 : Bool;
   END_VAR
BEGIN

REGION Network 1: 控制软件门：• 上升沿： 软件门打开
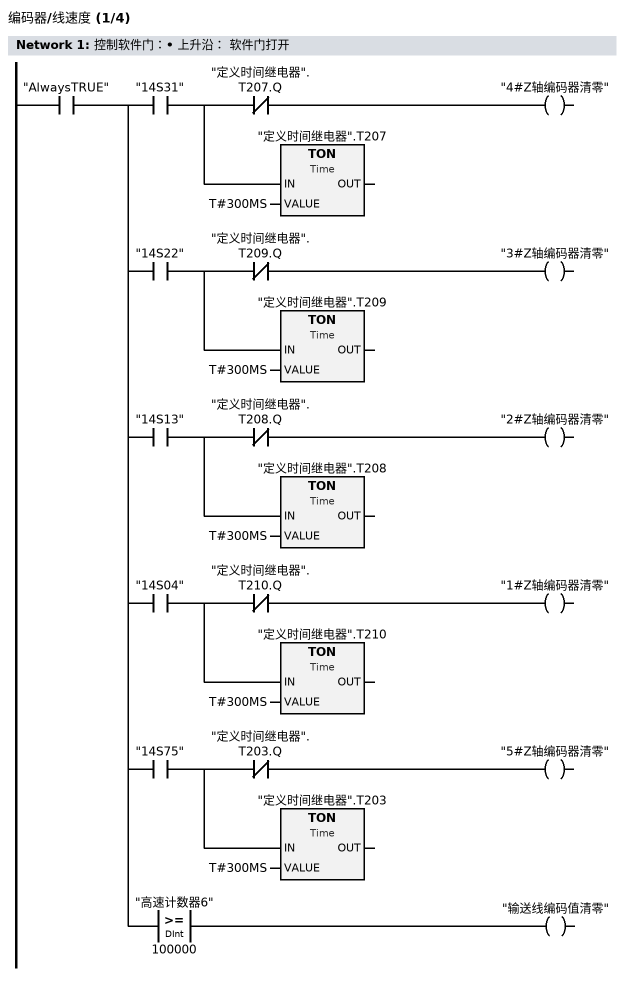
   #_w1 := "AlwaysTRUE" AND "14S31";
   "4#Z轴编码器清零" := #_w1 AND NOT "定义时间继电器".T207.Q;
   "定义时间继电器".T207.TON(IN := #_w1, PT := T#300MS);   // TON coil
   #_w2 := "AlwaysTRUE" AND "14S22";
   "3#Z轴编码器清零" := #_w2 AND NOT "定义时间继电器".T209.Q;
   "定义时间继电器".T209.TON(IN := #_w2, PT := T#300MS);   // TON coil
   #_w3 := "AlwaysTRUE" AND "14S13";
   "2#Z轴编码器清零" := #_w3 AND NOT "定义时间继电器".T208.Q;
   "定义时间继电器".T208.TON(IN := #_w3, PT := T#300MS);   // TON coil
   #_w4 := "AlwaysTRUE" AND "14S04";
   "1#Z轴编码器清零" := #_w4 AND NOT "定义时间继电器".T210.Q;
   "定义时间继电器".T210.TON(IN := #_w4, PT := T#300MS);   // TON coil
   #_w5 := "AlwaysTRUE" AND "14S75";
   "5#Z轴编码器清零" := #_w5 AND NOT "定义时间继电器".T203.Q;
   "定义时间继电器".T203.TON(IN := #_w5, PT := T#300MS);   // TON coil
   "输送线编码值清零" := "AlwaysTRUE" AND ("高速计数器6" >= 100000);
END_REGION

REGION Network 2: 1#机械手编码器数值读取
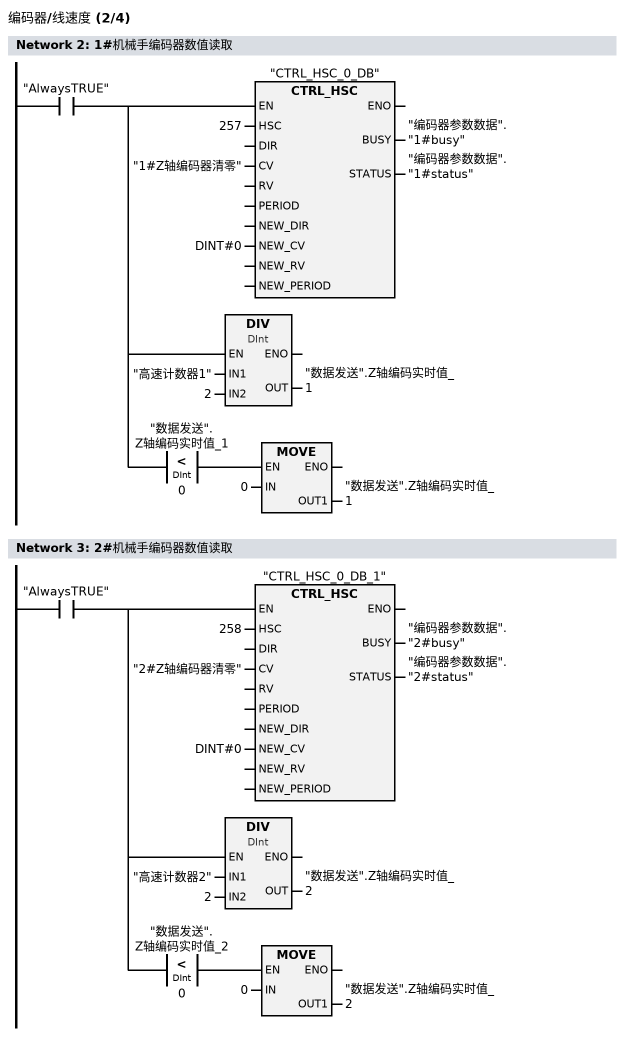
   #_w1 := "AlwaysTRUE";
   IF #_w1 THEN
       "CTRL_HSC_0_DB"(HSC := 257,   // CTRL_HSC
                       CV := "1#Z轴编码器清零",
                       NEW_CV := DINT#0,
                       BUSY => "编码器参数数据"."1#busy",
                       STATUS => "编码器参数数据"."1#status");
       "数据发送".Z轴编码实时值_1 := "高速计数器1" / 2;
   END_IF;
   IF #_w1 AND ("数据发送".Z轴编码实时值_1 < 0) THEN "数据发送".Z轴编码实时值_1 := 0; END_IF;
END_REGION

REGION Network 3: 2#机械手编码器数值读取
   #_w1 := "AlwaysTRUE";
   IF #_w1 THEN
       "CTRL_HSC_0_DB_1"(HSC := 258,   // CTRL_HSC
                         CV := "2#Z轴编码器清零",
                         NEW_CV := DINT#0,
                         BUSY => "编码器参数数据"."2#busy",
                         STATUS => "编码器参数数据"."2#status");
       "数据发送".Z轴编码实时值_2 := "高速计数器2" / 2;
   END_IF;
   IF #_w1 AND ("数据发送".Z轴编码实时值_2 < 0) THEN "数据发送".Z轴编码实时值_2 := 0; END_IF;
END_REGION

REGION Network 4: 3#机械手编码器数值读取
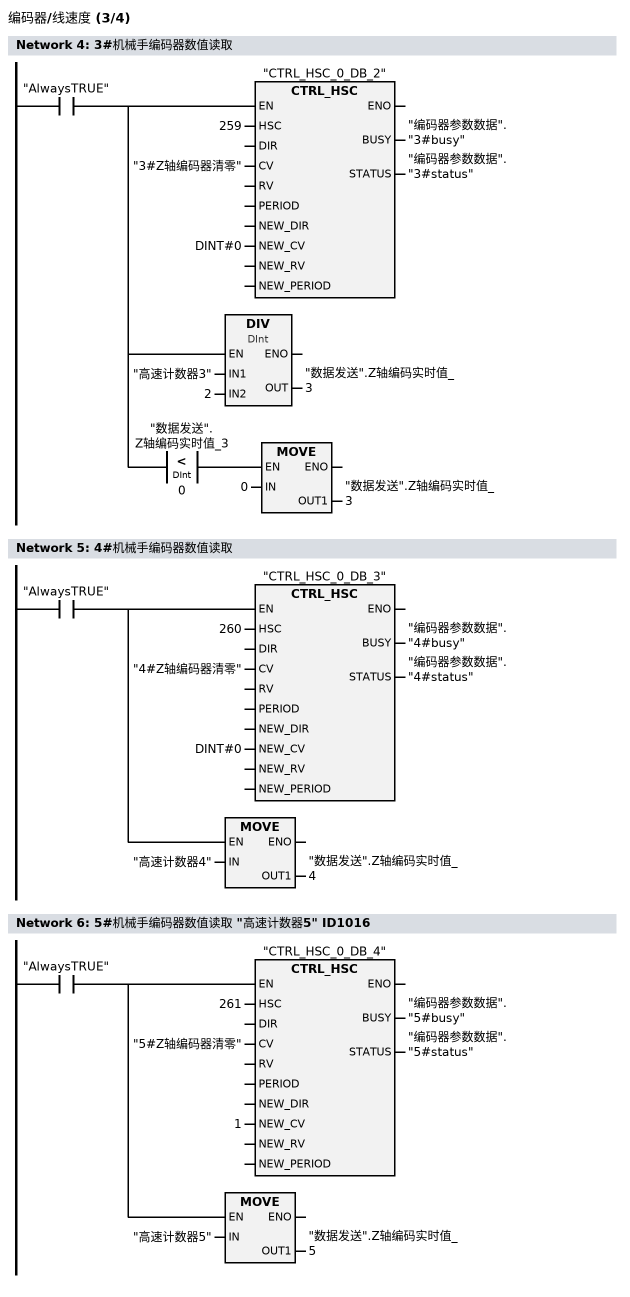
   #_w1 := "AlwaysTRUE";
   IF #_w1 THEN
       "CTRL_HSC_0_DB_2"(HSC := 259,   // CTRL_HSC
                         CV := "3#Z轴编码器清零",
                         NEW_CV := DINT#0,
                         BUSY => "编码器参数数据"."3#busy",
                         STATUS => "编码器参数数据"."3#status");
       "数据发送".Z轴编码实时值_3 := "高速计数器3" / 2;
   END_IF;
   IF #_w1 AND ("数据发送".Z轴编码实时值_3 < 0) THEN "数据发送".Z轴编码实时值_3 := 0; END_IF;
END_REGION

REGION Network 5: 4#机械手编码器数值读取
   #_w1 := "AlwaysTRUE";
   IF #_w1 THEN
       "CTRL_HSC_0_DB_3"(HSC := 260,   // CTRL_HSC
                         CV := "4#Z轴编码器清零",
                         NEW_CV := DINT#0,
                         BUSY => "编码器参数数据"."4#busy",
                         STATUS => "编码器参数数据"."4#status");
       "数据发送".Z轴编码实时值_4 := "高速计数器4";
   END_IF;
END_REGION

REGION Network 6: 5#机械手编码器数值读取 "高速计数器5" ID1016
   #_w1 := "AlwaysTRUE";
   IF #_w1 THEN
       "CTRL_HSC_0_DB_4"(HSC := 261,   // CTRL_HSC
                         CV := "5#Z轴编码器清零",
                         NEW_CV := 1,
                         BUSY => "编码器参数数据"."5#busy",
                         STATUS => "编码器参数数据"."5#status");
       "数据发送".Z轴编码实时值_5 := "高速计数器5";
   END_IF;
END_REGION

REGION Network 7: 输送线编码器数值读取 高速计数器6 ID1020
